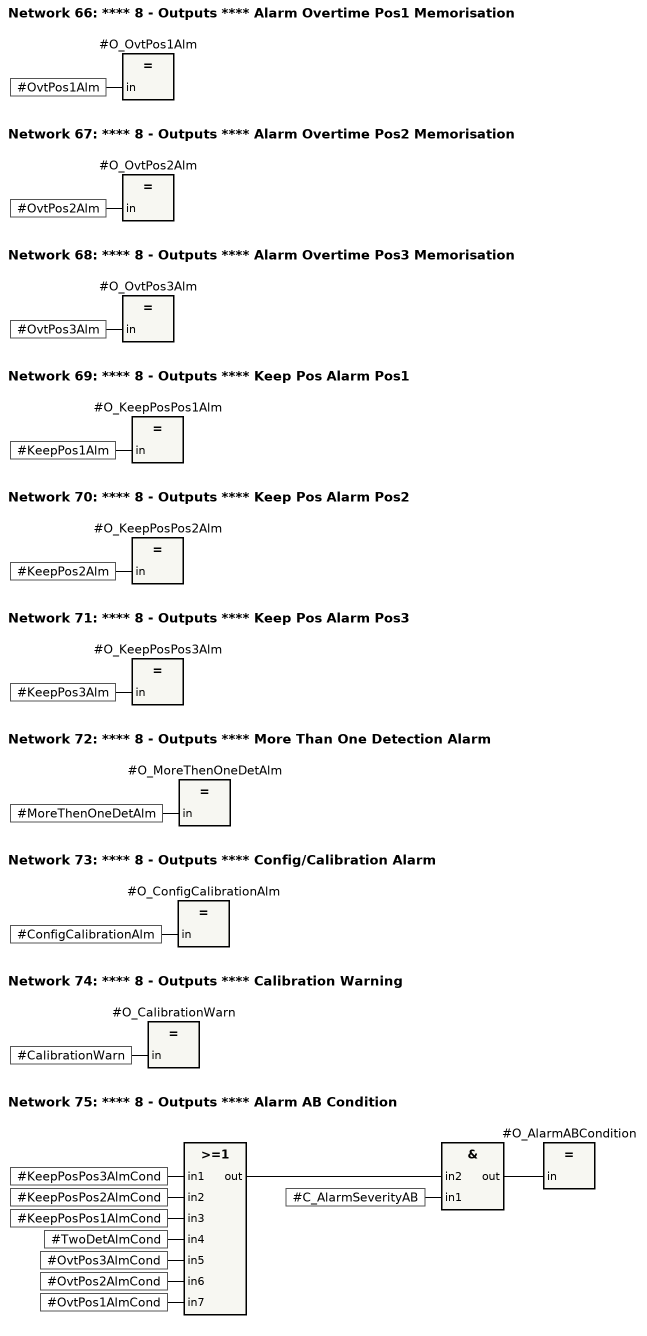
   #O_OvtPos1Alm := #OvtPos1Alm;
END_REGION

REGION Network 67: **** 8 - Outputs **** Alarm Overtime Pos2 Memorisation
   // Alarm Overtime Pos2 Memorisation
   #O_OvtPos2Alm := #OvtPos2Alm;
END_REGION

REGION Network 68: **** 8 - Outputs **** Alarm Overtime Pos3 Memorisation
   // Alarm Overtime Pos3  Memorisation
   #O_OvtPos3Alm := #OvtPos3Alm;
END_REGION

REGION Network 69: **** 8 - Outputs **** Keep Pos Alarm Pos1
   // Keep Pos Alarm Pos1
   #O_KeepPosPos1Alm := #KeepPos1Alm;
END_REGION

REGION Network 70: **** 8 - Outputs **** Keep Pos Alarm Pos2
   // Keep Pos Alarm Pos2
   #O_KeepPosPos2Alm := #KeepPos2Alm;
END_REGION

REGION Network 71: **** 8 - Outputs **** Keep Pos Alarm Pos3
   // Keep Pos Alarm Pos3
   #O_KeepPosPos3Alm := #KeepPos3Alm;
END_REGION

REGION Network 72: **** 8 - Outputs **** More Than One Detection Alarm
   // More Than One Detection Alarm
   #O_MoreThenOneDetAlm := #MoreThenOneDetAlm;
END_REGION

REGION Network 73: **** 8 - Outputs **** Config/Calibration Alarm
   #O_ConfigCalibrationAlm := #ConfigCalibrationAlm;
END_REGION

REGION Network 74: **** 8 - Outputs **** Calibration Warning
   #O_CalibrationWarn := #CalibrationWarn;
END_REGION

REGION Network 75: **** 8 - Outputs **** Alarm AB Condition
   // Alarm AB Condition
   #O_AlarmABCondition := (#KeepPosPos3AlmCond OR #KeepPosPos2AlmCond OR #KeepPosPos1AlmCond OR #TwoDetAlmCond OR #OvtPos3AlmCond OR #OvtPos2AlmCond OR #OvtPos1AlmCond) AND #C_AlarmSeverityAB;
END_REGION
END_FUNCTION_BLOCK

FUNCTION_BLOCK "LMovFnc3Pos2S"   // FB2192, FBD
TITLE = LMovFnc3Pos2S
{ S7_Optimized_Access := 'TRUE' }
VERSION : 0.1
// =============================================================================
// This module will be used for the steering of a three Position movement wit 2 speed
// It will get the commands from different Modes, evaluate the status of the 
// Interlock and give the command to the Actuator or direct to simple outputs.
// =============================================================================
// stored: AutoNumber false, IsIECCheckEnabled false, IsRetainMemResEnabled false, MemoryReserve 100, SetENOAutomatically False, UDAEnableTagReadback false
   VAR_INPUT
      I_Pos1 { ExternalAccessible := 'False'; ExternalVisible := 'False'; ExternalWritable := 'False'} : Bool;   // Position 1 Detection or Summary
      I_Pos2 { ExternalAccessible := 'False'; ExternalVisible := 'False'; ExternalWritable := 'False'} : Bool;   // Position 2 Detection or Summary
      I_Pos3 { ExternalAccessible := 'False'; ExternalVisible := 'False'; ExternalWritable := 'False'} : Bool;   // Position 3 Detection or Summary
      I_SlowPos1 { ExternalAccessible := 'False'; ExternalVisible := 'False'; ExternalWritable := 'False'} : Bool;   // Slow Position 1 Detection
      I_SlowPos2 { ExternalAccessible := 'False'; ExternalVisible := 'False'; ExternalWritable := 'False'} : Bool;   // Slow Position 2 Detection
      I_SlowPos3 { ExternalAccessible := 'False'; ExternalVisible := 'False'; ExternalWritable := 'False'} : Bool;   // Slow Position 3 Detection
      I_PBSet { ExternalAccessible := 'False'; ExternalVisible := 'False'; ExternalWritable := 'False'} : Bool;   // Push button for Set direction (used in manual with button OP panels )
      I_PBReset { ExternalAccessible := 'False'; ExternalVisible := 'False'; ExternalWritable := 'False'} : Bool;   // Push button for Reset direction (used in manual with Pushbutton OP panels)
      I_Pos1Begin { ExternalAccessible := 'False'; ExternalVisible := 'False'; ExternalWritable := 'False'} : Bool;   // Request Pos 1 Function Begin
      I_Pos2Begin { ExternalAccessible := 'False'; ExternalVisible := 'False'; ExternalWritable := 'False'} : Bool;   // Request Pos 2 Function Begin
      I_Pos3Begin { ExternalAccessible := 'False'; ExternalVisible := 'False'; ExternalWritable := 'False'} : Bool;   // Request Pos 3 Function Begin
      I_SetIntlkOK { ExternalAccessible := 'False'; ExternalVisible := 'False'; ExternalWritable := 'False'} : Bool;   // Interlock Set Ok
      I_ResIntlkOK { ExternalAccessible := 'False'; ExternalVisible := 'False'; ExternalWritable := 'False'} : Bool;   // Interlock Reset Ok
      I_SafetyOk { ExternalAccessible := 'False'; ExternalVisible := 'False'; ExternalWritable := 'False'} : Bool;   // Safety ok
      I_HardwareOk { ExternalAccessible := 'False'; ExternalVisible := 'False'; ExternalWritable := 'False'} : Bool;   // Safety Ok / Hardware Ok
   END_VAR
   VAR_OUTPUT
      O_CmdSetHighSpeed { ExternalAccessible := 'False'; ExternalVisible := 'False'; ExternalWritable := 'False'} : Bool;   // Command to Activate Set movement
      O_CmdResHighSpeed { ExternalAccessible := 'False'; ExternalVisible := 'False'; ExternalWritable := 'False'} : Bool;   // Command to Activate Reset movement
      O_CmdSetLowSpeed { ExternalAccessible := 'False'; ExternalVisible := 'False'; ExternalWritable := 'False'} : Bool;   // Command to Activate Slow Set movement
      O_CmdResLowSpeed { ExternalAccessible := 'False'; ExternalVisible := 'False'; ExternalWritable := 'False'} : Bool;   // Command to Activate Slow Reset movement
      O_CmdPos1 { ExternalAccessible := 'False'; ExternalVisible := 'False'; ExternalWritable := 'False'} : Bool;   // Command to activate Set movement / Command to Activate Pos1 movement
      O_CmdPos2 { ExternalAccessible := 'False'; ExternalVisible := 'False'; ExternalWritable := 'False'} : Bool;   // Command to activate Set movement / Command to Activate Pos2 movement
      O_CmdPos3 { ExternalAccessible := 'False'; ExternalVisible := 'False'; ExternalWritable := 'False'} : Bool;   // Command to activate Reset movement / Command to Activate Pos3 movement
      O_FuncRunning { ExternalAccessible := 'False'; ExternalVisible := 'False'; ExternalWritable := 'False'} : Bool;   // Signal that the function is running
      O_FuncBusyTM { ExternalAccessible := 'False'; ExternalVisible := 'False'; ExternalWritable := 'False'} : Bool;   // Memory Signal that the function is busy
      O_Pos1Finished { ExternalAccessible := 'False'; ExternalVisible := 'False'; ExternalWritable := 'False'} : Bool;   // Position1 Finished
      O_Pos2Finished { ExternalAccessible := 'False'; ExternalVisible := 'False'; ExternalWritable := 'False'} : Bool;   // Position2 Finished
      O_Pos3Finished { ExternalAccessible := 'False'; ExternalVisible := 'False'; ExternalWritable := 'False'} : Bool;   // Position3 Finished
      O_IntlkSetAlm { ExternalAccessible := 'False'; ExternalVisible := 'False'; ExternalWritable := 'False'} : Bool;   // Alarm Interlock Set
      O_IntlkResAlm { ExternalAccessible := 'False'; ExternalVisible := 'False'; ExternalWritable := 'False'} : Bool;   // Alarm Interlock Reset
      O_FuncIsSelInMan { ExternalAccessible := 'False'; ExternalVisible := 'False'; ExternalWritable := 'False'} : Bool;   // The function is Selected in manual Mode
      O_LED { ExternalAccessible := 'False'; ExternalVisible := 'False'; ExternalWritable := 'False'} : Bool;   // LED - Indication
      O_AlarmABCondition { ExternalAccessible := 'False'; ExternalVisible := 'False'; ExternalWritable := 'False'} : Bool;   // Alarms AB condition
   END_VAR
   VAR_IN_OUT
      IO_Modes : "Modes";   // Modes
      H_HMI : "H_HMI";   // Animation
      H_MovFnc3Pos2S : "H_MovFnc3Pos";   // Animation
      H_FncSelInHMI { ExternalAccessible := 'False'; ExternalVisible := 'False'; ExternalWritable := 'False'} : Bool;   // This function is Selected to run from HMI
      C_AlarmResetUsed { ExternalAccessible := 'False'; ExternalVisible := 'False'; ExternalWritable := 'False'} : Bool;   // If true, the alrms will be stored untill Reseted
      C_EnableMemBegin { ExternalAccessible := 'False'; ExternalVisible := 'False'; ExternalWritable := 'False'} : Bool;   // Enable memory Begin (Command request is memorised until pos reached)
      C_EnIntlkAlm { ExternalAccessible := 'False'; ExternalVisible := 'False'; ExternalWritable := 'False'} : Bool := TRUE;   // Enable Interlock Alarm
      C_ForceManual { ExternalAccessible := 'False'; ExternalVisible := 'False'; ExternalWritable := 'False'} : Bool := FALSE;   // Force Manual
   END_VAR
   VAR
      ResetAlarm { ExternalAccessible := 'False'; ExternalVisible := 'False'; ExternalWritable := 'False'} : Bool;   // Reset Alarm Memory
      BeginPos1Req { ExternalAccessible := 'False'; ExternalVisible := 'False'; ExternalWritable := 'False'} : Bool;   // Request Pos 1 Function Begin
      BeginPos2Req { ExternalAccessible := 'False'; ExternalVisible := 'False'; ExternalWritable := 'False'} : Bool;   // Request Pos 2 Function Begin
      BeginPos3Req { ExternalAccessible := 'False'; ExternalVisible := 'False'; ExternalWritable := 'False'} : Bool;   // Request Pos 3 Function Begin
      CmdSet { ExternalAccessible := 'False'; ExternalVisible := 'False'; ExternalWritable := 'False'} : Bool;   // Command set
      CmdSetSl { ExternalAccessible := 'False'; ExternalVisible := 'False'; ExternalWritable := 'False'} : Bool;   // Command to Activate Slow Set movement
      CmdSetRequest { ExternalAccessible := 'False'; ExternalVisible := 'False'; ExternalWritable := 'False'} : Bool;   // Set Command request to Activate the Interlock
      CmdRes { ExternalAccessible := 'False'; ExternalVisible := 'False'; ExternalWritable := 'False'} : Bool;   // Command Reset
      CmdResSl { ExternalAccessible := 'False'; ExternalVisible := 'False'; ExternalWritable := 'False'} : Bool;   // Command to Activate Slow Reset movement
      CmdResRequest { ExternalAccessible := 'False'; ExternalVisible := 'False'; ExternalWritable := 'False'} : Bool;   // Reset Command request to Activate the Interlock
   END_VAR
   VAR RETAIN
      BetweenPos1Pos2 { ExternalAccessible := 'False'; ExternalVisible := 'False'; ExternalWritable := 'False'} : Bool;   // Table Between Pos 1 And 2
      BetweenPos1Pos2Set { ExternalAccessible := 'False'; ExternalVisible := 'False'; ExternalWritable := 'False'} : Bool;   // Table Between Pos 1 And 2 Set
      BetweenPos1Pos2Res { ExternalAccessible := 'False'; ExternalVisible := 'False'; ExternalWritable := 'False'} : Bool;   // Table Between Pos 1 And 2 Reset
      BetweenPos2Pos3 { ExternalAccessible := 'False'; ExternalVisible := 'False'; ExternalWritable := 'False'} : Bool;   // Table Between Pos 2 And 3
      BetweenPos2Pos3Set { ExternalAccessible := 'False'; ExternalVisible := 'False'; ExternalWritable := 'False'} : Bool;   // Table Between Pos 2 And 3 Set
      BetweenPos2Pos3Res { ExternalAccessible := 'False'; ExternalVisible := 'False'; ExternalWritable := 'False'} : Bool;   // Table Between Pos 2 And 3 Reset
   END_VAR
   VAR
      Pos2SetReached { ExternalAccessible := 'False'; ExternalVisible := 'False'; ExternalWritable := 'False'} : Bool;   // Position 2 Set Reached
      P_CmdSetRequest { ExternalAccessible := 'False'; ExternalVisible := 'False'; ExternalWritable := 'False'} : Bool;   // Cmd Request Set Pos Trig
      Pos2ResReached { ExternalAccessible := 'False'; ExternalVisible := 'False'; ExternalWritable := 'False'} : Bool;   // Position 2 Reset Reached
      P_CmdResRequest { ExternalAccessible := 'False'; ExternalVisible := 'False'; ExternalWritable := 'False'} : Bool;   // Cmd Request Res Pos Trig
      CmdPos1 { ExternalAccessible := 'False'; ExternalVisible := 'False'; ExternalWritable := 'False'} : Bool;   // Command to activate Set movement / Command to Activate Pos1 movement
      CmdPos2 { ExternalAccessible := 'False'; ExternalVisible := 'False'; ExternalWritable := 'False'} : Bool;   // Command to activate Set movement / Command to Activate Pos2 movement
      CmdPos3 { ExternalAccessible := 'False'; ExternalVisible := 'False'; ExternalWritable := 'False'} : Bool;   // Command to activate Reset movement / Command to Activate Pos3 movement
      IntlkSetAlm { ExternalAccessible := 'False'; ExternalVisible := 'False'; ExternalWritable := 'False'} : Bool;   // Alarm Interlock Set
      IntlkResAlm { ExternalAccessible := 'False'; ExternalVisible := 'False'; ExternalWritable := 'False'} : Bool;   // Alarm Interlock Reset
      IntlkSetAlmCond { ExternalAccessible := 'False'; ExternalVisible := 'False'; ExternalWritable := 'False'} : Bool;   // Alarm Interlock Set condition
      IntlkResAlmCond { ExternalAccessible := 'False'; ExternalVisible := 'False'; ExternalWritable := 'False'} : Bool;   // Alarm Interlock Reset condition
      FuncRunning { ExternalAccessible := 'False'; ExternalVisible := 'False'; ExternalWritable := 'False'} : Bool;   // Function is running
      FuncBusyTM { ExternalAccessible := 'False'; ExternalVisible := 'False'; ExternalWritable := 'False'} : Bool;   // Memory Signal that the function is busy
      Edge { ExternalAccessible := 'False'; ExternalVisible := 'False'; ExternalWritable := 'False'} : Array[1..5] of Bool;   // Edge
      AlarmTimer { ExternalAccessible := 'False'; ExternalVisible := 'False'; ExternalWritable := 'False'} : "LTimer";
      AlmFilterResult { ExternalAccessible := 'False'; ExternalVisible := 'False'; ExternalWritable := 'False'} : Bool;
   END_VAR
   VAR_TEMP   // added for the SCL form of the ladder/FBD networks
      _w1 : Bool;
      _w2 : Bool;
      _w3 : Bool;
      _w4 : Bool;
   END_VAR
BEGIN

REGION Network 1: **** 2.2 - Alarms - Alarm Generation **** Alarm Filter
   // Alarm Filter
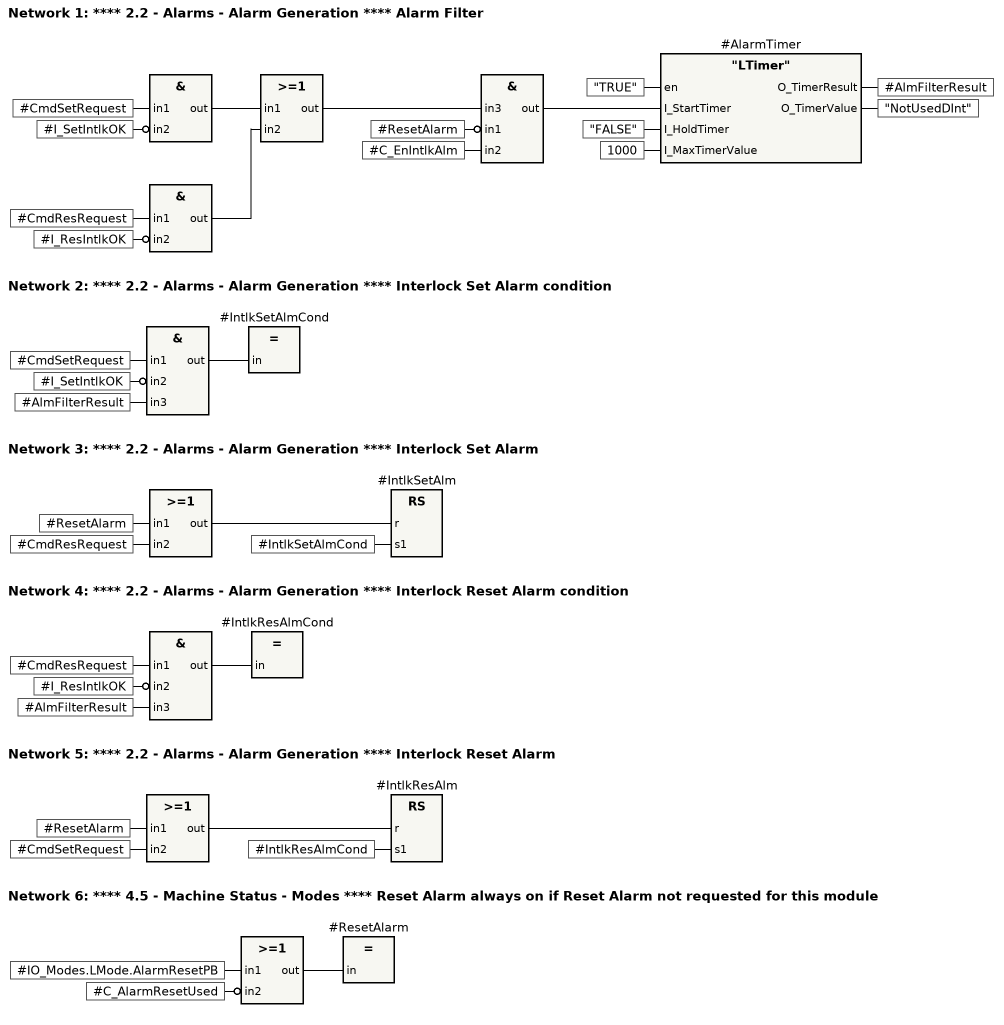
   IF "TRUE" THEN
       #AlarmTimer(I_StartTimer := ((#CmdSetRequest AND NOT #I_SetIntlkOK) OR (#CmdResRequest AND NOT #I_ResIntlkOK)) AND NOT #ResetAlarm AND #C_EnIntlkAlm,   // "LTimer"
                   I_HoldTimer := "FALSE",
                   I_MaxTimerValue := 1000,
                   O_TimerResult => #AlmFilterResult,
                   O_TimerValue => "NotUsedDInt");
   END_IF;
END_REGION

REGION Network 2: **** 2.2 - Alarms - Alarm Generation **** Interlock Set Alarm condition
   // Interlock Set Alarm condition
   #IntlkSetAlmCond := #CmdSetRequest AND NOT #I_SetIntlkOK AND #AlmFilterResult;
END_REGION

REGION Network 3: **** 2.2 - Alarms - Alarm Generation **** Interlock Set Alarm
   // Interlock Set Alarm
   IF #ResetAlarm OR #CmdResRequest THEN
       #IntlkSetAlm := FALSE;   // RS flip-flop
   END_IF;
   IF #IntlkSetAlmCond THEN #IntlkSetAlm := TRUE; END_IF;
END_REGION

REGION Network 4: **** 2.2 - Alarms - Alarm Generation **** Interlock Reset Alarm condition
   // Interlock Reset Alarm condition
   #IntlkResAlmCond := #CmdResRequest AND NOT #I_ResIntlkOK AND #AlmFilterResult;
END_REGION

REGION Network 5: **** 2.2 - Alarms - Alarm Generation **** Interlock Reset Alarm
   // Interlock Reset Alarm
   IF #ResetAlarm OR #CmdSetRequest THEN
       #IntlkResAlm := FALSE;   // RS flip-flop
   END_IF;
   IF #IntlkResAlmCond THEN #IntlkResAlm := TRUE; END_IF;
END_REGION

REGION Network 6: **** 4.5 - Machine Status - Modes **** Reset Alarm always on if Reset Alarm not requested for this module
   // Reset Alarm always on if Reset Alarm not requested for this module
   #ResetAlarm := #IO_Modes.LMode.AlarmResetPB OR NOT #C_AlarmResetUsed;
END_REGION

REGION Network 7: **** 4.6 - Machine Status - Indication **** Icon Animation
   // Icon Animation
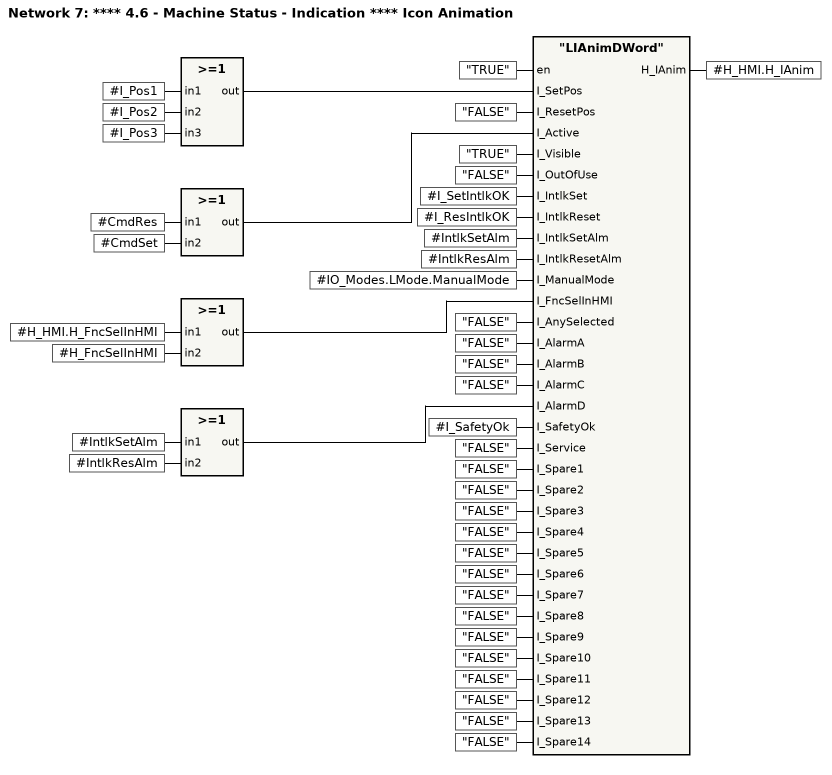
   IF "TRUE" THEN
       "LIAnimDWord"(I_SetPos := #I_Pos1 OR #I_Pos2 OR #I_Pos3,
                     I_ResetPos := "FALSE",
                     I_Active := #CmdRes OR #CmdSet,
                     I_Visible := "TRUE",
                     I_OutOfUse := "FALSE",
                     I_IntlkSet := #I_SetIntlkOK,
                     I_IntlkReset := #I_ResIntlkOK,
                     I_IntlkSetAlm := #IntlkSetAlm,
                     I_IntlkResetAlm := #IntlkResAlm,
                     I_ManualMode := #IO_Modes.LMode.ManualMode,
                     I_FncSelInHMI := #H_HMI.H_FncSelInHMI OR #H_FncSelInHMI,
                     I_AnySelected := "FALSE",
                     I_AlarmA := "FALSE",
                     I_AlarmB := "FALSE",
                     I_AlarmC := "FALSE",
                     I_AlarmD := #IntlkSetAlm OR #IntlkResAlm,
                     I_SafetyOk := #I_SafetyOk,
                     I_Service := "FALSE",
                     I_Spare1 := "FALSE",
                     I_Spare2 := "FALSE",
                     I_Spare3 := "FALSE",
                     I_Spare4 := "FALSE",
                     I_Spare5 := "FALSE",
                     I_Spare6 := "FALSE",
                     I_Spare7 := "FALSE",
                     I_Spare8 := "FALSE",
                     I_Spare9 := "FALSE",
                     I_Spare10 := "FALSE",
                     I_Spare11 := "FALSE",
                     I_Spare12 := "FALSE",
                     I_Spare13 := "FALSE",
                     I_Spare14 := "FALSE",
                     H_IAnim => #H_HMI.H_IAnim);
   END_IF;
END_REGION

REGION Network 8: **** 4.6 - Machine Status - Indication **** Animation
   // Animation
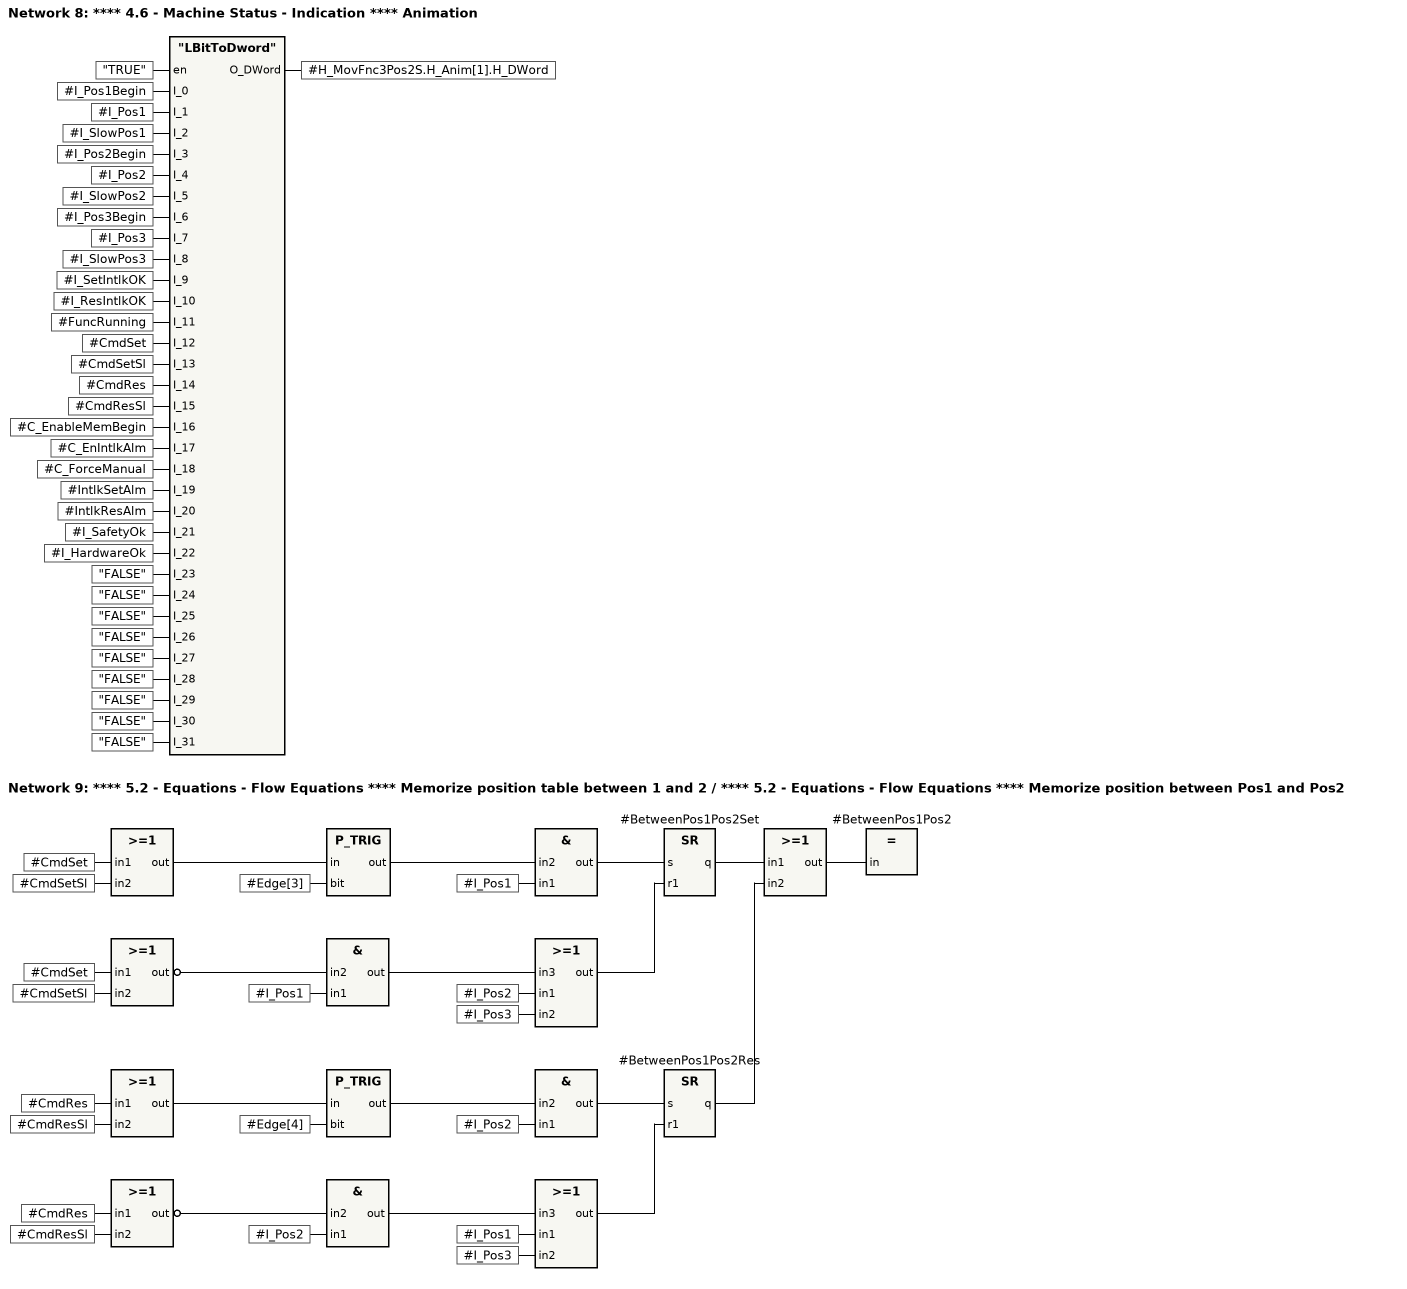
   IF "TRUE" THEN
       "LBitToDword"(I_0 := #I_Pos1Begin,
                     I_1 := #I_Pos1,
                     I_2 := #I_SlowPos1,
                     I_3 := #I_Pos2Begin,
                     I_4 := #I_Pos2,
                     I_5 := #I_SlowPos2,
                     I_6 := #I_Pos3Begin,
                     I_7 := #I_Pos3,
                     I_8 := #I_SlowPos3,
                     I_9 := #I_SetIntlkOK,
                     I_10 := #I_ResIntlkOK,
                     I_11 := #FuncRunning,
                     I_12 := #CmdSet,
                     I_13 := #CmdSetSl,
                     I_14 := #CmdRes,
                     I_15 := #CmdResSl,
                     I_16 := #C_EnableMemBegin,
                     I_17 := #C_EnIntlkAlm,
                     I_18 := #C_ForceManual,
                     I_19 := #IntlkSetAlm,
                     I_20 := #IntlkResAlm,
                     I_21 := #I_SafetyOk,
                     I_22 := #I_HardwareOk,
                     I_23 := "FALSE",
                     I_24 := "FALSE",
                     I_25 := "FALSE",
                     I_26 := "FALSE",
                     I_27 := "FALSE",
                     I_28 := "FALSE",
                     I_29 := "FALSE",
                     I_30 := "FALSE",
                     I_31 := "FALSE",
                     O_DWord => #H_MovFnc3Pos2S.H_Anim[1].H_DWord);
   END_IF;
END_REGION

REGION Network 9: **** 5.2 - Equations - Flow Equations **** Memorize position table between 1 and 2 / **** 5.2 - Equations - Flow Equations **** Memorize position between Pos1 and Pos2
   // Memorize Position table between 1 and 2
   #_w1 := #CmdSet OR #CmdSetSl;
   #_w2 := #_w1 AND NOT #Edge[3];   // rising edge
   #Edge[3] := #_w1;
   IF #_w2 AND #I_Pos1 THEN
       #BetweenPos1Pos2Set := TRUE;   // SR flip-flop
   END_IF;
   IF (NOT (#CmdSet OR #CmdSetSl) AND #I_Pos1) OR #I_Pos2 OR #I_Pos3 THEN
       #BetweenPos1Pos2Set := FALSE;
   END_IF;
   #_w3 := #CmdRes OR #CmdResSl;
   #_w4 := #_w3 AND NOT #Edge[4];   // rising edge
   #Edge[4] := #_w3;
   IF #_w4 AND #I_Pos2 THEN
       #BetweenPos1Pos2Res := TRUE;   // SR flip-flop
   END_IF;
   IF (NOT (#CmdRes OR #CmdResSl) AND #I_Pos2) OR #I_Pos1 OR #I_Pos3 THEN
       #BetweenPos1Pos2Res := FALSE;
   END_IF;
   #BetweenPos1Pos2 := #BetweenPos1Pos2Set OR #BetweenPos1Pos2Res;
END_REGION

REGION Network 10: **** 5.2 - Equations - Flow Equations **** Memorize position between 2 and 3 / **** 5.2 - Equations - Flow Equations **** Memorize position between Pos2 and Pos3
   // Memorize Position table  2 and 3
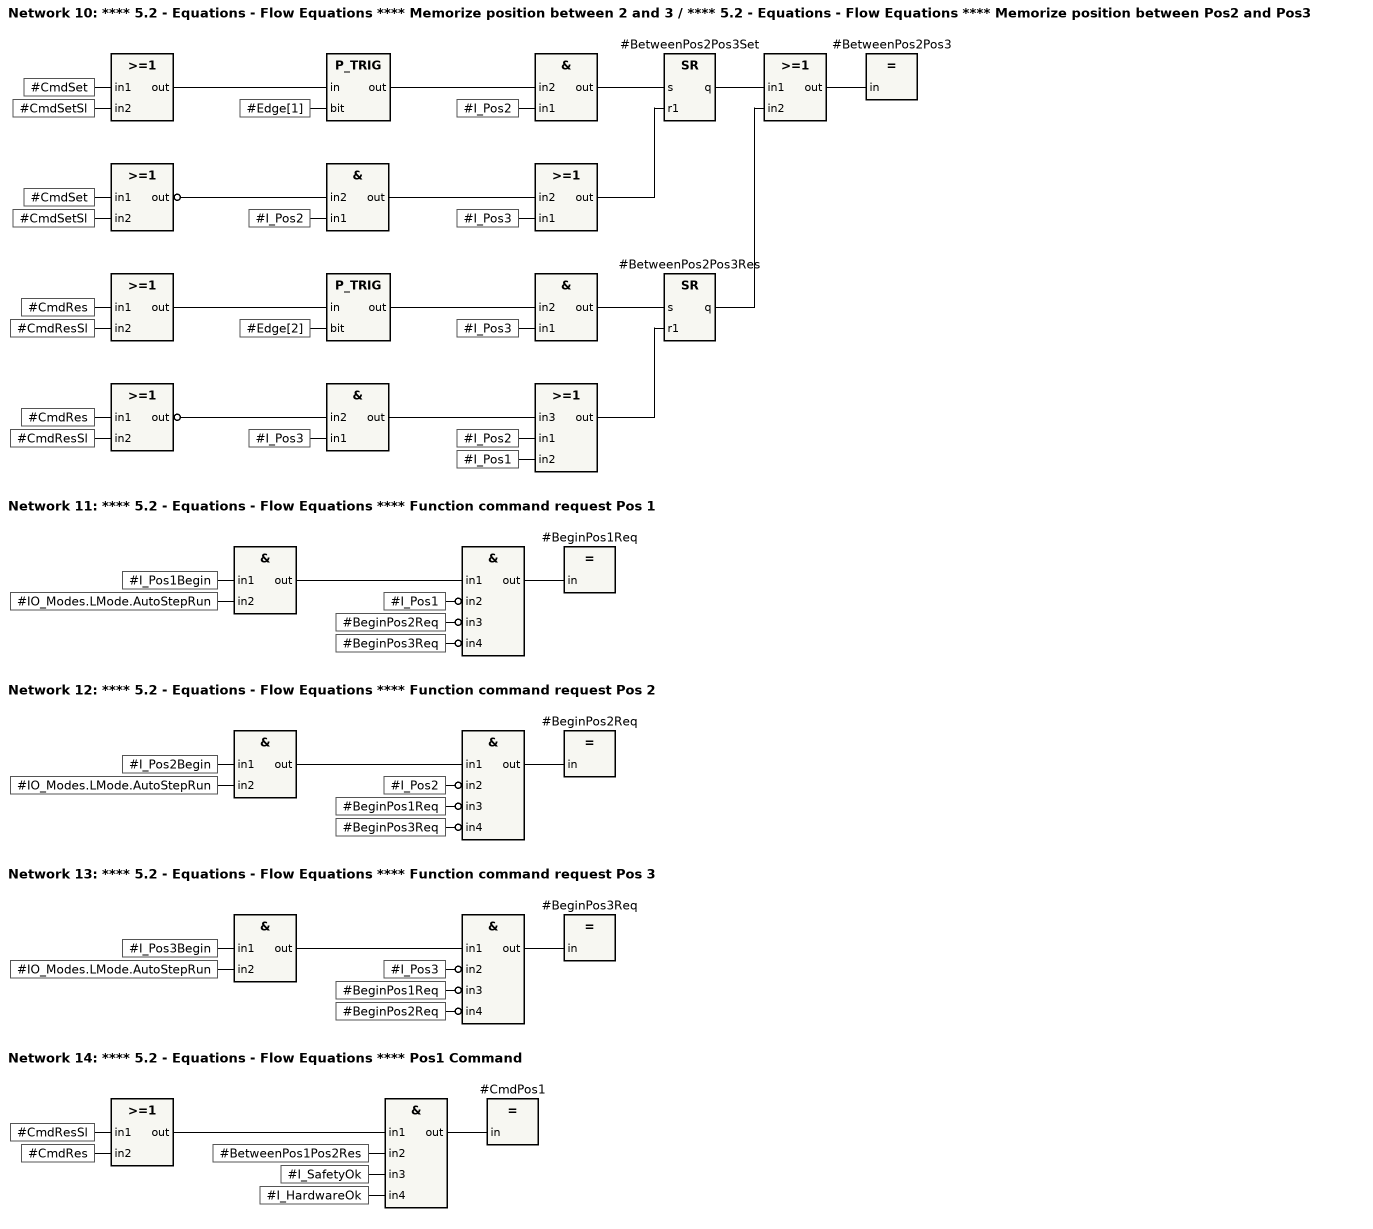
   #_w1 := #CmdSet OR #CmdSetSl;
   #_w2 := #_w1 AND NOT #Edge[1];   // rising edge
   #Edge[1] := #_w1;
   IF #_w2 AND #I_Pos2 THEN
       #BetweenPos2Pos3Set := TRUE;   // SR flip-flop
   END_IF;
   IF (NOT (#CmdSet OR #CmdSetSl) AND #I_Pos2) OR #I_Pos3 THEN #BetweenPos2Pos3Set := FALSE; END_IF;
   #_w3 := #CmdRes OR #CmdResSl;
   #_w4 := #_w3 AND NOT #Edge[2];   // rising edge
   #Edge[2] := #_w3;
   IF #_w4 AND #I_Pos3 THEN
       #BetweenPos2Pos3Res := TRUE;   // SR flip-flop
   END_IF;
   IF (NOT (#CmdRes OR #CmdResSl) AND #I_Pos3) OR #I_Pos2 OR #I_Pos1 THEN
       #BetweenPos2Pos3Res := FALSE;
   END_IF;
   #BetweenPos2Pos3 := #BetweenPos2Pos3Set OR #BetweenPos2Pos3Res;
END_REGION

REGION Network 11: **** 5.2 - Equations - Flow Equations **** Function command request Pos 1
   // Function command request Pos 1
   #BeginPos1Req := #I_Pos1Begin AND #IO_Modes.LMode.AutoStepRun AND NOT #I_Pos1 AND NOT #BeginPos2Req AND NOT #BeginPos3Req;
END_REGION

REGION Network 12: **** 5.2 - Equations - Flow Equations **** Function command request Pos 2
   // Function command request Pos 2
   #BeginPos2Req := #I_Pos2Begin AND #IO_Modes.LMode.AutoStepRun AND NOT #I_Pos2 AND NOT #BeginPos1Req AND NOT #BeginPos3Req;
END_REGION

REGION Network 13: **** 5.2 - Equations - Flow Equations **** Function command request Pos 3
   // Function command request Pos 3
   #BeginPos3Req := #I_Pos3Begin AND #IO_Modes.LMode.AutoStepRun AND NOT #I_Pos3 AND NOT #BeginPos1Req AND NOT #BeginPos2Req;
END_REGION

REGION Network 14: **** 5.2 - Equations - Flow Equations **** Pos1 Command
   // Pos1 Command
   #CmdPos1 := (#CmdResSl OR #CmdRes) AND #BetweenPos1Pos2Res AND #I_SafetyOk AND #I_HardwareOk;
END_REGION

REGION Network 15: **** 5.2 - Equations - Flow Equations **** Pos2 Command
   // Pos2 Command
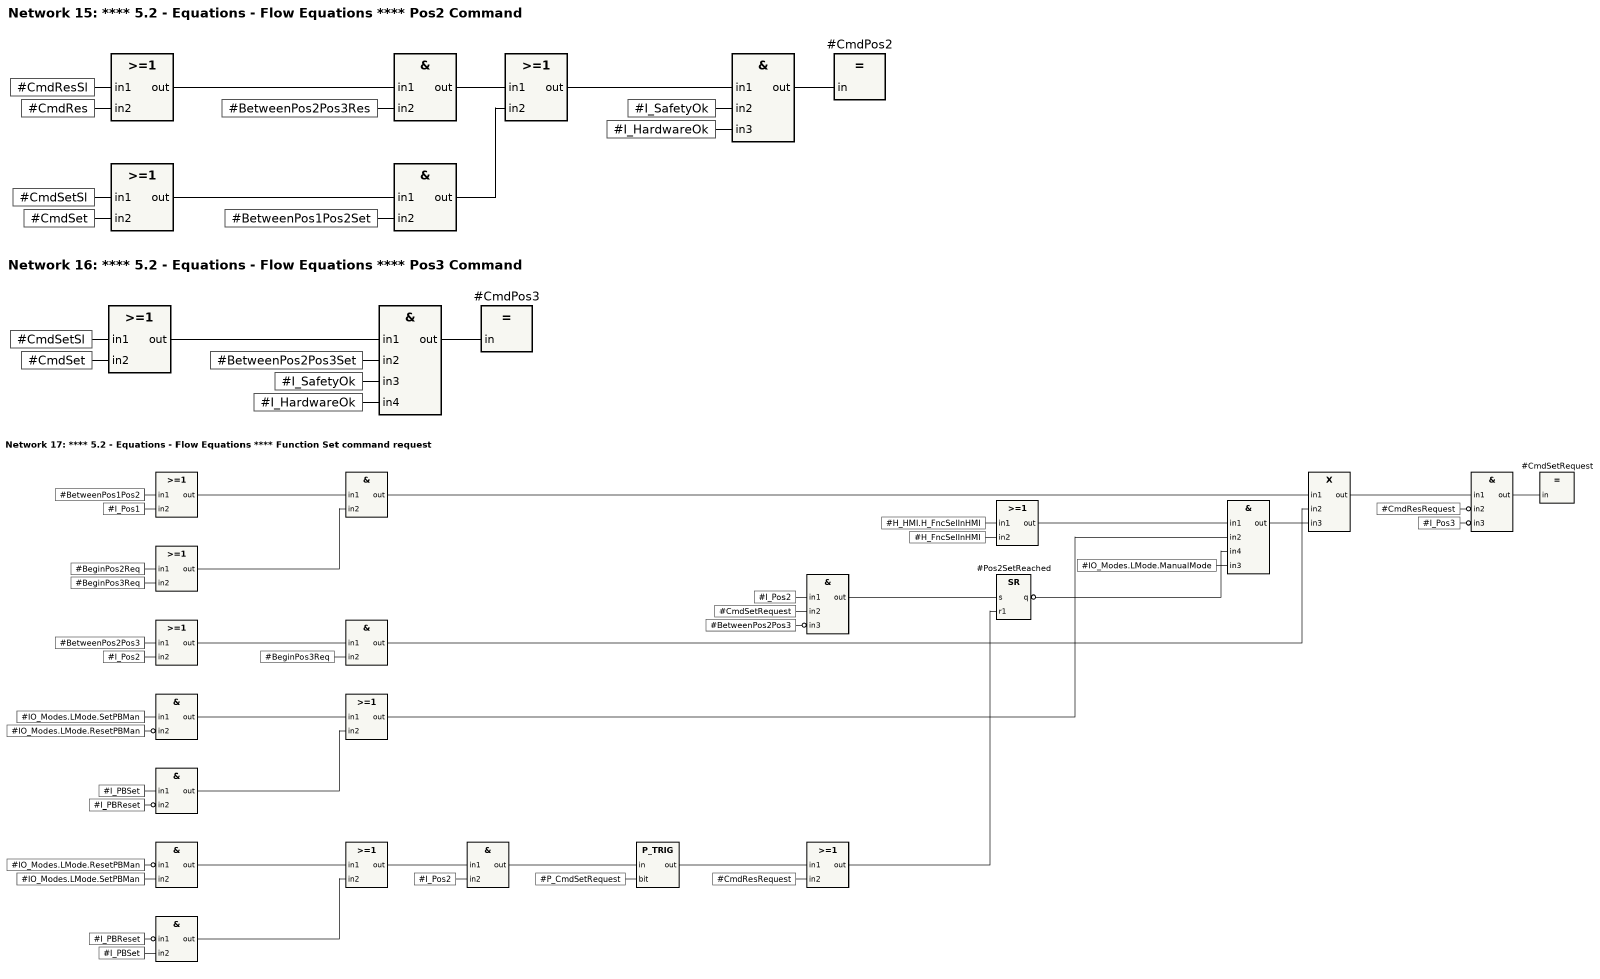
   #CmdPos2 := (((#CmdResSl OR #CmdRes) AND #BetweenPos2Pos3Res) OR ((#CmdSetSl OR #CmdSet) AND #BetweenPos1Pos2Set)) AND #I_SafetyOk AND #I_HardwareOk;
END_REGION

REGION Network 16: **** 5.2 - Equations - Flow Equations **** Pos3 Command
   // Pos3 Command
   #CmdPos3 := (#CmdSetSl OR #CmdSet) AND #BetweenPos2Pos3Set AND #I_SafetyOk AND #I_HardwareOk;
END_REGION

REGION Network 17: **** 5.2 - Equations - Flow Equations **** Function Set command request
   // Function Set command request
   #_w1 := ((NOT #IO_Modes.LMode.ResetPBMan AND #IO_Modes.LMode.SetPBMan) OR (NOT #I_PBReset AND #I_PBSet)) AND #I_Pos2;
   #_w2 := #_w1 AND NOT #P_CmdSetRequest;   // rising edge
   #P_CmdSetRequest := #_w1;
   IF #I_Pos2 AND #CmdSetRequest AND NOT #BetweenPos2Pos3 THEN
       #Pos2SetReached := TRUE;   // SR flip-flop
   END_IF;
   IF #_w2 OR #CmdResRequest THEN #Pos2SetReached := FALSE; END_IF;
   #CmdSetRequest := (((#BetweenPos1Pos2 OR #I_Pos1) AND (#BeginPos2Req OR #BeginPos3Req)) XOR ((#BetweenPos2Pos3 OR #I_Pos2) AND #BeginPos3Req) XOR ((#H_HMI.H_FncSelInHMI OR #H_FncSelInHMI) AND ((#IO_Modes.LMode.SetPBMan AND NOT #IO_Modes.LMode.ResetPBMan) OR (#I_PBSet AND NOT #I_PBReset)) AND NOT #Pos2SetReached AND #IO_Modes.LMode.ManualMode)) AND NOT #CmdResRequest AND NOT #I_Pos3;
END_REGION

REGION Network 18: **** 5.2 - Equations - Flow Equations **** Function Reset command request
   // Function Reset command request
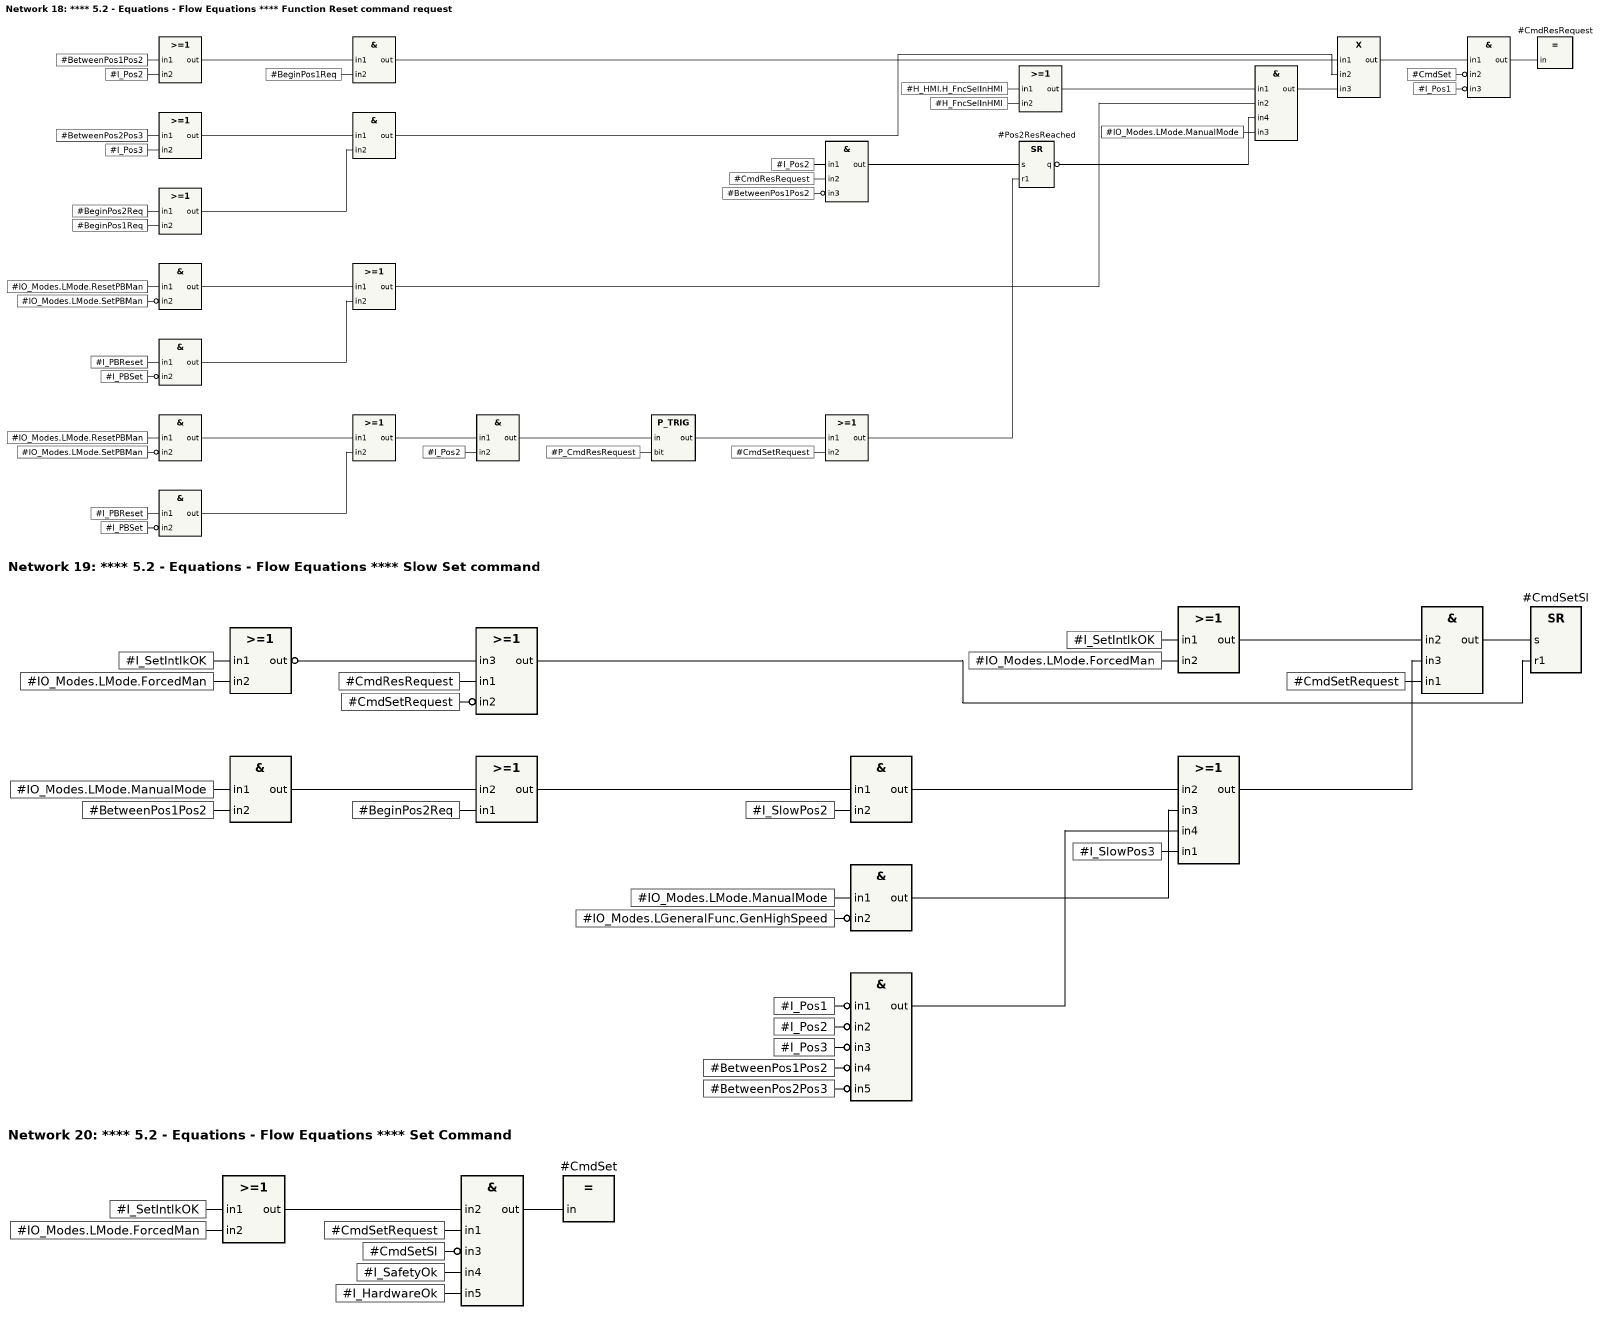
   #_w1 := ((#IO_Modes.LMode.ResetPBMan AND NOT #IO_Modes.LMode.SetPBMan) OR (#I_PBReset AND NOT #I_PBSet)) AND #I_Pos2;
   #_w2 := #_w1 AND NOT #P_CmdResRequest;   // rising edge
   #P_CmdResRequest := #_w1;
   IF #I_Pos2 AND #CmdResRequest AND NOT #BetweenPos1Pos2 THEN
       #Pos2ResReached := TRUE;   // SR flip-flop
   END_IF;
   IF #_w2 OR #CmdSetRequest THEN #Pos2ResReached := FALSE; END_IF;
   #CmdResRequest := (((#BetweenPos1Pos2 OR #I_Pos2) AND #BeginPos1Req) XOR ((#BetweenPos2Pos3 OR #I_Pos3) AND (#BeginPos2Req OR #BeginPos1Req)) XOR ((#H_HMI.H_FncSelInHMI OR #H_FncSelInHMI) AND ((#IO_Modes.LMode.ResetPBMan AND NOT #IO_Modes.LMode.SetPBMan) OR (#I_PBReset AND NOT #I_PBSet)) AND NOT #Pos2ResReached AND #IO_Modes.LMode.ManualMode)) AND NOT #CmdSet AND NOT #I_Pos1;
END_REGION

REGION Network 19: **** 5.2 - Equations - Flow Equations **** Slow Set command
   // Slow Set command
   IF (#I_SetIntlkOK OR #IO_Modes.LMode.ForcedMan) AND ((((#IO_Modes.LMode.ManualMode AND #BetweenPos1Pos2) OR #BeginPos2Req) AND #I_SlowPos2) OR (#IO_Modes.LMode.ManualMode AND NOT #IO_Modes.LGeneralFunc.GenHighSpeed) OR (NOT #I_Pos1 AND NOT #I_Pos2 AND NOT #I_Pos3 AND NOT #BetweenPos1Pos2 AND NOT #BetweenPos2Pos3) OR #I_SlowPos3) AND #CmdSetRequest THEN
       #CmdSetSl := TRUE;   // SR flip-flop
   END_IF;
   IF NOT (#I_SetIntlkOK OR #IO_Modes.LMode.ForcedMan) OR #CmdResRequest OR NOT #CmdSetRequest THEN
       #CmdSetSl := FALSE;
   END_IF;
END_REGION

REGION Network 20: **** 5.2 - Equations - Flow Equations **** Set Command
   // Set Command
   #CmdSet := (#I_SetIntlkOK OR #IO_Modes.LMode.ForcedMan) AND #CmdSetRequest AND NOT #CmdSetSl AND #I_SafetyOk AND #I_HardwareOk;
END_REGION

REGION Network 21: **** 5.2 - Equations - Flow Equations **** Slow Reset command
   // Slow Reset command
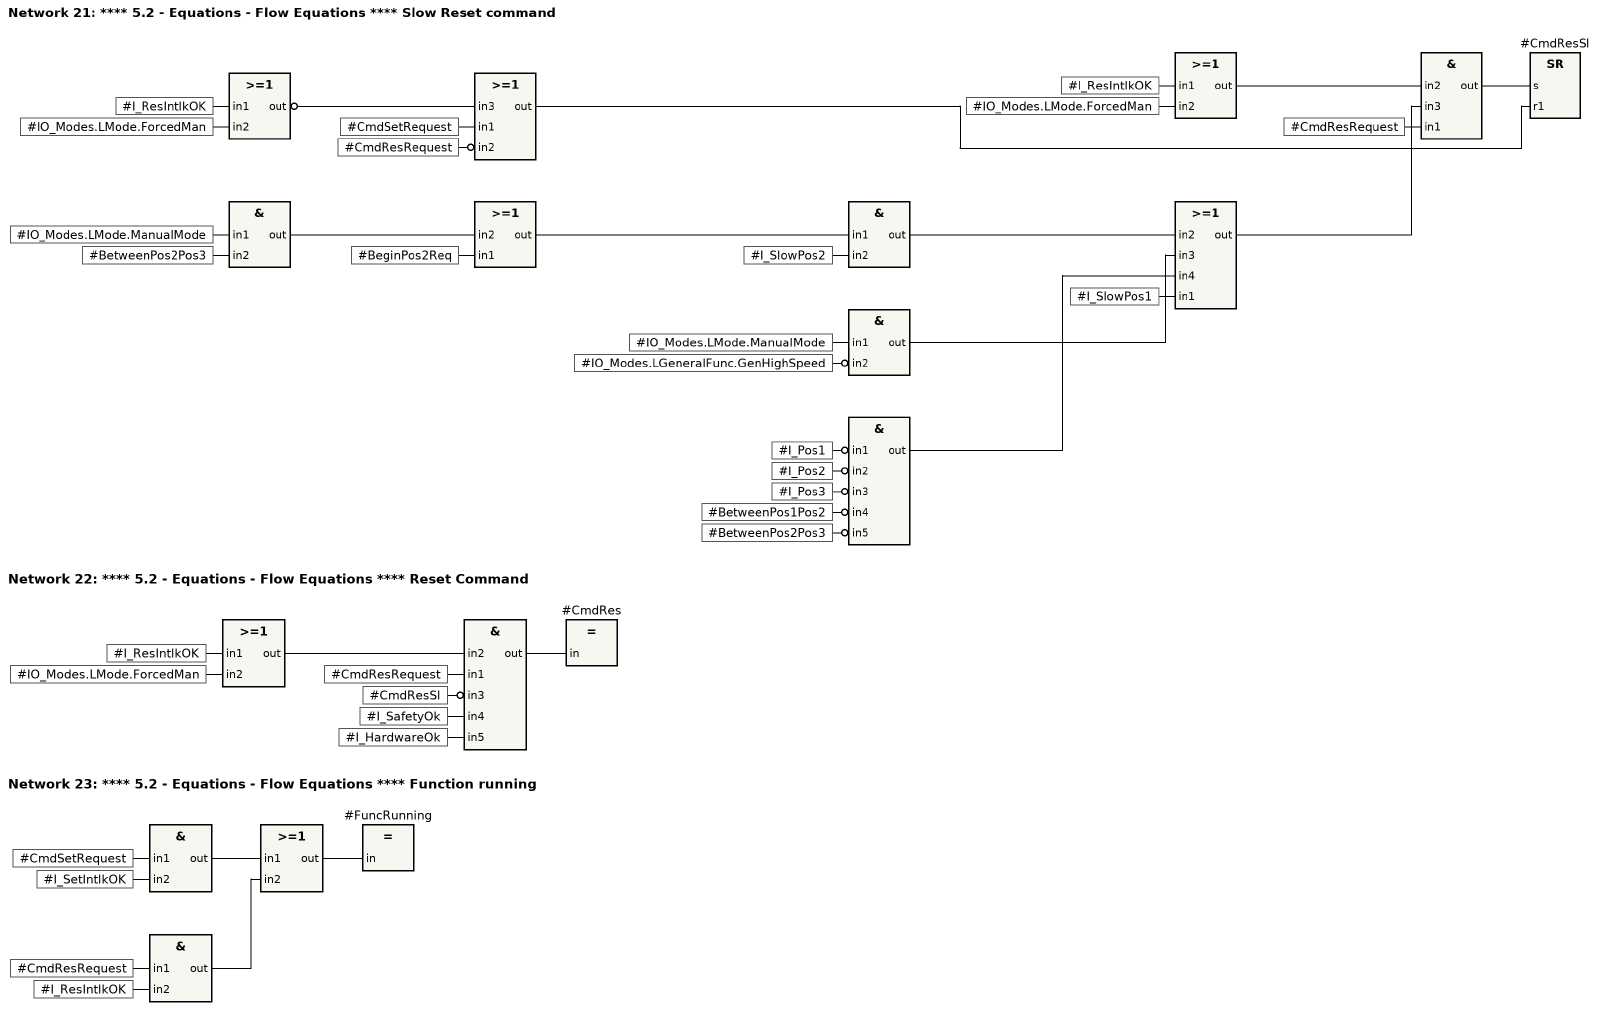
   IF (#I_ResIntlkOK OR #IO_Modes.LMode.ForcedMan) AND ((((#IO_Modes.LMode.ManualMode AND #BetweenPos2Pos3) OR #BeginPos2Req) AND #I_SlowPos2) OR (#IO_Modes.LMode.ManualMode AND NOT #IO_Modes.LGeneralFunc.GenHighSpeed) OR (NOT #I_Pos1 AND NOT #I_Pos2 AND NOT #I_Pos3 AND NOT #BetweenPos1Pos2 AND NOT #BetweenPos2Pos3) OR #I_SlowPos1) AND #CmdResRequest THEN
       #CmdResSl := TRUE;   // SR flip-flop
   END_IF;
   IF NOT (#I_ResIntlkOK OR #IO_Modes.LMode.ForcedMan) OR #CmdSetRequest OR NOT #CmdResRequest THEN
       #CmdResSl := FALSE;
   END_IF;
END_REGION

REGION Network 22: **** 5.2 - Equations - Flow Equations **** Reset Command
   // Reset Command
   #CmdRes := (#I_ResIntlkOK OR #IO_Modes.LMode.ForcedMan) AND #CmdResRequest AND NOT #CmdResSl AND #I_SafetyOk AND #I_HardwareOk;
END_REGION

REGION Network 23: **** 5.2 - Equations - Flow Equations **** Function running
   // Function running
   #FuncRunning := (#CmdSetRequest AND #I_SetIntlkOK) OR (#CmdResRequest AND #I_ResIntlkOK);
END_REGION

REGION Network 24: **** 5.2 - Equations - Flow Equations **** Set Function Running
   // Set Function Running
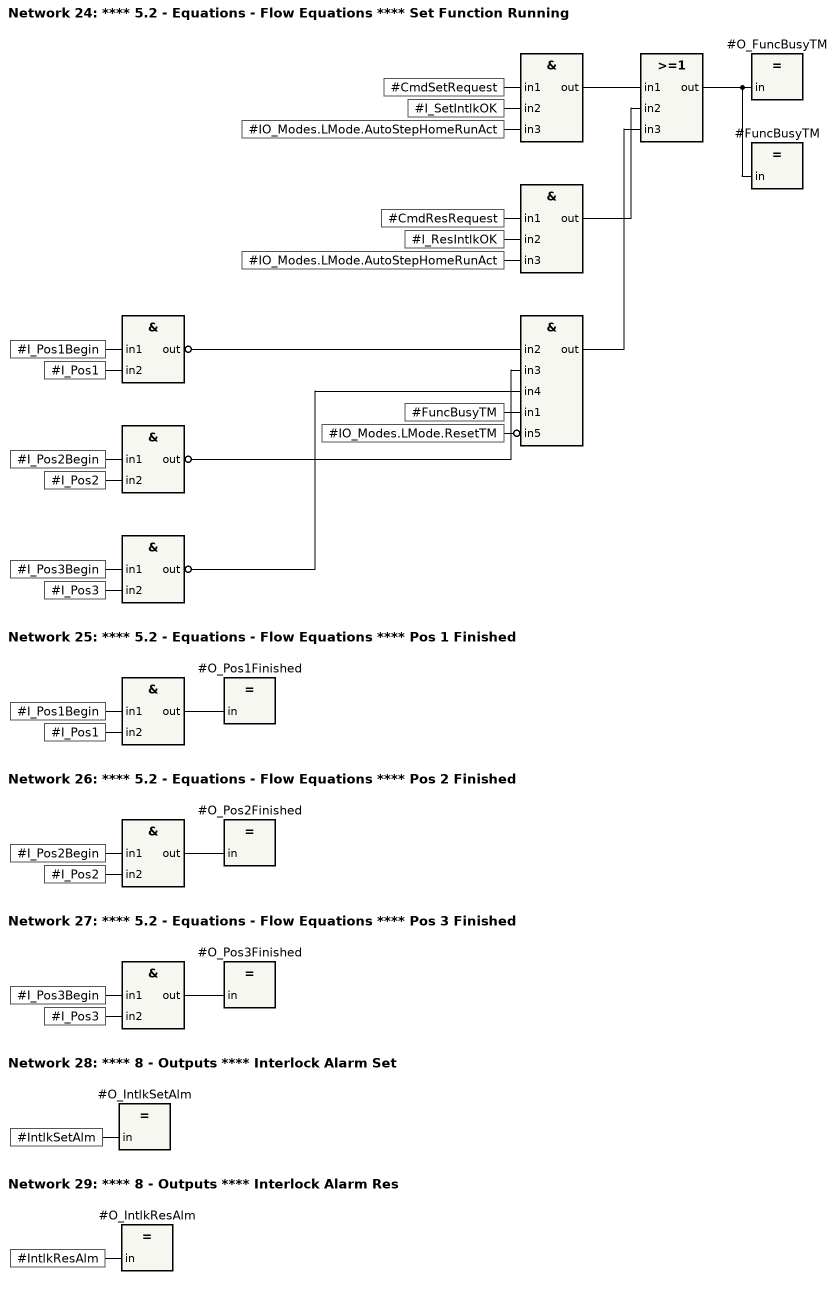
   #O_FuncBusyTM := (#CmdSetRequest AND #I_SetIntlkOK AND #IO_Modes.LMode.AutoStepHomeRunAct) OR (#CmdResRequest AND #I_ResIntlkOK AND #IO_Modes.LMode.AutoStepHomeRunAct) OR (NOT (#I_Pos1Begin AND #I_Pos1) AND NOT (#I_Pos2Begin AND #I_Pos2) AND NOT (#I_Pos3Begin AND #I_Pos3) AND #FuncBusyTM AND NOT #IO_Modes.LMode.ResetTM);
   #FuncBusyTM := #O_FuncBusyTM;
END_REGION

REGION Network 25: **** 5.2 - Equations - Flow Equations **** Pos 1 Finished
   // Pos 1 Finished
   #O_Pos1Finished := #I_Pos1Begin AND #I_Pos1;
END_REGION

REGION Network 26: **** 5.2 - Equations - Flow Equations **** Pos 2 Finished
   // Pos 2 Finished
   #O_Pos2Finished := #I_Pos2Begin AND #I_Pos2;
END_REGION

REGION Network 27: **** 5.2 - Equations - Flow Equations **** Pos 3 Finished
   // Pos 3 Finished
   #O_Pos3Finished := #I_Pos3Begin AND #I_Pos3;
END_REGION

REGION Network 28: **** 8 - Outputs **** Interlock Alarm Set
   // Interlock Alarm Set
   #O_IntlkSetAlm := #IntlkSetAlm;
END_REGION

REGION Network 29: **** 8 - Outputs **** Interlock Alarm Res
   // Interlock Alarm Res
   #O_IntlkResAlm := #IntlkResAlm;
END_REGION

REGION Network 30: **** 8 - Outputs **** Command High set
   // Command set
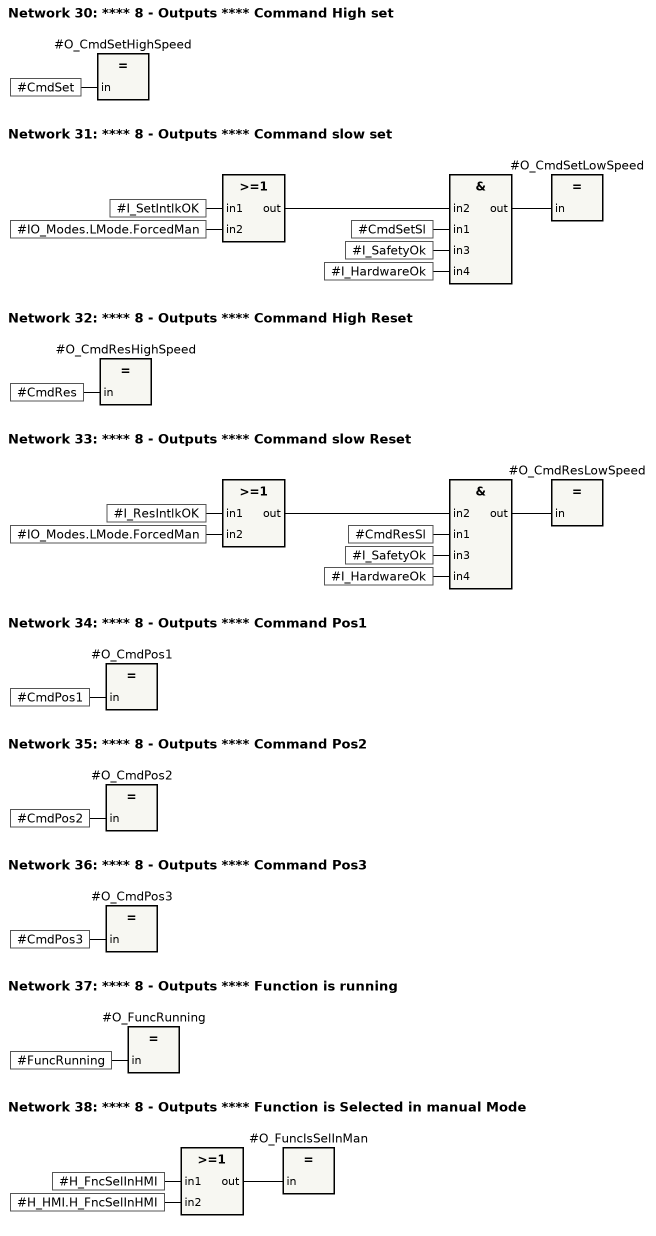
   #O_CmdSetHighSpeed := #CmdSet;
END_REGION

REGION Network 31: **** 8 - Outputs **** Command slow set
   // Command slow set
   #O_CmdSetLowSpeed := (#I_SetIntlkOK OR #IO_Modes.LMode.ForcedMan) AND #CmdSetSl AND #I_SafetyOk AND #I_HardwareOk;
END_REGION

REGION Network 32: **** 8 - Outputs **** Command High Reset
   // Command Reset
   #O_CmdResHighSpeed := #CmdRes;
END_REGION

REGION Network 33: **** 8 - Outputs **** Command slow Reset
   // Command slow Reset
   #O_CmdResLowSpeed := (#I_ResIntlkOK OR #IO_Modes.LMode.ForcedMan) AND #CmdResSl AND #I_SafetyOk AND #I_HardwareOk;
END_REGION

REGION Network 34: **** 8 - Outputs **** Command Pos1
   // Command Pos1
   #O_CmdPos1 := #CmdPos1;
END_REGION

REGION Network 35: **** 8 - Outputs **** Command Pos2
   // Command Pos2
   #O_CmdPos2 := #CmdPos2;
END_REGION

REGION Network 36: **** 8 - Outputs **** Command Pos3
   // Command Pos3
   #O_CmdPos3 := #CmdPos3;
END_REGION

REGION Network 37: **** 8 - Outputs **** Function is running
   // Function is running
   #O_FuncRunning := #FuncRunning;
END_REGION

REGION Network 38: **** 8 - Outputs **** Function is Selected in manual Mode
   // Function is Selected in manual Mode
   #O_FuncIsSelInMan := #H_FncSelInHMI OR #H_HMI.H_FncSelInHMI;
END_REGION

REGION Network 39: **** 8 - Outputs **** LED - Indication
   // LED - Indication
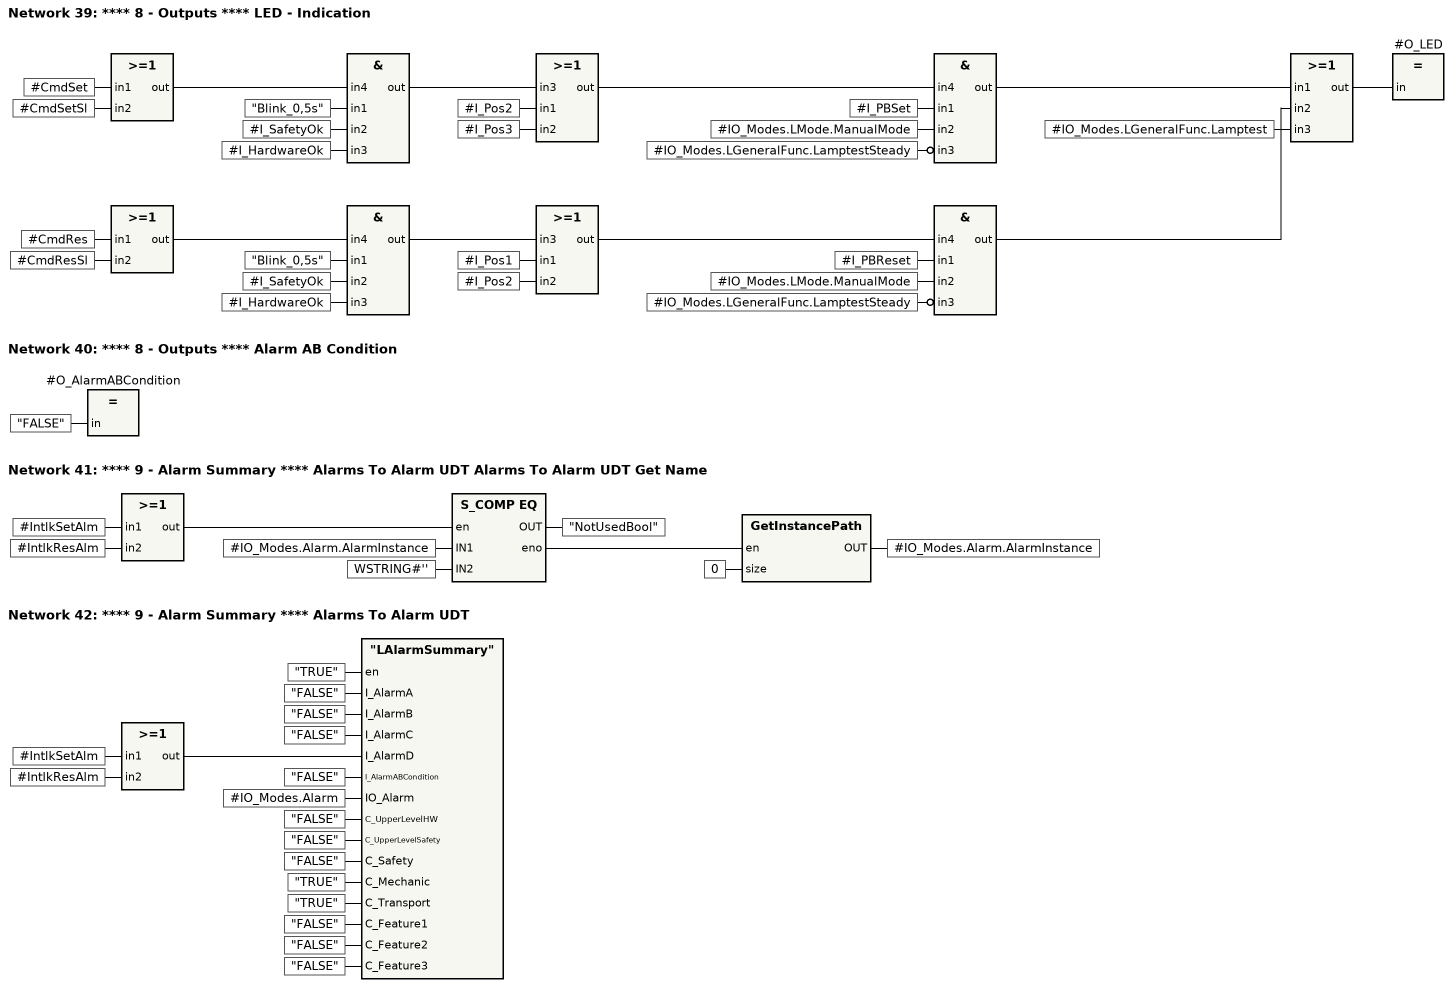
   #O_LED := ((((#CmdSet OR #CmdSetSl) AND "Blink_0,5s" AND #I_SafetyOk AND #I_HardwareOk) OR #I_Pos2 OR #I_Pos3) AND #I_PBSet AND #IO_Modes.LMode.ManualMode AND NOT #IO_Modes.LGeneralFunc.LamptestSteady) OR ((((#CmdRes OR #CmdResSl) AND "Blink_0,5s" AND #I_SafetyOk AND #I_HardwareOk) OR #I_Pos1 OR #I_Pos2) AND #I_PBReset AND #IO_Modes.LMode.ManualMode AND NOT #IO_Modes.LGeneralFunc.LamptestSteady) OR #IO_Modes.LGeneralFunc.Lamptest;
END_REGION

REGION Network 40: **** 8 - Outputs **** Alarm AB Condition
   // Alarm AB Condition
   #O_AlarmABCondition := "FALSE";
END_REGION

REGION Network 41: **** 9 - Alarm Summary **** Alarms To Alarm UDT Alarms To Alarm UDT Get Name
   // Alarms To Alarm UDT Alarms To Alarm UDT Get Name
   S_COMP(EN := #IntlkSetAlm OR #IntlkResAlm,
          IN1 := #IO_Modes.Alarm.AlarmInstance,
          IN2 := WSTRING#'',
          OUT => "NotUsedBool",
          ENO => #_w1);
   IF #_w1 THEN GetInstancePath(size := 0, OUT => #IO_Modes.Alarm.AlarmInstance); END_IF;
END_REGION

REGION Network 42: **** 9 - Alarm Summary **** Alarms To Alarm UDT
   // Alarms To Alarm UDT
   IF "TRUE" THEN
       "LAlarmSummary"(I_AlarmA := "FALSE",
                       I_AlarmB := "FALSE",
                       I_AlarmC := "FALSE",
                       I_AlarmD := #IntlkSetAlm OR #IntlkResAlm,
                       I_AlarmABCondition := "FALSE",
                       IO_Alarm := #IO_Modes.Alarm,
                       C_UpperLevelHW := "FALSE",
                       C_UpperLevelSafety := "FALSE",
                       C_Safety := "FALSE",
                       C_Mechanic := "TRUE",
                       C_Transport := "TRUE",
                       C_Feature1 := "FALSE",
                       C_Feature2 := "FALSE",
                       C_Feature3 := "FALSE");
   END_IF;
END_REGION
END_FUNCTION_BLOCK

FUNCTION_BLOCK "LPNIODiagS7-1500"   // FB2205, SCL
TITLE = PN_IO for HMI
{ S7_Optimized_Access := 'TRUE' }
AUTHOR : VCC
FAMILY : PNIODiag
VERSION : 0.0.0.0
// apette18,PADA
// stored: AutoNumber false, IsIECCheckEnabled true, IsRetainMemResEnabled true, MemoryReserve 200, RetainMemoryReserve 0, SetENOAutomatically True, UDAEnableTagReadback false
   VAR_INPUT
      I_HWIOSYSTEM { ExternalAccessible := 'False'; ExternalVisible := 'False'; ExternalWritable := 'False'} : HW_IOSYSTEM;   // HW ID ProfiNet System
      I_PLCIOSYSTEM { ExternalAccessible := 'False'; ExternalVisible := 'False'; ExternalWritable := 'False'} : HW_INTERFACE;   // HW ID ProfiNet System PLC Port 1
      I_LastDeviceNumber { ExternalAccessible := 'False'; ExternalVisible := 'False'; ExternalWritable := 'False'} : Int;   // Last Device of ProfiNet System
   END_VAR
   VAR_OUTPUT
      O_LastDeviceNumber { ExternalAccessible := 'False'; ExternalVisible := 'False'; ExternalWritable := 'False'} : Int;   // Last Device of ProfiNet System
   END_VAR
   VAR_IN_OUT
      IO_DeviceExist : Array[0..255] of Bool;   // IO devices exist
      IO_HWIdentifier : Array[0..255] of UInt;   // HW Device
      IO_PNIODIAG_Global : "H_PNIODiagS7-1500";
   END_VAR
   VAR
      PNDeviceConfigured { ExternalAccessible := 'False'; ExternalVisible := 'False'; ExternalWritable := 'False'} : Array[0..255] of Bool;   // IO devices are configured
      PNDeviceExist { ExternalAccessible := 'False'; ExternalVisible := 'False'; ExternalWritable := 'False'} : Array[0..255] of Bool;   // IO devices are faulty
      PNDeviceFaulty { ExternalAccessible := 'False'; ExternalVisible := 'False'; ExternalWritable := 'False'} : Array[0..255] of Bool;   // IO devices are faulty
      PNDeviceDisabled { ExternalAccessible := 'False'; ExternalVisible := 'False'; ExternalWritable := 'False'} : Array[0..255] of Bool;   // IO devices are disabled
      PNDeviceServiceReq { ExternalAccessible := 'False'; ExternalVisible := 'False'; ExternalWritable := 'False'} : Array[0..255] of Bool;   // IO devices for which a problem has occurred
      Edge { ExternalAccessible := 'False'; ExternalVisible := 'False'; ExternalWritable := 'False'} : Bool;   // Temp
      GeoAdress { ExternalAccessible := 'False'; ExternalVisible := 'False'; ExternalWritable := 'False'; S7_SetPoint := 'True'} : GEOADDR;   // Int Function
      _ReadIP { ExternalAccessible := 'False'; ExternalVisible := 'False'; ExternalWritable := 'False'; S7_SetPoint := 'True'} : "LPNIODiagReadIPS7-1500";   // FB
      TimerResetPNStatus { ExternalAccessible := 'False'; ExternalVisible := 'False'; ExternalWritable := 'False'; S7_SetPoint := 'True'} : TP_TIME;   // Timer
   END_VAR
   VAR_TEMP
      No1 : Int;   // Temp
      ReturnMode1 : Int;   // Temp
      ReturnMode2 : Int;   // Temp
      ReturnMode3 : Int;   // Temp
      ReturnMode4 : Int;   // Temp
      ReturnMode5 : Int;   // Temp
      ReturnGeo : Int;   // Temp
      ReturnActPNIO : Int;   // Temp
   END_VAR
   // GeoAdress.HWTYPE := 2;
   // GeoAdress.AREA := 1;
   // GeoAdress.IOSYSTEM := 100;
BEGIN

   //**** 1 - Inputs **** Activate Scan
   IF "TRUE" THEN
       #ReturnMode1 := DeviceStates(LADDR := #I_HWIOSYSTEM, MODE := 1, STATE := #PNDeviceConfigured); //1:IO devices are configured
       #ReturnMode2 := DeviceStates(LADDR := #I_HWIOSYSTEM, MODE := 2, STATE := #PNDeviceFaulty); //2: IO devices are faulty   
       #ReturnMode3 := DeviceStates(LADDR := #I_HWIOSYSTEM, MODE := 3, STATE := #PNDeviceDisabled); //3: IO devices are disabled
       #ReturnMode4 := DeviceStates(LADDR := #I_HWIOSYSTEM, MODE := 4, STATE := #PNDeviceExist); //4: IO devices exist
       #ReturnMode5 := DeviceStates(LADDR := #I_HWIOSYSTEM, MODE := 5, STATE := #PNDeviceServiceReq); //5: IO devices for which a problem has occurred    
   END_IF;

   //**** 2.2 - Alarms - Alarm Generation **** Reset Alarm and Warning
   #IO_PNIODIAG_Global.GlobStat_DeviceFaulty := FALSE;
   #IO_PNIODIAG_Global.GlobStat_DeviceDisabled := FALSE;
   #IO_PNIODIAG_Global.GlobStat_DeviceServiceReq := FALSE;

   //**** 4.4 - Machine status - Calculated  **** Set Status color on the HMI
   FOR #No1 := 1 TO #I_LastDeviceNumber DO
       IF #PNDeviceConfigured[#No1] THEN

           //Get HW_DEVICE number from all PN devices that are aviable on the PROFINET
           #GeoAdress.AREA := 1;
           #GeoAdress.HWTYPE := 2;
           #GeoAdress.STATION := INT_TO_UINT(#No1);
           #ReturnGeo := GEO2LOG(GEOADDR := #GeoAdress, LADDR => #IO_HWIdentifier[#No1]);

           //Check If IO Devices Are Faulty
           IF #PNDeviceFaulty[#No1] THEN
               #IO_PNIODIAG_Global.DeviceColor[#No1]:= 1; //red
               #IO_PNIODIAG_Global.DeviceFaulty[#No1] := True;
               #IO_PNIODIAG_Global.DeviceDisabled[#No1] := False;
               #IO_PNIODIAG_Global.DeviceServiceReq[#No1] := False;
               #IO_PNIODIAG_Global.GlobStat_DeviceFaulty := True;
               #IO_PNIODIAG_Global.GlobStat_DeviceDisabled := False;
               #IO_PNIODIAG_Global.GlobStat_DeviceServiceReq := False;

               //Check If  Maintenance Demand Or Service Request Is Active   
           ELSIF #PNDeviceServiceReq[#No1] = TRUE THEN
               #IO_PNIODIAG_Global.DeviceColor[#No1] := 4; //yellow
               #IO_PNIODIAG_Global.DeviceServiceReq[#No1] := True;
               #IO_PNIODIAG_Global.GlobStat_DeviceServiceReq := True;

               //Check if IO Devices Are disabled
           ELSIF #PNDeviceDisabled[#No1] = TRUE THEN
               #IO_PNIODIAG_Global.DeviceColor[#No1] := 2; //blue
               #IO_PNIODIAG_Global.DeviceDisabled[#No1] := True;
               #IO_PNIODIAG_Global.DeviceFaulty[#No1] := False;
               #IO_PNIODIAG_Global.GlobStat_DeviceFaulty := False;
               #IO_PNIODIAG_Global.GlobStat_DeviceDisabled := True;

               //Check If IO Devices Are Existing Without Error/Fault
           ELSIF #PNDeviceExist[#No1] = TRUE THEN
               #IO_PNIODIAG_Global.DeviceColor[#No1] := 3; //green
           END_IF;
       END_IF;
   END_FOR;


   //**** 4.4 - Machine status - Calculated  **** Get IP Address of PLC
   #_ReadIP(I_ReqIN := "TRUE",
            I_HWID := #I_PLCIOSYSTEM);


   //**** 4.4 - Machine status - Calculated  **** Reset the status from the HMI
   IF #IO_PNIODIAG_Global.HMICmd_ResetPNStatus AND NOT #Edge THEN
       #Edge := TRUE;
       FOR #No1 := 1 TO #I_LastDeviceNumber DO
           #IO_PNIODIAG_Global.DeviceFaulty[#No1] := FALSE;
           #IO_PNIODIAG_Global.DeviceDisabled[#No1] := FALSE;
           #IO_PNIODIAG_Global.DeviceServiceReq[#No1] := FALSE;
           #IO_PNIODIAG_Global.GlobStat_DeviceFaulty := FALSE;
           #IO_PNIODIAG_Global.GlobStat_DeviceDisabled := FALSE;
           #IO_PNIODIAG_Global.GlobStat_DeviceServiceReq := FALSE;
       END_FOR;
       #Edge := FALSE;
   END_IF;
   #TimerResetPNStatus(IN:=#IO_PNIODIAG_Global.HMICmd_ResetPNStatus,
                       PT:=T#500ms);
   //IF #TimerResetPNStatus.Q THEN
   //    #IO_PNIODIAG_Global.HMICmd_ResetPNStatus := False;
   //END_IF;


   //**** 4.4 - Machine status - Calculated  **** Activate or Deactivate PN Devices
   #ReturnActPNIO := D_ACT_DP(REQ := #IO_PNIODIAG_Global.HMICmd_ActivateDeactivate, MODE :=#IO_PNIODIAG_Global.PNMode, LADDR := #IO_HWIdentifier[ #IO_PNIODIAG_Global.DeviceNumber], BUSY => #IO_PNIODIAG_Global.ActivateDeactivateBusy);
   #IO_PNIODIAG_Global.HMICmd_ActivateDeactivate := FALSE;


   // **** 4.6 - Machine status - Indication ****  Animation
   #IO_PNIODIAG_Global.IPAddressPLC[0]:= #_ReadIP.O_IPParam.IPAddress[0];
   #IO_PNIODIAG_Global.IPAddressPLC[1] := #_ReadIP.O_IPParam.IPAddress[1];
   #IO_PNIODIAG_Global.IPAddressPLC[2] := #_ReadIP.O_IPParam.IPAddress[2];
   #IO_PNIODIAG_Global.IPAddressPLC[3] := #_ReadIP.O_IPParam.IPAddress[3];

   #IO_PNIODIAG_Global.DeviceExist := #PNDeviceExist;
   #IO_DeviceExist := #PNDeviceExist;

   #O_LastDeviceNumber := #I_LastDeviceNumber;
END_FUNCTION_BLOCK

FUNCTION_BLOCK "LPNIODiagReadIPS7-1500"   // FB2209, SCL
TITLE = LPNIODiagReadIPS7-1500
{ S7_Optimized_Access := 'TRUE' }
AUTHOR : VCC
FAMILY : PNIODiag
VERSION : 0.0.0.0
// apette18,PADA
// stored: AutoNumber false, IsIECCheckEnabled false, IsRetainMemResEnabled false, MemoryReserve 100, SetENOAutomatically False, UDAEnableTagReadback false
   VAR_INPUT
      I_ReqIN { ExternalAccessible := 'False'; ExternalVisible := 'False'; ExternalWritable := 'False'} : Bool;
      I_HWID { ExternalAccessible := 'False'; ExternalVisible := 'False'; ExternalWritable := 'False'} : UInt := 16#64;
   END_VAR
   VAR_OUTPUT
      O_IPParam { ExternalAccessible := 'False'; ExternalVisible := 'False'; ExternalWritable := 'False'} : Struct
         IPAddress { ExternalAccessible := 'False'; ExternalVisible := 'False'; ExternalWritable := 'False'} : Array[0..3] of USInt;
         SubnetMask { ExternalAccessible := 'False'; ExternalVisible := 'False'; ExternalWritable := 'False'} : Array[0..3] of USInt;
         StandardGateway { ExternalAccessible := 'False'; ExternalVisible := 'False'; ExternalWritable := 'False'} : Array[0..3] of USInt;
         MACAddress { ExternalAccessible := 'False'; ExternalVisible := 'False'; ExternalWritable := 'False'} : Array[0..5] of USInt;
         PNName { ExternalAccessible := 'False'; ExternalVisible := 'False'; ExternalWritable := 'False'} : String;
      END_STRUCT;
      O_Busy { ExternalAccessible := 'False'; ExternalVisible := 'False'; ExternalWritable := 'False'} : Bool;
      O_Valid { ExternalAccessible := 'False'; ExternalVisible := 'False'; ExternalWritable := 'False'} : Bool;
      O_Error { ExternalAccessible := 'False'; ExternalVisible := 'False'; ExternalWritable := 'False'} : Bool;
      O_Status { ExternalAccessible := 'False'; ExternalVisible := 'False'; ExternalWritable := 'False'} : DWord;
      O_LEN { ExternalAccessible := 'False'; ExternalVisible := 'False'; ExternalWritable := 'False'} : UInt;
   END_VAR
   VAR
      ReqFlag { ExternalAccessible := 'False'; ExternalVisible := 'False'; ExternalWritable := 'False'} : Bool;
      RDREC_Status { ExternalAccessible := 'False'; ExternalVisible := 'False'; ExternalWritable := 'False'} : DWord;
      RDREC_LEN { ExternalAccessible := 'False'; ExternalVisible := 'False'; ExternalWritable := 'False'} : UInt;
      RDREC_Valid { ExternalAccessible := 'False'; ExternalVisible := 'False'; ExternalWritable := 'False'} : Bool;
      RDREC_Busy { ExternalAccessible := 'False'; ExternalVisible := 'False'; ExternalWritable := 'False'} : Bool;
      RDREC_Error { ExternalAccessible := 'False'; ExternalVisible := 'False'; ExternalWritable := 'False'} : Bool;
      StatusSave { ExternalAccessible := 'False'; ExternalVisible := 'False'; ExternalWritable := 'False'} : DWord;
      PDInterfaceDataReal { ExternalAccessible := 'False'; ExternalVisible := 'False'; ExternalWritable := 'False'} : Struct
         BlockType { ExternalAccessible := 'False'; ExternalVisible := 'False'; ExternalWritable := 'False'} : UInt;
         BlockLength { ExternalAccessible := 'False'; ExternalVisible := 'False'; ExternalWritable := 'False'} : UInt;
         BlockVersionHigh { ExternalAccessible := 'False'; ExternalVisible := 'False'; ExternalWritable := 'False'} : USInt;
         BlockVersionLow { ExternalAccessible := 'False'; ExternalVisible := 'False'; ExternalWritable := 'False'} : USInt;
         Data { ExternalAccessible := 'False'; ExternalVisible := 'False'; ExternalWritable := 'False'} : Array[0..301] of Byte;
         OwnChassisID { ExternalAccessible := 'False'; ExternalVisible := 'False'; ExternalWritable := 'False'} : String;
      END_STRUCT;
      R_TRIG { ExternalAccessible := 'False'; ExternalVisible := 'False'; ExternalWritable := 'False'; S7_SetPoint := 'True'} : R_TRIG;
      RDREC { ExternalAccessible := 'False'; ExternalVisible := 'False'; ExternalWritable := 'False'; S7_SetPoint := 'True'} : RDREC;
   END_VAR
   VAR_TEMP
      IPParValStartAddress : USInt;
      LengthOwnChassisID : USInt;
   END_VAR
BEGIN
   (*
   =================================================================================================================
   This Block is used for reading the IP Address, Subnet Mask etc. of the PLC.
   =================================================================================================================
   *)

   #R_TRIG(CLK:=#I_ReqIN,
           Q=>#ReqFlag);

   #RDREC(REQ:=#ReqFlag,
          ID:=#I_HWID,
          INDEX:=w#16#8080,
          MLEN:=300,
          VALID=>#RDREC_Valid,
          BUSY=>#RDREC_Busy,
          ERROR=>#RDREC_Error,
          STATUS=>#RDREC_Status,
          LEN=>#RDREC_LEN,
          RECORD:=#PDInterfaceDataReal);

   IF #RDREC_Valid THEN

       // Get PN-interface Name. String starts at an odd address within the array
       Chars_TO_Strg(Chars := #PDInterfaceDataReal.Data, pChars := 1, Cnt := #PDInterfaceDataReal.Data[0], Strg => #O_IPParam.PNName );

       // Calculate start address of IP-address data. Blockdata is padded to make it Unsigned32 aligned!      
       #IPParValStartAddress := #PDInterfaceDataReal.Data[0]  + (4 - ((#PDInterfaceDataReal.Data[0] + 2) MOD 4));

       // Copy MAC-Address data
       #O_IPParam.MACAddress[0] := #PDInterfaceDataReal.Data[#IPParValStartAddress + 0];
       #O_IPParam.MACAddress[1] := #PDInterfaceDataReal.Data[#IPParValStartAddress + 1];
       #O_IPParam.MACAddress[2] := #PDInterfaceDataReal.Data[#IPParValStartAddress + 2];
       #O_IPParam.MACAddress[3] := #PDInterfaceDataReal.Data[#IPParValStartAddress + 3];
       #O_IPParam.MACAddress[4] := #PDInterfaceDataReal.Data[#IPParValStartAddress + 4];
       #O_IPParam.MACAddress[5] := #PDInterfaceDataReal.Data[#IPParValStartAddress + 5];

        // Copy IP-Address data
       #O_IPParam.IPAddress[0] := #PDInterfaceDataReal.Data[#IPParValStartAddress + 8 + 0];
       #O_IPParam.IPAddress[1] := #PDInterfaceDataReal.Data[#IPParValStartAddress + 8 + 1];
       #O_IPParam.IPAddress[2] := #PDInterfaceDataReal.Data[#IPParValStartAddress + 8 + 2];
       #O_IPParam.IPAddress[3] := #PDInterfaceDataReal.Data[#IPParValStartAddress + 8 + 3];

       // Copy Subnetmask data
       #O_IPParam.SubnetMask[0] := #PDInterfaceDataReal.Data[#IPParValStartAddress + 12 + 0];
       #O_IPParam.SubnetMask[1] := #PDInterfaceDataReal.Data[#IPParValStartAddress + 12 + 1];
       #O_IPParam.SubnetMask[2] := #PDInterfaceDataReal.Data[#IPParValStartAddress + 12 + 2];
       #O_IPParam.SubnetMask[3] := #PDInterfaceDataReal.Data[#IPParValStartAddress + 12 + 3];

     // Copy Standard Gateway data
       #O_IPParam.StandardGateway[0] := #PDInterfaceDataReal.Data[#IPParValStartAddress + 16 + 0];
       #O_IPParam.StandardGateway[1] := #PDInterfaceDataReal.Data[#IPParValStartAddress + 16 + 1];
       #O_IPParam.StandardGateway[2] := #PDInterfaceDataReal.Data[#IPParValStartAddress + 16 + 2];
       #O_IPParam.StandardGateway[3] := #PDInterfaceDataReal.Data[#IPParValStartAddress + 16 + 3];

   END_IF;

   IF #RDREC_Error THEN
     // Statement section IF
     #StatusSave:=#RDREC_Status;
     #O_LEN:=0;
   ELSE
     #StatusSave:=0;
     #O_LEN:=#RDREC_LEN;
   END_IF;


   IF  #RDREC_Error OR #RDREC_Valid THEN
     // Statement section IF
     #ReqFlag:=FALSE;
   END_IF;

   #O_Status:=#StatusSave;
   #O_Valid:=#RDREC_Valid;
   #O_Busy:=#RDREC_Busy;
   #O_Error:=#RDREC_Error;
END_FUNCTION_BLOCK

FUNCTION_BLOCK "LVDComMasterS7-1500"   // FB2210, FBD
TITLE = LVDComMasterPNS7-1500
{ S7_Optimized_Access := 'FALSE' }
AUTHOR : VCC
FAMILY : Communic
VERSION : 0.1
// =============================================================================
// This module Is Used To Read & Send Data With VDCom Protocol
// =============================================================================
// stored: AutoNumber false, IsIECCheckEnabled false, SetENOAutomatically False, UDAEnableTagReadback false
   VAR_INPUT
      I_VDCommRecvDB { ExternalAccessible := 'False'; ExternalVisible := 'False'; ExternalWritable := 'False'} : DB_ANY;   // VD Communication Master DB
      I_VDCommSendDB { ExternalAccessible := 'False'; ExternalVisible := 'False'; ExternalWritable := 'False'} : DB_ANY;   // VD Communication Master DB
   END_VAR
   VAR_OUTPUT
      O_AlarmA { ExternalAccessible := 'False'; ExternalVisible := 'False'; ExternalWritable := 'False'} : Bool;   // Alarm A
      O_AlarmB { ExternalAccessible := 'False'; ExternalVisible := 'False'; ExternalWritable := 'False'} : Bool;   // Alarm B
      O_AlarmC { ExternalAccessible := 'False'; ExternalVisible := 'False'; ExternalWritable := 'False'} : Bool;   // Alarm C
      O_AlarmD { ExternalAccessible := 'False'; ExternalVisible := 'False'; ExternalWritable := 'False'} : Bool;   // Alarm D
      H_AlarmWord { ExternalAccessible := 'False'; ExternalVisible := 'False'; ExternalWritable := 'False'} : DWord;   // HMI Animation
   END_VAR
   VAR_IN_OUT
      IO_Alarm : "Alarm";   // Alarm
      IO_VD : "VDComm";
      IO_ConnectionSetting : Variant;   // Software Connection Settings
      "H_VDComMasterPNS7-1500" : "H_VDComMasterPNS7-1500";   // Animation
   END_VAR
   VAR DB_SPECIFIC
      AD_SendTimeOut { ExternalAccessible := 'False'; ExternalVisible := 'False'; ExternalWritable := 'False'} : Bool;   // Communication Error Send Condition Active Too Long / Kommunikationsfel Sändvillkor Aktivt För Länge
      AD_VersionError { ExternalAccessible := 'False'; ExternalVisible := 'False'; ExternalWritable := 'False'} : Bool;   // Wrong Version Number / Fel Versionsnummer
      AD_ConnError { ExternalAccessible := 'False'; ExternalVisible := 'False'; ExternalWritable := 'False'} : Bool;   // Communication Error Connecting Or Disconnecting / Kommunikationsfel Uppkoppling Eller Nerkoppling
      AD_TCONConnected { ExternalAccessible := 'False'; ExternalVisible := 'False'; ExternalWritable := 'False'} : Bool;   // Not Connected / Ej Uppkopplad
      AD_TSENDError { ExternalAccessible := 'False'; ExternalVisible := 'False'; ExternalWritable := 'False'} : Bool;   // Error Transmission / Fel Sändning
      AD_TRECVError { ExternalAccessible := 'False'; ExternalVisible := 'False'; ExternalWritable := 'False'} : Bool;   // Error Receiving / Fel Mottagning
      AD_NoAckReceived { ExternalAccessible := 'False'; ExternalVisible := 'False'; ExternalWritable := 'False'} : Bool;   // Error On Ack Message / Fel Vid Ack Meddelande
      AD_SequenceNumberNok { ExternalAccessible := 'False'; ExternalVisible := 'False'; ExternalWritable := 'False'} : Bool;   // Incorrect Sequence Number / Felaktigt Sekvensnummer
      AD_TimeoutApplMsgMem { ExternalAccessible := 'False'; ExternalVisible := 'False'; ExternalWritable := 'False'} : Bool;   // Timeout Message To Subsystem / Timeout Meddelande Till Subsystem
      HMIManual { ExternalAccessible := 'False'; ExternalVisible := 'False'; ExternalWritable := 'False'} : Bool;   // Connect or disconnect manual via HMI
      HMIResetAndInit { ExternalAccessible := 'False'; ExternalVisible := 'False'; ExternalWritable := 'False'} : Bool;   // Reset Alarms from HMI
      HMIConnect { ExternalAccessible := 'False'; ExternalVisible := 'False'; ExternalWritable := 'False'} : Bool;   // Connect from HMI
      HMIDisConnect { ExternalAccessible := 'False'; ExternalVisible := 'False'; ExternalWritable := 'False'} : Bool;   // DisConnect from HMI
      Manual { ExternalAccessible := 'False'; ExternalVisible := 'False'; ExternalWritable := 'False'} : Bool;   // Connect or disconnect manual via HMI
      SendActive { ExternalAccessible := 'False'; ExternalVisible := 'False'; ExternalWritable := 'False'} : Bool;   // Sending is Active
      NdrDelayed { ExternalAccessible := 'False'; ExternalVisible := 'False'; ExternalWritable := 'False'} : Bool;   // Time required to elapse before to send acknowledge
      KeepAliveReq { ExternalAccessible := 'False'; ExternalVisible := 'False'; ExternalWritable := 'False'} : Bool;   // Request to send keep alive message
      AckRcvd { ExternalAccessible := 'False'; ExternalVisible := 'False'; ExternalWritable := 'False'} : Bool;   // Acknowledge Received
      SeqNbrOk { ExternalAccessible := 'False'; ExternalVisible := 'False'; ExternalWritable := 'False'} : Bool;   // Sequence number in received message is the same as sended
      AckOk { ExternalAccessible := 'False'; ExternalVisible := 'False'; ExternalWritable := 'False'} : Bool;   // Received acknowledge message ok
      AckNok { ExternalAccessible := 'False'; ExternalVisible := 'False'; ExternalWritable := 'False'} : Bool;   // Received acknowledge message not ok
      NewMessage { ExternalAccessible := 'False'; ExternalVisible := 'False'; ExternalWritable := 'False'} : Bool;   // New Data Message has been received
      SendInactive { ExternalAccessible := 'False'; ExternalVisible := 'False'; ExternalWritable := 'False'} : Bool;   // Sending inActive
      SendJobCompleted { ExternalAccessible := 'False'; ExternalVisible := 'False'; ExternalWritable := 'False'} : Bool;   // Status of the TSEND module: Job Completed no job active
      SendStartOfProc { ExternalAccessible := 'False'; ExternalVisible := 'False'; ExternalWritable := 'False'} : Bool;   // Status of TSEND: Start of Processing
      SendFollowOnCall { ExternalAccessible := 'False'; ExternalVisible := 'False'; ExternalWritable := 'False'} : Bool;   // Status of TSEND: Followon calls being processed
      SendNackMem { ExternalAccessible := 'False'; ExternalVisible := 'False'; ExternalWritable := 'False'} : Bool;   // Command to send Not acknowledge message
      SendNackPulse { ExternalAccessible := 'False'; ExternalVisible := 'False'; ExternalWritable := 'False'} : Bool;   // Pulse to send the Not Acknowledge message
      SendNackCmd { ExternalAccessible := 'False'; ExternalVisible := 'False'; ExternalWritable := 'False'} : Bool;   // Command to send a NOT Acknowledge message
      SendAckMem { ExternalAccessible := 'False'; ExternalVisible := 'False'; ExternalWritable := 'False'} : Bool;   // Command to send Acknowledge message
      SendAckPulse { ExternalAccessible := 'False'; ExternalVisible := 'False'; ExternalWritable := 'False'} : Bool;   // Pulse to send Acknowledge message
      SendAckCmd { ExternalAccessible := 'False'; ExternalVisible := 'False'; ExternalWritable := 'False'} : Bool;   // Command to send an Acknowledge message
      SendKeepAliveMem { ExternalAccessible := 'False'; ExternalVisible := 'False'; ExternalWritable := 'False'} : Bool;   // Command to send the keep alive signal
      SendKeepAlivePulse { ExternalAccessible := 'False'; ExternalVisible := 'False'; ExternalWritable := 'False'} : Bool;   // Pulse to send keep alive message
      SendKeepAliveCmd { ExternalAccessible := 'False'; ExternalVisible := 'False'; ExternalWritable := 'False'} : Bool;   // Command to Send Keep Alive message
      SendApplMsgMem { ExternalAccessible := 'False'; ExternalVisible := 'False'; ExternalWritable := 'False'} : Bool;   // Command to send apllication data
      SendApplMsgPulse { ExternalAccessible := 'False'; ExternalVisible := 'False'; ExternalWritable := 'False'} : Bool;   // Pulse created upon SendApplMsgCmd
      SendApplMsgCmd { ExternalAccessible := 'False'; ExternalVisible := 'False'; ExternalWritable := 'False'} : Bool;   // Command to send an Application message
      NewMsgNbr { ExternalAccessible := 'False'; ExternalVisible := 'False'; ExternalWritable := 'False'} : Bool;   // Message number of last received message
      NackIsLastSent { ExternalAccessible := 'False'; ExternalVisible := 'False'; ExternalWritable := 'False'} : Bool;   // Memorise that Nack was send
      DupplMsg { ExternalAccessible := 'False'; ExternalVisible := 'False'; ExternalWritable := 'False'} : Bool;   // When received msg number is the same as previous
      RecvLenOK { ExternalAccessible := 'False'; ExternalVisible := 'False'; ExternalWritable := 'False'} : Bool;   // If protocol Len and actual received msg are the same
      WaitForAck { ExternalAccessible := 'False'; ExternalVisible := 'False'; ExternalWritable := 'False'} : Bool;   // State waiting for acknowledge
      TimeOutTConn { ExternalAccessible := 'False'; ExternalVisible := 'False'; ExternalWritable := 'False'} : Bool;   // Time out on connecting or disconnecting
      TimeoutTCON { ExternalAccessible := 'False'; ExternalVisible := 'False'; ExternalWritable := 'False'} : Bool;   // Memory of connection time out
      TimeoutTDISCON { ExternalAccessible := 'False'; ExternalVisible := 'False'; ExternalWritable := 'False'} : Bool;   // Time out on disconnecting
      TimeoutApplMsg { ExternalAccessible := 'False'; ExternalVisible := 'False'; ExternalWritable := 'False'} : Bool;   // Time Out on apllication message, no ack received
      DisconnConn { ExternalAccessible := 'False'; ExternalVisible := 'False'; ExternalWritable := 'False'} : Bool;   // Time before connecting after disconnecting
      Edge { ExternalAccessible := 'False'; ExternalVisible := 'False'; ExternalWritable := 'False'} : Bool;   // Positive edge Detection for connected
      ResetAppliMsgCnt { ExternalAccessible := 'False'; ExternalVisible := 'False'; ExternalWritable := 'False'} : Bool;   // Reset the Application message counter
      ResetKeepAliveCnt { ExternalAccessible := 'False'; ExternalVisible := 'False'; ExternalWritable := 'False'} : Bool;   // Reset the keep alive counter
      ResetAckCmdCnt { ExternalAccessible := 'False'; ExternalVisible := 'False'; ExternalWritable := 'False'} : Bool;   // Reset the acknowledge counter
      ResetNackCmdCnt { ExternalAccessible := 'False'; ExternalVisible := 'False'; ExternalWritable := 'False'} : Bool;   // Reset the Nacknowledge counter
      ResetAckRcvCnt { ExternalAccessible := 'False'; ExternalVisible := 'False'; ExternalWritable := 'False'} : Bool;   // Reset the received Ack counter
      ResetDataMsgCnt { ExternalAccessible := 'False'; ExternalVisible := 'False'; ExternalWritable := 'False'} : Bool;   // Reset the received Data message counter
      ResetSeqNokCnt { ExternalAccessible := 'False'; ExternalVisible := 'False'; ExternalWritable := 'False'} : Bool;   // Reset the sequence nok counter
      ResetSendActive { ExternalAccessible := 'False'; ExternalVisible := 'False'; ExternalWritable := 'False'} : Bool;   // Reset Send Active due to time out
      SendDone { ExternalAccessible := 'False'; ExternalVisible := 'False'; ExternalWritable := 'False'} : Bool;   // Reset the Ndr counter on overrun
      DelayOpen { ExternalAccessible := 'False'; ExternalVisible := 'False'; ExternalWritable := 'False'} : Bool;   // Delay Start Connect
      DelayConn { ExternalAccessible := 'False'; ExternalVisible := 'False'; ExternalWritable := 'False'} : Bool;   // Delay Connected
      AlarmA { ExternalAccessible := 'False'; ExternalVisible := 'False'; ExternalWritable := 'False'} : Bool;   // Alarm A
      AlarmB { ExternalAccessible := 'False'; ExternalVisible := 'False'; ExternalWritable := 'False'} : Bool;   // Alarm B
      AlarmC { ExternalAccessible := 'False'; ExternalVisible := 'False'; ExternalWritable := 'False'} : Bool;   // Alarm C
      AlarmD { ExternalAccessible := 'False'; ExternalVisible := 'False'; ExternalWritable := 'False'} : Bool;   // Alarm D
      OldSubSystem { ExternalAccessible := 'False'; ExternalVisible := 'False'; ExternalWritable := 'False'} : Word;   // Memorise last received subsystem address
      OldRecMsgNbr { ExternalAccessible := 'False'; ExternalVisible := 'False'; ExternalWritable := 'False'} : Word := W#16#999;   // Memorise the last message number
      SendMsgNbr { ExternalAccessible := 'False'; ExternalVisible := 'False'; ExternalWritable := 'False'} : Word;   // Number is incremented for each msg and Reset to 1 when > 1000
      RecvLen { ExternalAccessible := 'False'; ExternalVisible := 'False'; ExternalWritable := 'False'} : Int;   // Memory of the received data length
      RecvDBNbr { ExternalAccessible := 'False'; ExternalVisible := 'False'; ExternalWritable := 'False'} : Int;   // Receive DB Number
      SendDBNbr { ExternalAccessible := 'False'; ExternalVisible := 'False'; ExternalWritable := 'False'} : Int;   // Send DB Number
      SendApplMsgCnt { ExternalAccessible := 'False'; ExternalVisible := 'False'; ExternalWritable := 'False'} : Int;   // Counting number of Application messages
      SendKeepAliveCnt { ExternalAccessible := 'False'; ExternalVisible := 'False'; ExternalWritable := 'False'} : Int;   // Counting number of keep alive messages
      SendAckCmdCnt { ExternalAccessible := 'False'; ExternalVisible := 'False'; ExternalWritable := 'False'} : Int;   // Counting the number of Ack messages
      SendNackCmdCnt { ExternalAccessible := 'False'; ExternalVisible := 'False'; ExternalWritable := 'False'} : Int;   // Counting the number of Nack messages
      RcvAckCnt { ExternalAccessible := 'False'; ExternalVisible := 'False'; ExternalWritable := 'False'} : Int;   // Counting the number of received Ack messages
      RcvDataMsgCnt { ExternalAccessible := 'False'; ExternalVisible := 'False'; ExternalWritable := 'False'} : Int;   // Counting the number of Data messages
      SeqNokCnt { ExternalAccessible := 'False'; ExternalVisible := 'False'; ExternalWritable := 'False'} : Int;   // Counter indicating the number of received sequence errors
      NdrCnt { ExternalAccessible := 'False'; ExternalVisible := 'False'; ExternalWritable := 'False'} : Int;   // Counter indicating the all received events
   END_VAR
   VAR
      TConVD { ExternalAccessible := 'False'; ExternalVisible := 'False'; ExternalWritable := 'False'; S7_SetPoint := 'True'} : TCON;   // Connect
      TDisConVD { ExternalAccessible := 'False'; ExternalVisible := 'False'; ExternalWritable := 'False'; S7_SetPoint := 'True'} : TDISCON;   // Disconnect
      TRcvVDData { ExternalAccessible := 'False'; ExternalVisible := 'False'; ExternalWritable := 'False'; S7_SetPoint := 'True'} : TRCV;   // Receive
      TSendVD { ExternalAccessible := 'False'; ExternalVisible := 'False'; ExternalWritable := 'False'; S7_SetPoint := 'True'} : TSEND;   // Send
   END_VAR
   VAR DB_SPECIFIC
      TCON { ExternalAccessible := 'False'; ExternalVisible := 'False'; ExternalWritable := 'False'} : Struct   // Structure
         Connecting { ExternalAccessible := 'False'; ExternalVisible := 'False'; ExternalWritable := 'False'} : Bool;
         Connected { ExternalAccessible := 'False'; ExternalVisible := 'False'; ExternalWritable := 'False'} : Bool;
         Done { ExternalAccessible := 'False'; ExternalVisible := 'False'; ExternalWritable := 'False'} : Bool;
         Busy { ExternalAccessible := 'False'; ExternalVisible := 'False'; ExternalWritable := 'False'} : Bool;
         Error { ExternalAccessible := 'False'; ExternalVisible := 'False'; ExternalWritable := 'False'} : Bool;
         Req { ExternalAccessible := 'False'; ExternalVisible := 'False'; ExternalWritable := 'False'} : Bool;
         Status { ExternalAccessible := 'False'; ExternalVisible := 'False'; ExternalWritable := 'False'} : Word;
         Status_Mem { ExternalAccessible := 'False'; ExternalVisible := 'False'; ExternalWritable := 'False'} : Word;
         Status_Int { ExternalAccessible := 'False'; ExternalVisible := 'False'; ExternalWritable := 'False'} : Int;
      END_STRUCT;
      TDISCON { ExternalAccessible := 'False'; ExternalVisible := 'False'; ExternalWritable := 'False'} : Struct   // Structure
         Disconnecting { ExternalAccessible := 'False'; ExternalVisible := 'False'; ExternalWritable := 'False'} : Bool;
         Done { ExternalAccessible := 'False'; ExternalVisible := 'False'; ExternalWritable := 'False'} : Bool;
         Busy { ExternalAccessible := 'False'; ExternalVisible := 'False'; ExternalWritable := 'False'} : Bool;
         Error { ExternalAccessible := 'False'; ExternalVisible := 'False'; ExternalWritable := 'False'} : Bool;
         Req { ExternalAccessible := 'False'; ExternalVisible := 'False'; ExternalWritable := 'False'} : Bool;
         Status { ExternalAccessible := 'False'; ExternalVisible := 'False'; ExternalWritable := 'False'} : Word;
         Status_Mem { ExternalAccessible := 'False'; ExternalVisible := 'False'; ExternalWritable := 'False'} : Word;
      END_STRUCT;
      TRECV { ExternalAccessible := 'False'; ExternalVisible := 'False'; ExternalWritable := 'False'} : Struct   // Structure
         Receiving { ExternalAccessible := 'False'; ExternalVisible := 'False'; ExternalWritable := 'False'} : Bool;
         Ndr { ExternalAccessible := 'False'; ExternalVisible := 'False'; ExternalWritable := 'False'} : Bool;
         Busy { ExternalAccessible := 'False'; ExternalVisible := 'False'; ExternalWritable := 'False'} : Bool;
         Error { ExternalAccessible := 'False'; ExternalVisible := 'False'; ExternalWritable := 'False'} : Bool;
         RcvConError { ExternalAccessible := 'False'; ExternalVisible := 'False'; ExternalWritable := 'False'} : Bool;
         Status { ExternalAccessible := 'False'; ExternalVisible := 'False'; ExternalWritable := 'False'} : Word;
         Status_Mem { ExternalAccessible := 'False'; ExternalVisible := 'False'; ExternalWritable := 'False'} : Word;
         Length { ExternalAccessible := 'False'; ExternalVisible := 'False'; ExternalWritable := 'False'} : UDInt;
      END_STRUCT;
      TSEND { ExternalAccessible := 'False'; ExternalVisible := 'False'; ExternalWritable := 'False'} : Struct   // Structure
         Sending { ExternalAccessible := 'False'; ExternalVisible := 'False'; ExternalWritable := 'False'} : Bool;
         Done { ExternalAccessible := 'False'; ExternalVisible := 'False'; ExternalWritable := 'False'} : Bool;
         Busy { ExternalAccessible := 'False'; ExternalVisible := 'False'; ExternalWritable := 'False'} : Bool;
         Error { ExternalAccessible := 'False'; ExternalVisible := 'False'; ExternalWritable := 'False'} : Bool;
         Status { ExternalAccessible := 'False'; ExternalVisible := 'False'; ExternalWritable := 'False'} : Word;
         Status_Mem { ExternalAccessible := 'False'; ExternalVisible := 'False'; ExternalWritable := 'False'} : Word;
      END_STRUCT;
      NackCmdCntr { ExternalAccessible := 'False'; ExternalVisible := 'False'; ExternalWritable := 'False'; S7_SetPoint := 'True'} : CTU_INT;   // Count number of NotAck messages send by PLC
      AckCmdCnt { ExternalAccessible := 'False'; ExternalVisible := 'False'; ExternalWritable := 'False'; S7_SetPoint := 'True'} : CTU_INT;   // Count number of Ack messages send by PLC
      KeepAliveCnt { ExternalAccessible := 'False'; ExternalVisible := 'False'; ExternalWritable := 'False'; S7_SetPoint := 'True'} : CTU_INT;   // Count number of Keep Alived Messages send by PLC
      AppliMsgCnt { ExternalAccessible := 'False'; ExternalVisible := 'False'; ExternalWritable := 'False'; S7_SetPoint := 'True'} : CTU_INT;   // Count number of Application messages send by PLC
      AckRvcCntr { ExternalAccessible := 'False'; ExternalVisible := 'False'; ExternalWritable := 'False'; S7_SetPoint := 'True'} : CTU_INT;   // Count number of Ack messages received
      DataMsgRcvCntr { ExternalAccessible := 'False'; ExternalVisible := 'False'; ExternalWritable := 'False'; S7_SetPoint := 'True'} : CTU_INT;   // Count number of data messages received
      SeqNumNok { ExternalAccessible := 'False'; ExternalVisible := 'False'; ExternalWritable := 'False'; S7_SetPoint := 'True'} : CTU_INT;   // counter to know the sequence number errors
      NdrPace { ExternalAccessible := 'False'; ExternalVisible := 'False'; ExternalWritable := 'False'; S7_SetPoint := 'True'} : TOF_TIME;   // Make sure that not too many messages are received at once
      TimeOutSending { ExternalAccessible := 'False'; ExternalVisible := 'False'; ExternalWritable := 'False'; S7_SetPoint := 'True'} : TON_TIME;   // TimeOut on Send operation
      TimeOutAckApplMsg { ExternalAccessible := 'False'; ExternalVisible := 'False'; ExternalWritable := 'False'; S7_SetPoint := 'True'} : TON_TIME;   // Timeout on reception of Ack on Application message
      TimeOutOnConnection { ExternalAccessible := 'False'; ExternalVisible := 'False'; ExternalWritable := 'False'; S7_SetPoint := 'True'} : TON_TIME;   // TimeOut on connecting
      KeepAliveFreq { ExternalAccessible := 'False'; ExternalVisible := 'False'; ExternalWritable := 'False'; S7_SetPoint := 'True'} : TON_TIME;   // Timer to timeout the keep alive messages
      DisconnectRequest { ExternalAccessible := 'False'; ExternalVisible := 'False'; ExternalWritable := 'False'; S7_SetPoint := 'True'} : TON_TIME;   // Request to disconnect after timeout
      WaitingForAck { ExternalAccessible := 'False'; ExternalVisible := 'False'; ExternalWritable := 'False'; S7_SetPoint := 'True'} : TON_TIME;   // Waiting for Ack to receive
      SubSystResponseTimeOut { ExternalAccessible := 'False'; ExternalVisible := 'False'; ExternalWritable := 'False'; S7_SetPoint := 'True'} : TON_TIME;   // TimeOut subsystem reply
      TimeOutSendActive { ExternalAccessible := 'False'; ExternalVisible := 'False'; ExternalWritable := 'False'; S7_SetPoint := 'True'} : TON_TIME;   // When SendActive is ON for too long
      DelayStartConnect { ExternalAccessible := 'False'; ExternalVisible := 'False'; ExternalWritable := 'False'; S7_SetPoint := 'True'} : TON_TIME;   // FB
      DelayConnected { ExternalAccessible := 'False'; ExternalVisible := 'False'; ExternalWritable := 'False'; S7_SetPoint := 'True'} : TON_TIME;   // FB
   END_VAR
   VAR
      _VDConManual { ExternalAccessible := 'False'; ExternalVisible := 'False'; ExternalWritable := 'False'; S7_SetPoint := 'True'} : "LToggle";   // FB
   END_VAR
   VAR DB_SPECIFIC
      ConnectionSettings { ExternalAccessible := 'False'; ExternalVisible := 'False'; ExternalWritable := 'False'; S7_SetPoint := 'True'} : TCON_Param;   // Structrure
   END_VAR
   VAR_TEMP
      PointerRecv : Any;   // Pointer to receive buffer
      PointerSend : Any;   // Pointer to Send Buffer
      PointerSendBuf : Any;   // Pointer to Send buffer
      OutBuf : Int;   // Integer to select the Send buffer
      UserMsgType : Bool;   // Message Type
      RecvTimeOut : Bool;   // Receive Time Out
      MsgLen : UDInt;   // Message length
      MessageLengthRecv : Int;   // Message Length receive
      TempIntStatus : Int;   // for type casting to integer
      TempInt : Int;   // for type casting to integer
      RecvDBNO : UInt;
      LengthDB : UDInt;
      TempBool : Array[1..16] of Bool;
      ConnectionSetting : Variant;
   END_VAR
   VAR_TEMP   // added for the SCL form of the ladder/FBD networks
      _w1 : Bool;
      _w2 : Bool;
   END_VAR
BEGIN

REGION Network 1: **** 1 - Inputs **** Extract the selection from HMI
   // Extract the selection from HMI
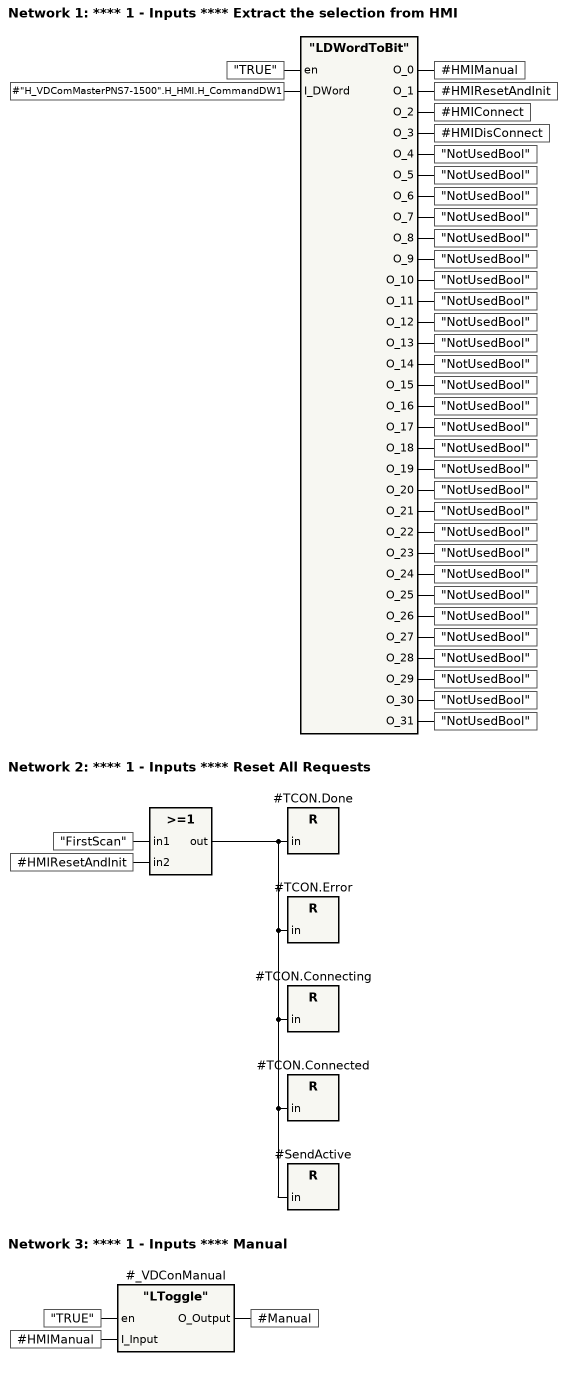
   IF "TRUE" THEN
       "LDWordToBit"(I_DWord := #"H_VDComMasterPNS7-1500".H_HMI.H_CommandDW1,
                     O_0 => #HMIManual,
                     O_1 => #HMIResetAndInit,
                     O_2 => #HMIConnect,
                     O_3 => #HMIDisConnect,
                     O_4 => "NotUsedBool",
                     O_5 => "NotUsedBool",
                     O_6 => "NotUsedBool",
                     O_7 => "NotUsedBool",
                     O_8 => "NotUsedBool",
                     O_9 => "NotUsedBool",
                     O_10 => "NotUsedBool",
                     O_11 => "NotUsedBool",
                     O_12 => "NotUsedBool",
                     O_13 => "NotUsedBool",
                     O_14 => "NotUsedBool",
                     O_15 => "NotUsedBool",
                     O_16 => "NotUsedBool",
                     O_17 => "NotUsedBool",
                     O_18 => "NotUsedBool",
                     O_19 => "NotUsedBool",
                     O_20 => "NotUsedBool",
                     O_21 => "NotUsedBool",
                     O_22 => "NotUsedBool",
                     O_23 => "NotUsedBool",
                     O_24 => "NotUsedBool",
                     O_25 => "NotUsedBool",
                     O_26 => "NotUsedBool",
                     O_27 => "NotUsedBool",
                     O_28 => "NotUsedBool",
                     O_29 => "NotUsedBool",
                     O_30 => "NotUsedBool",
                     O_31 => "NotUsedBool");
   END_IF;
END_REGION

REGION Network 2: **** 1 - Inputs **** Reset All Requests
   // Reset All Requests
   IF "FirstScan" OR #HMIResetAndInit THEN
       #TCON.Done := FALSE;
       #TCON.Error := FALSE;
       #TCON.Connecting := FALSE;
       #TCON.Connected := FALSE;
       #SendActive := FALSE;
   END_IF;
END_REGION

REGION Network 3: **** 1 - Inputs **** Manual
   // Manual
   IF "TRUE" THEN
       #_VDConManual(I_Input := #HMIManual, O_Output => #Manual);   // "LToggle"
   END_IF;
END_REGION

REGION Network 4: **** 1 - Inputs **** Reset Com Disconnect
   // Reset Com Disconnect
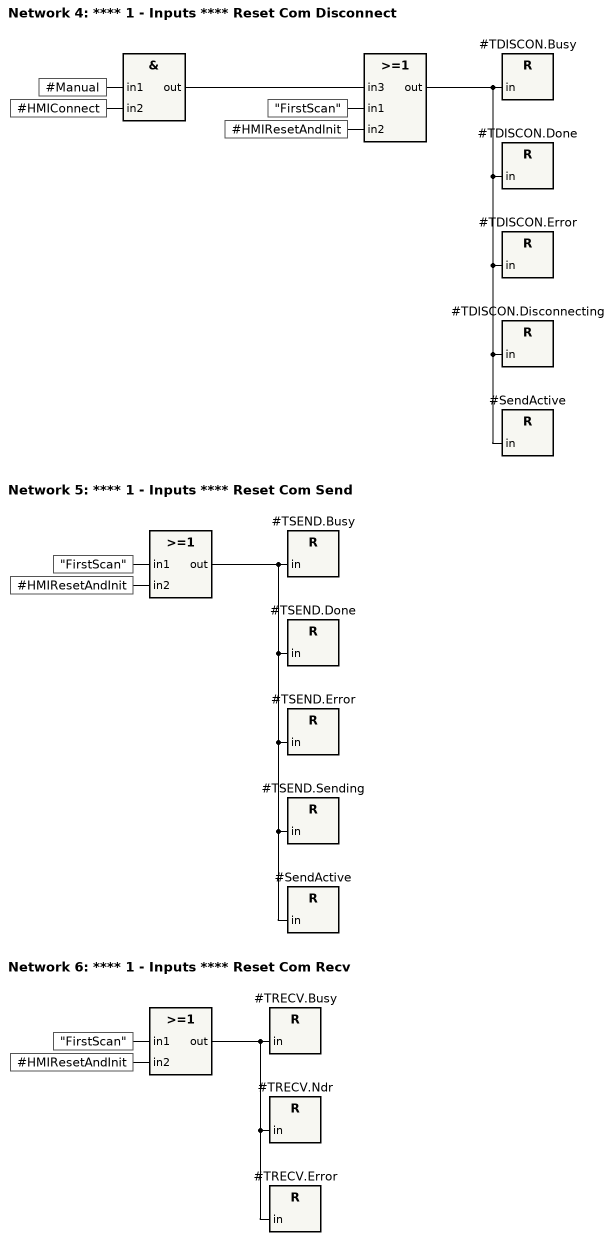
   IF (#Manual AND #HMIConnect) OR "FirstScan" OR #HMIResetAndInit THEN
       #TDISCON.Busy := FALSE;
       #TDISCON.Done := FALSE;
       #TDISCON.Error := FALSE;
       #TDISCON.Disconnecting := FALSE;
       #SendActive := FALSE;
   END_IF;
END_REGION

REGION Network 5: **** 1 - Inputs **** Reset Com Send
   // Reset com Send
   IF "FirstScan" OR #HMIResetAndInit THEN
       #TSEND.Busy := FALSE;
       #TSEND.Done := FALSE;
       #TSEND.Error := FALSE;
       #TSEND.Sending := FALSE;
       #SendActive := FALSE;
   END_IF;
END_REGION

REGION Network 6: **** 1 - Inputs **** Reset Com Recv
   // Reset Com Recv
   IF "FirstScan" OR #HMIResetAndInit THEN
       #TRECV.Busy := FALSE;
       #TRECV.Ndr := FALSE;
       #TRECV.Error := FALSE;
   END_IF;
END_REGION

REGION Network 7: **** 3.1 - Communication - Other Systems **** Reset Communications / **** 1 - Inputs **** Reset Communication
   // Reset Communications / Reset communication status words
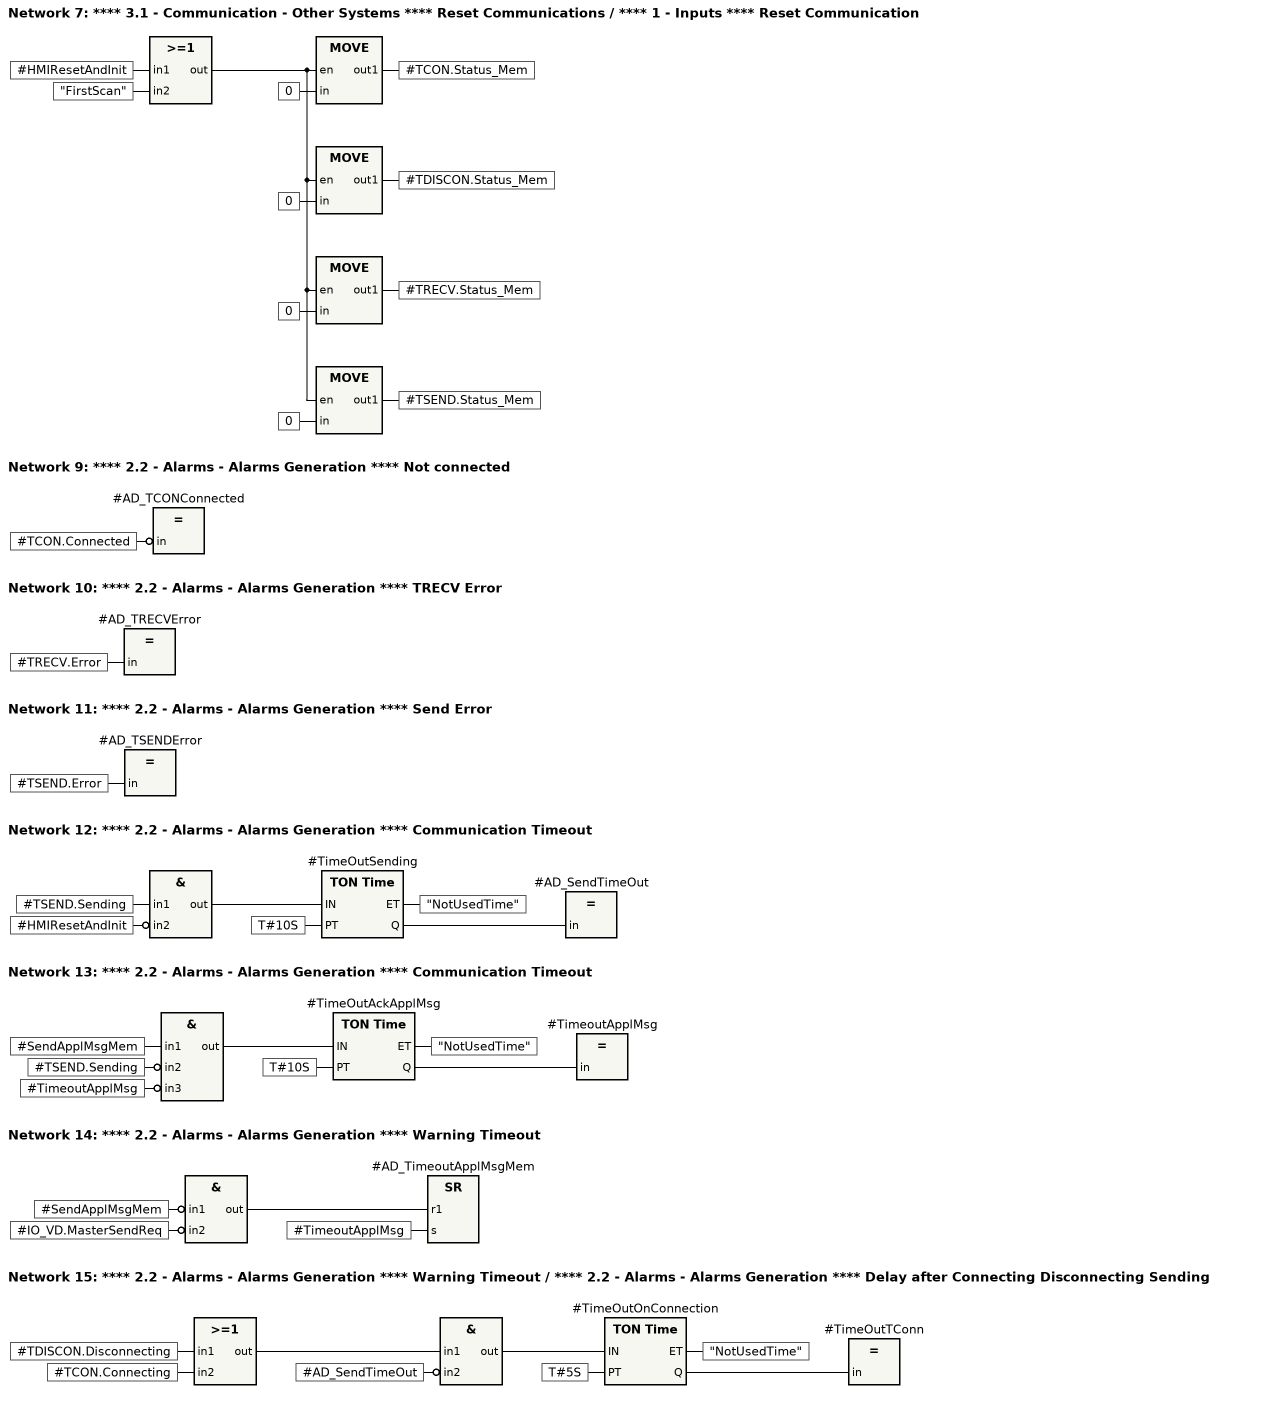
   IF #HMIResetAndInit OR "FirstScan" THEN
       #TCON.Status_Mem := 0;
       #TDISCON.Status_Mem := 0;
       #TRECV.Status_Mem := 0;
       #TSEND.Status_Mem := 0;
   END_IF;
END_REGION

NETWORK
TITLE = **** 1 - Inputs **** Load DB
// Load DB numbers to local variables from the Receive and Send DB
// Read DB Number Receive (VD Master System Receive DB)
      OPN   #I_VDCommRecvDB;
      L     DBNO;
      T     #RecvDBNbr;

// Read DB Number Send (VD Master System Send DB)
      OPN   #I_VDCommSendDB;
      L     DBNO;
      T     #SendDBNbr;



REGION Network 9: **** 2.2 - Alarms - Alarms Generation **** Not connected
   // Not connected
   #AD_TCONConnected := NOT #TCON.Connected;
END_REGION

REGION Network 10: **** 2.2 - Alarms - Alarms Generation **** TRECV Error
   // TRECV Error
   #AD_TRECVError := #TRECV.Error;
END_REGION

REGION Network 11: **** 2.2 - Alarms - Alarms Generation **** Send Error
   // Send Error
   #AD_TSENDError := #TSEND.Error;
END_REGION

REGION Network 12: **** 2.2 - Alarms - Alarms Generation **** Communication Timeout
   // Communication timeout while sending
   #TimeOutSending(IN := #TSEND.Sending AND NOT #HMIResetAndInit, PT := T#10S, ET => "NotUsedTime");   // TON
   #AD_SendTimeOut := #TimeOutSending.Q;
END_REGION

REGION Network 13: **** 2.2 - Alarms - Alarms Generation **** Communication Timeout
   // Communication timeout while Application message
   #TimeOutAckApplMsg(IN := #SendApplMsgMem AND NOT #TSEND.Sending AND NOT #TimeoutApplMsg,   // TON
                      PT := T#10S,
                      ET => "NotUsedTime");
   #TimeoutApplMsg := #TimeOutAckApplMsg.Q;
END_REGION

REGION Network 14: **** 2.2 - Alarms - Alarms Generation **** Warning Timeout
   // Warning Timeout Application message
   IF #TimeoutApplMsg THEN
       #AD_TimeoutApplMsgMem := TRUE;   // SR flip-flop
   END_IF;
   IF NOT #SendApplMsgMem AND NOT #IO_VD.MasterSendReq THEN #AD_TimeoutApplMsgMem := FALSE; END_IF;
END_REGION

REGION Network 15: **** 2.2 - Alarms - Alarms Generation **** Warning Timeout / **** 2.2 - Alarms - Alarms Generation **** Delay after Connecting Disconnecting Sending
   // Warning Timeout Application message / Delay after Connecting Disconnecting Sending
   #TimeOutOnConnection(IN := (#TDISCON.Disconnecting OR #TCON.Connecting) AND NOT #AD_SendTimeOut,   // TON
                        PT := T#5S,
                        ET => "NotUsedTime");
   #TimeOutTConn := #TimeOutOnConnection.Q;
END_REGION

REGION Network 16: **** 2.2 - Alarms - Alarms Generation **** Timeout Keep Alive
   // Timeout Keep Alive
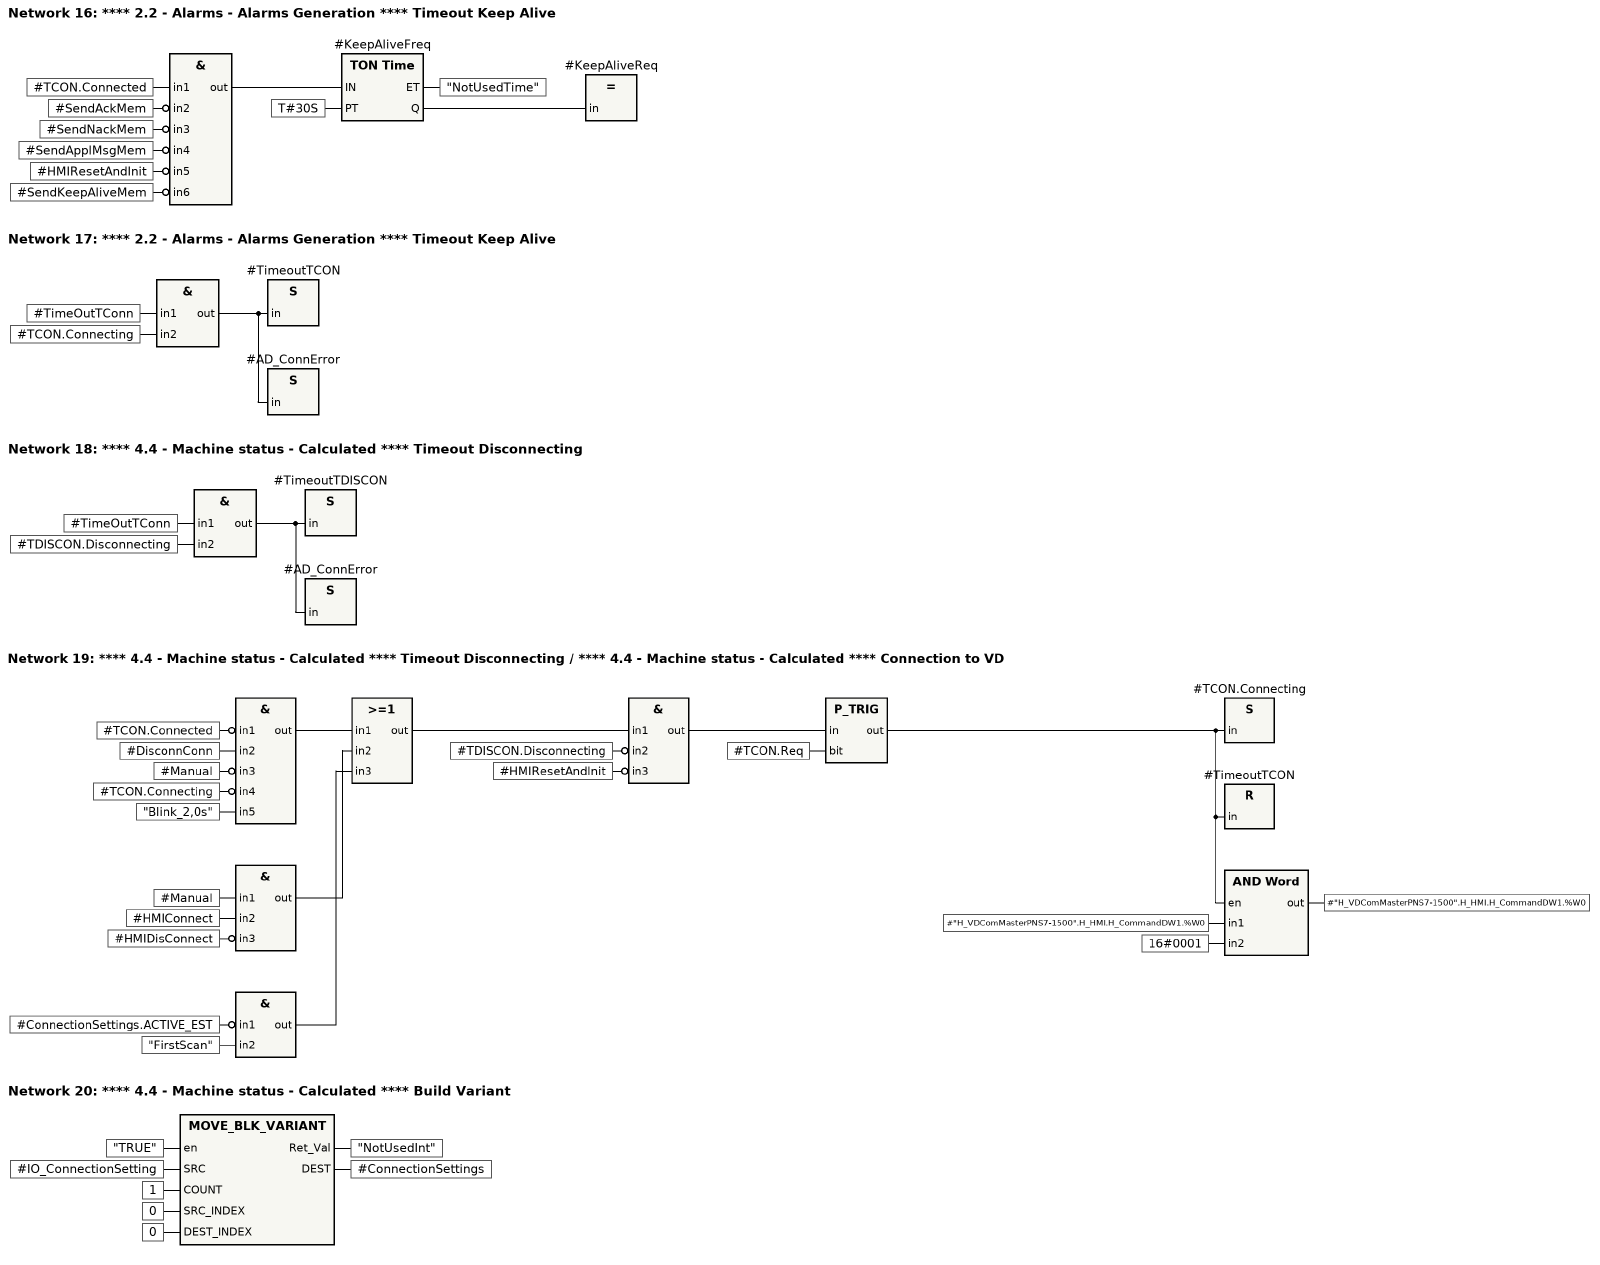
   #KeepAliveFreq(IN := #TCON.Connected AND NOT #SendAckMem AND NOT #SendNackMem AND NOT #SendApplMsgMem AND NOT #HMIResetAndInit AND NOT #SendKeepAliveMem,   // TON
                  PT := T#30S,
                  ET => "NotUsedTime");
   #KeepAliveReq := #KeepAliveFreq.Q;
END_REGION

REGION Network 17: **** 2.2 - Alarms - Alarms Generation **** Timeout Keep Alive
   // Timeout Keep Alive
   IF #TimeOutTConn AND #TCON.Connecting THEN
       #TimeoutTCON := TRUE;
       #AD_ConnError := TRUE;
   END_IF;
END_REGION

REGION Network 18: **** 4.4 - Machine status - Calculated **** Timeout Disconnecting
   // Timeout Disconnecting
   IF #TimeOutTConn AND #TDISCON.Disconnecting THEN
       #TimeoutTDISCON := TRUE;
       #AD_ConnError := TRUE;
   END_IF;
END_REGION

REGION Network 19: **** 4.4 - Machine status - Calculated **** Timeout Disconnecting / **** 4.4 - Machine status - Calculated **** Connection to VD
   // Timeout Disconnecting / Connection to the VD if NOT connecting AND NOT connecte PLC restart and passive connection establishment (to be ready to listen)
   #_w1 := ((NOT #TCON.Connected AND #DisconnConn AND NOT #Manual AND NOT #TCON.Connecting AND "Blink_2,0s") OR (#Manual AND #HMIConnect AND NOT #HMIDisConnect) OR (NOT #ConnectionSettings.ACTIVE_EST AND "FirstScan")) AND NOT #TDISCON.Disconnecting AND NOT #HMIResetAndInit;
   #_w2 := #_w1 AND NOT #TCON.Req;   // rising edge
   #TCON.Req := #_w1;
   IF #_w2 THEN
       #TCON.Connecting := TRUE;
       #TimeoutTCON := FALSE;
       #"H_VDComMasterPNS7-1500".H_HMI.H_CommandDW1.%W0 := #"H_VDComMasterPNS7-1500".H_HMI.H_CommandDW1.%W0 AND 16#0001;
   END_IF;
END_REGION

REGION Network 20: **** 4.4 - Machine status - Calculated **** Build Variant
   // Build Variant
   IF "TRUE" THEN
       "NotUsedInt" := MOVE_BLK_VARIANT(SRC := #IO_ConnectionSetting,
                               COUNT := 1,
                               SRC_INDEX := 0,
                               DEST_INDEX := 0,
                               DEST => #ConnectionSettings);
   END_IF;
END_REGION

REGION Network 21: **** 4.4 - Machine status - Calculated **** Build Variant / **** 4.4 - Machine status - Calculated **** Connection
   // Build Variant / Connection
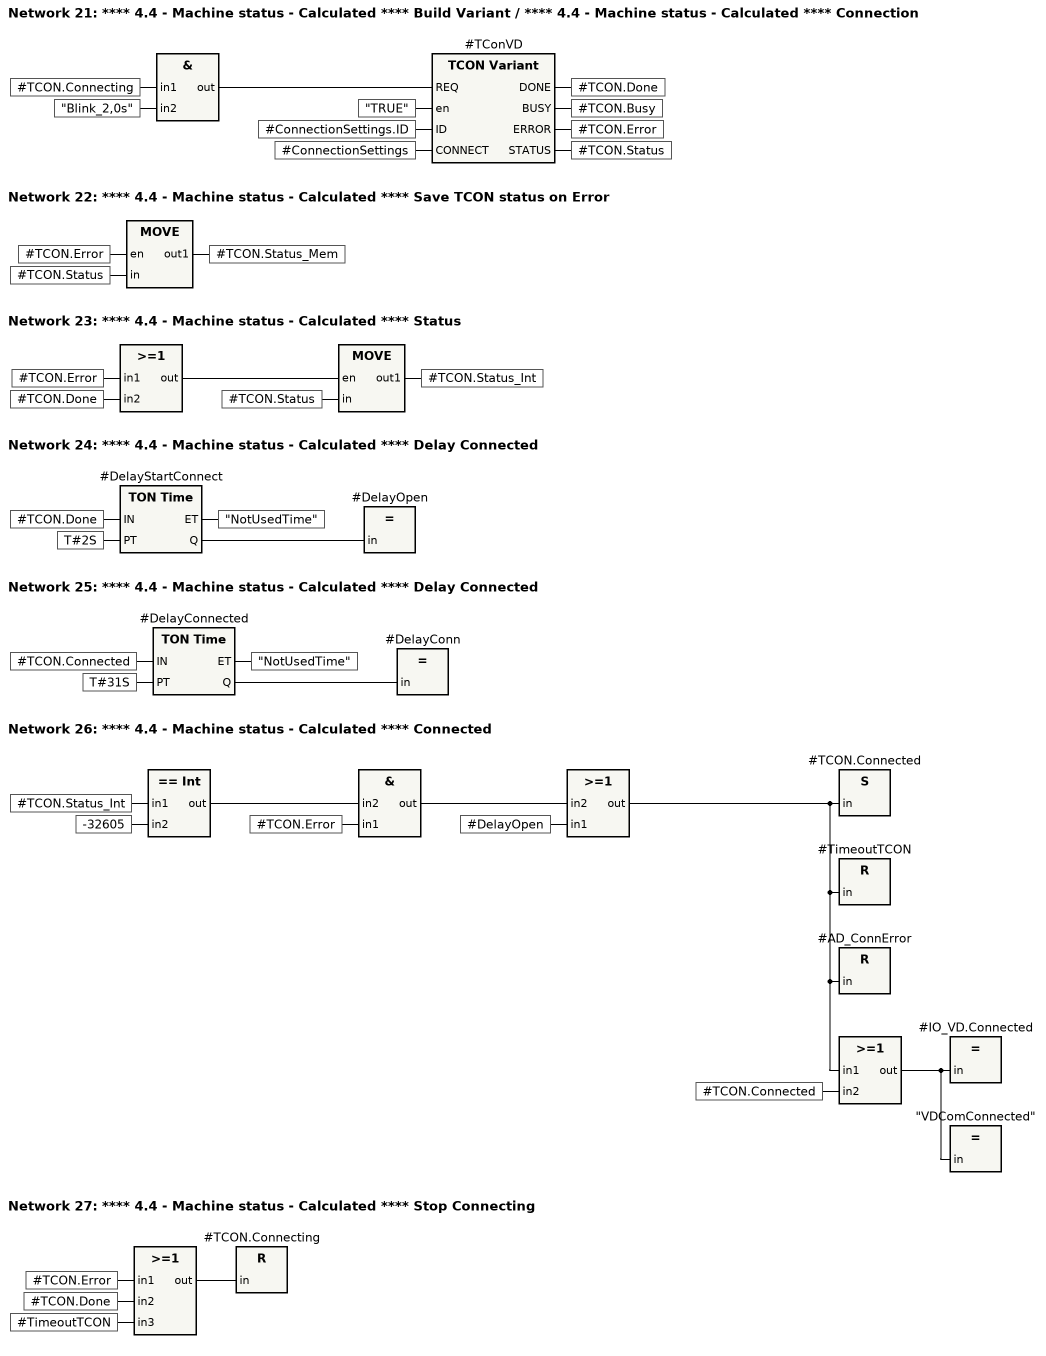
   IF "TRUE" THEN
       #TConVD(REQ := #TCON.Connecting AND "Blink_2,0s",   // TCON
               ID := #ConnectionSettings.ID,
               CONNECT := #ConnectionSettings,
               DONE => #TCON.Done,
               BUSY => #TCON.Busy,
               ERROR => #TCON.Error,
               STATUS => #TCON.Status);
   END_IF;
END_REGION

REGION Network 22: **** 4.4 - Machine status - Calculated **** Save TCON status on Error
   // Save TCON status on Error
   IF #TCON.Error THEN #TCON.Status_Mem := #TCON.Status; END_IF;
END_REGION

REGION Network 23: **** 4.4 - Machine status - Calculated **** Status
   // Status
   IF #TCON.Error OR #TCON.Done THEN #TCON.Status_Int := #TCON.Status; END_IF;
END_REGION

REGION Network 24: **** 4.4 - Machine status - Calculated **** Delay Connected
   // Delay Conected
   #DelayStartConnect(IN := #TCON.Done, PT := T#2S, ET => "NotUsedTime");   // TON
   #DelayOpen := #DelayStartConnect.Q;
END_REGION

REGION Network 25: **** 4.4 - Machine status - Calculated **** Delay Connected
   // Delay Conected
   #DelayConnected(IN := #TCON.Connected, PT := T#31S, ET => "NotUsedTime");   // TON
   #DelayConn := #DelayConnected.Q;
END_REGION

REGION Network 26: **** 4.4 - Machine status - Calculated **** Connected
   // Connected if ,Done bit or if connected already (80A3 = -32605)
   #_w1 := ((#TCON.Status_Int = (-32605)) AND #TCON.Error) OR #DelayOpen;
   IF #_w1 THEN
       #TCON.Connected := TRUE;
       #TimeoutTCON := FALSE;
       #AD_ConnError := FALSE;
   END_IF;
   #IO_VD.Connected := #_w1 OR #TCON.Connected;
   "VDComConnected" := #IO_VD.Connected;
END_REGION

REGION Network 27: **** 4.4 - Machine status - Calculated **** Stop Connecting
   // Stop connecting attempt if Error,Done,Connecting AND NOT Busy
   IF #TCON.Error OR #TCON.Done OR #TimeoutTCON THEN #TCON.Connecting := FALSE; END_IF;
END_REGION

REGION Network 28: **** 4.4 - Machine status - Calculated **** Timeout Disconnecting / **** 4.4 - Machine status - Calculated **** Disconnect on Receive
   // Timeout Disconnecting / Disconnect on Receive error or on HMI Request
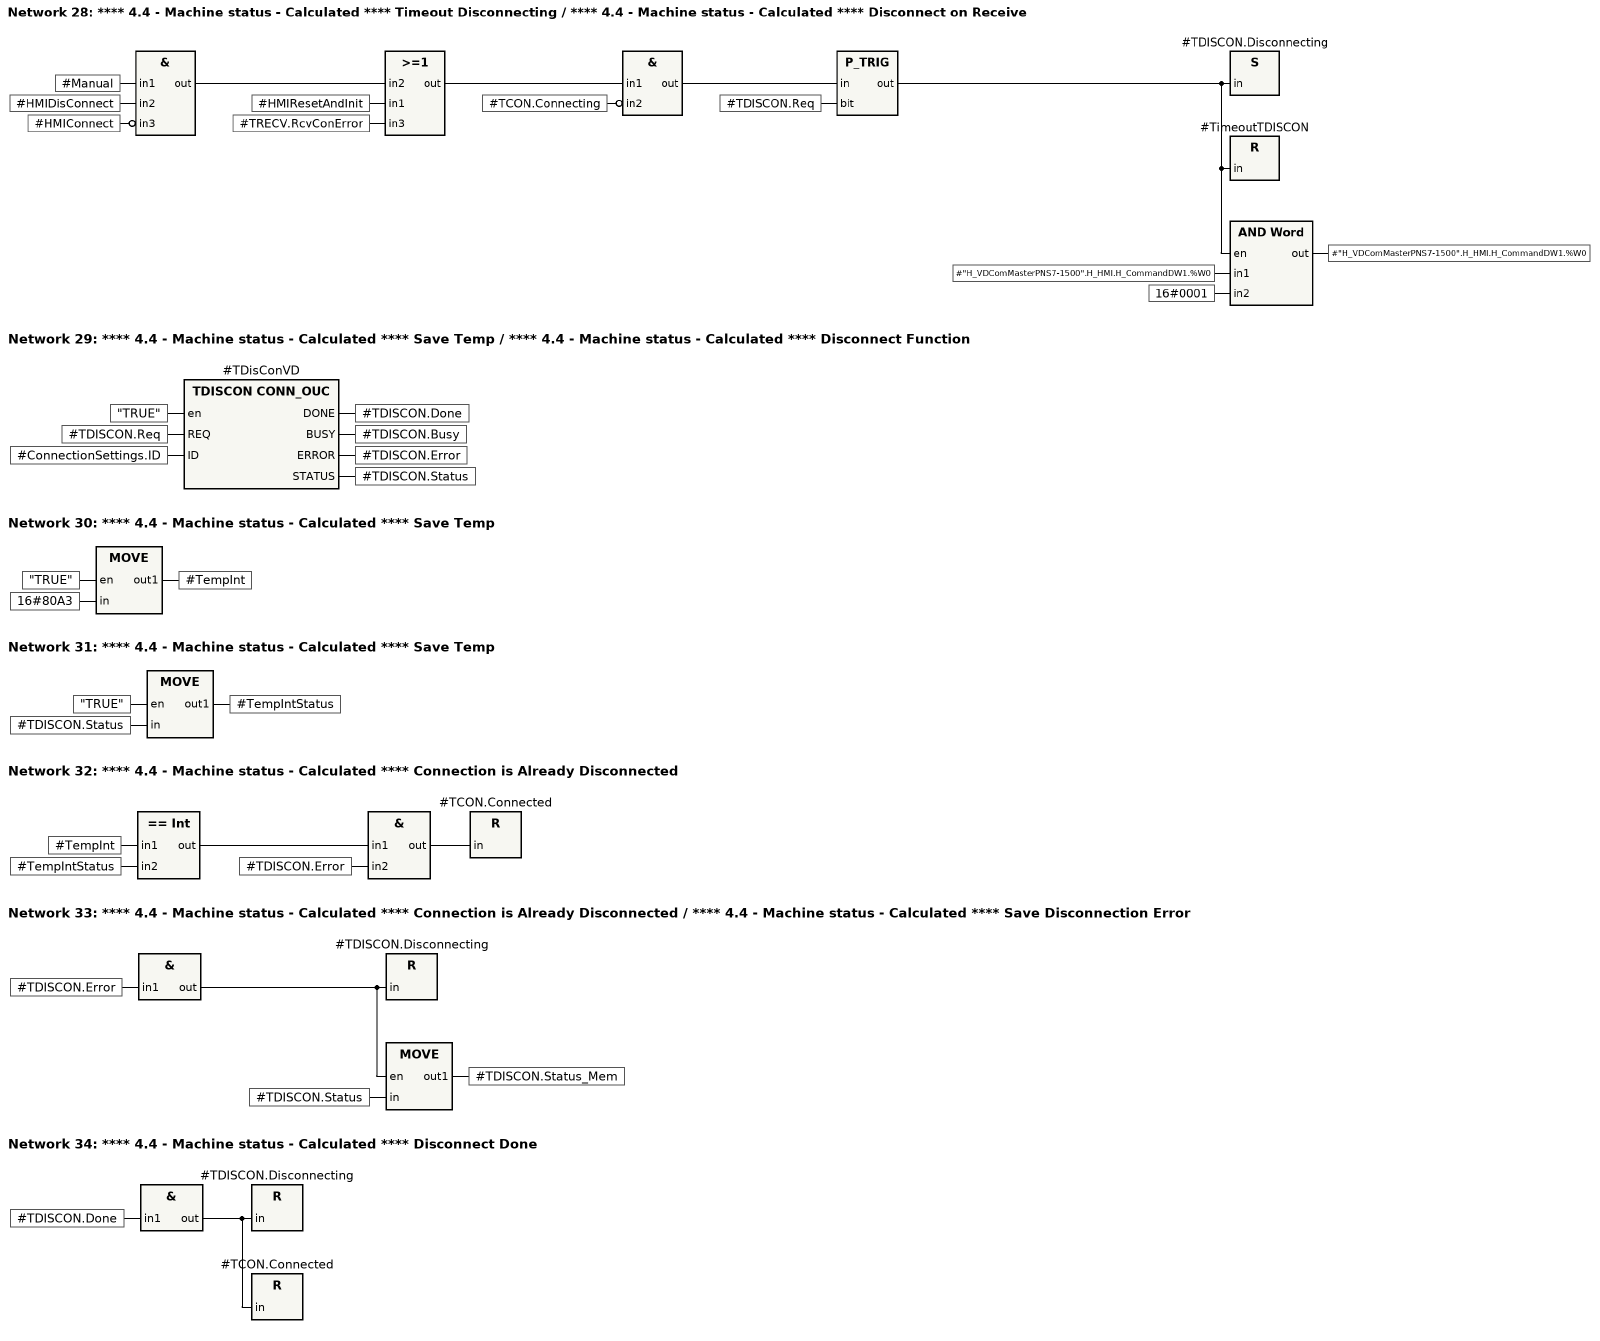
   #_w1 := ((#Manual AND #HMIDisConnect AND NOT #HMIConnect) OR #HMIResetAndInit OR #TRECV.RcvConError) AND NOT #TCON.Connecting;
   #_w2 := #_w1 AND NOT #TDISCON.Req;   // rising edge
   #TDISCON.Req := #_w1;
   IF #_w2 THEN
       #TDISCON.Disconnecting := TRUE;
       #TimeoutTDISCON := FALSE;
       #"H_VDComMasterPNS7-1500".H_HMI.H_CommandDW1.%W0 := #"H_VDComMasterPNS7-1500".H_HMI.H_CommandDW1.%W0 AND 16#0001;
   END_IF;
END_REGION

REGION Network 29: **** 4.4 - Machine status - Calculated **** Save Temp / **** 4.4 - Machine status - Calculated **** Disconnect Function
   // Temp / Disconnect function
   IF "TRUE" THEN
       #TDisConVD(REQ := #TDISCON.Req,   // TDISCON
                  ID := #ConnectionSettings.ID,
                  DONE => #TDISCON.Done,
                  BUSY => #TDISCON.Busy,
                  ERROR => #TDISCON.Error,
                  STATUS => #TDISCON.Status);
   END_IF;
END_REGION

REGION Network 30: **** 4.4 - Machine status - Calculated **** Save Temp
   // Temp
   IF "TRUE" THEN #TempInt := 16#80A3; END_IF;
END_REGION

REGION Network 31: **** 4.4 - Machine status - Calculated **** Save Temp
   // Temp
   IF "TRUE" THEN #TempIntStatus := #TDISCON.Status; END_IF;
END_REGION

REGION Network 32: **** 4.4 - Machine status - Calculated **** Connection is Already Disconnected
   // Connection is Already Disconnected
   IF (#TempInt = #TempIntStatus) AND #TDISCON.Error THEN #TCON.Connected := FALSE; END_IF;
END_REGION

REGION Network 33: **** 4.4 - Machine status - Calculated **** Connection is Already Disconnected / **** 4.4 - Machine status - Calculated **** Save Disconnection Error
   // Connection is Already Disconnected / Save Disconnection error
   IF #TDISCON.Error THEN
       #TDISCON.Disconnecting := FALSE;
       #TDISCON.Status_Mem := #TDISCON.Status;
   END_IF;
END_REGION

REGION Network 34: **** 4.4 - Machine status - Calculated **** Disconnect Done
   // Disconnect Done
   IF #TDISCON.Done THEN
       #TDISCON.Disconnecting := FALSE;
       #TCON.Connected := FALSE;
   END_IF;
END_REGION

REGION Network 35: **** 4.4 - Machine status - Calculated **** Diconnect / **** 4.4 - Machine status - Calculated **** Disconnect
   // Diconnect / Disconnect
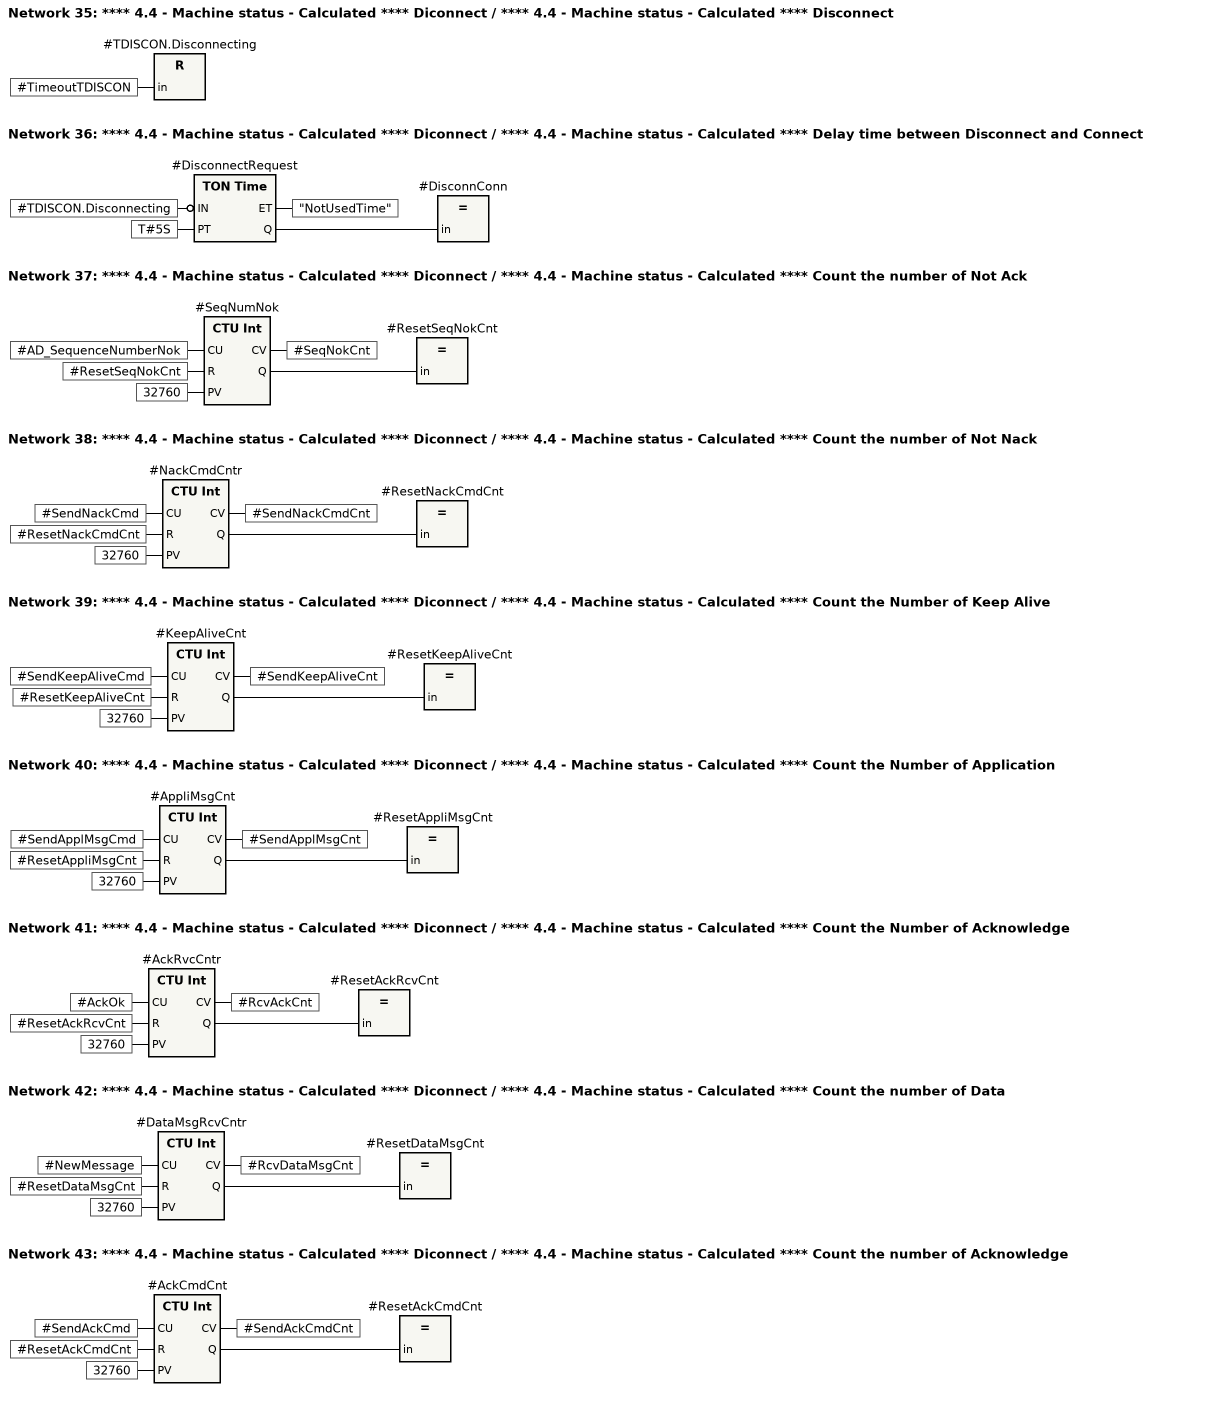
   IF #TimeoutTDISCON THEN #TDISCON.Disconnecting := FALSE; END_IF;
END_REGION

REGION Network 36: **** 4.4 - Machine status - Calculated **** Diconnect / **** 4.4 - Machine status - Calculated **** Delay time between Disconnect and Connect
   // Diconnect / Delay time between disconnect and connect
   #DisconnectRequest(IN := NOT #TDISCON.Disconnecting, PT := T#5S, ET => "NotUsedTime");   // TON
   #DisconnConn := #DisconnectRequest.Q;
END_REGION

REGION Network 37: **** 4.4 - Machine status - Calculated **** Diconnect / **** 4.4 - Machine status - Calculated **** Count the number of Not Ack
   // Diconnect / Count the number of Not acknowledge messages; for diagnostics only
   #SeqNumNok(CU := #AD_SequenceNumberNok, R := #ResetSeqNokCnt, PV := 32760, CV => #SeqNokCnt);   // CTU
   #ResetSeqNokCnt := #SeqNumNok.Q;
END_REGION

REGION Network 38: **** 4.4 - Machine status - Calculated **** Diconnect / **** 4.4 - Machine status - Calculated **** Count the number of Not Nack
   // Diconnect / Count the number of Not acknowledge messages; for diagnostics only
   #NackCmdCntr(CU := #SendNackCmd, R := #ResetNackCmdCnt, PV := 32760, CV => #SendNackCmdCnt);   // CTU
   #ResetNackCmdCnt := #NackCmdCntr.Q;
END_REGION

REGION Network 39: **** 4.4 - Machine status - Calculated **** Diconnect / **** 4.4 - Machine status - Calculated **** Count the Number of Keep Alive
   // Diconnect / Count the number of keep alive messages; for diagnostics only
   #KeepAliveCnt(CU := #SendKeepAliveCmd, R := #ResetKeepAliveCnt, PV := 32760, CV => #SendKeepAliveCnt);   // CTU
   #ResetKeepAliveCnt := #KeepAliveCnt.Q;
END_REGION

REGION Network 40: **** 4.4 - Machine status - Calculated **** Diconnect / **** 4.4 - Machine status - Calculated **** Count the Number of Application
   // Diconnect / Count the number of Application messages; for diagnostics only
   #AppliMsgCnt(CU := #SendApplMsgCmd, R := #ResetAppliMsgCnt, PV := 32760, CV => #SendApplMsgCnt);   // CTU
   #ResetAppliMsgCnt := #AppliMsgCnt.Q;
END_REGION

REGION Network 41: **** 4.4 - Machine status - Calculated **** Diconnect / **** 4.4 - Machine status - Calculated **** Count the Number of Acknowledge
   // Diconnect / Count the number of Acknowledge messages received; for diagnostics only
   #AckRvcCntr(CU := #AckOk, R := #ResetAckRcvCnt, PV := 32760, CV => #RcvAckCnt);   // CTU
   #ResetAckRcvCnt := #AckRvcCntr.Q;
END_REGION

REGION Network 42: **** 4.4 - Machine status - Calculated **** Diconnect / **** 4.4 - Machine status - Calculated **** Count the number of Data
   // Diconnect / Count the number of Data messages received; for diagnostics only
   #DataMsgRcvCntr(CU := #NewMessage, R := #ResetDataMsgCnt, PV := 32760, CV => #RcvDataMsgCnt);   // CTU
   #ResetDataMsgCnt := #DataMsgRcvCntr.Q;
END_REGION

REGION Network 43: **** 4.4 - Machine status - Calculated **** Diconnect / **** 4.4 - Machine status - Calculated **** Count the number of Acknowledge
   // Diconnect / Count the number of Acknowledge messages; for diagnostics only
   #AckCmdCnt(CU := #SendAckCmd, R := #ResetAckCmdCnt, PV := 32760, CV => #SendAckCmdCnt);   // CTU
   #ResetAckCmdCnt := #AckCmdCnt.Q;
END_REGION

NETWORK
TITLE = **** 4.4 - Machine status - Calculated **** Pointers
// Build the any pointers to the different DB's, needed for:
//  * BLKMOV (RecvPointer & BufferPointer)
//  * SEND (FB63 -> TSEND)
//  * RCV  (FB64 -> TRCV)
// Common Pointer parameters for
//  * RECV DB
//  * SEND DB
//  * SEND Buf DB
      LAR1  P##PointerRecv;
      L     16#1002;
      T     LW [AR1, P#0.0];
      LAR1  P##PointerSend;
      L     16#1002;
      T     LW [AR1, P#0.0];
      LAR1  P##PointerSendBuf;
      L     16#1002;
      T     LW [AR1, P#0.0];
// Cleaning Warnings APa
//      L     16#10                // S7  S7
//      T     %LB0                 // RECV
//      T     %LB10                // SEND
//      T     %LB20                // SEND BUF
//
//      L     16#02                //Data type (Bytes = 2)
//      T     %LB1                 // RECV
//      T     %LB11                // SEND
//      T     %LB21                // SEND BUF
      L     #RecvDBNbr;
      T     #RecvDBNO;

      CALL  ATTR_DB
      ( REQ       := "TRUE",
        DB_NUMBER := #RecvDBNO,
        RET_VAL   := "NotUsedInt",
        DB_LENGTH := #LengthDB,
        ATTRIB    := "NotUsedByte"
      );

//DB Header
      LAR1  P##PointerRecv;
      L     #LengthDB;
      T     LW [AR1, P#2.0];
      LAR1  P##PointerSend;
      L     16#000A;  //LengthLength
      T     LW [AR1, P#2.0];


//      L     #LengthDB
//      T     %LW2                 // RECV
//      L     16#000A              //LengthLength
//      T     %LW12                // SEND
      LAR1  P##PointerRecv;
      L     0;
      SLD   3;
      OD    16#8400_0000;
      T     LD [AR1, P#6.0];

      LAR1  P##PointerSend;
      L     0;
      SLD   3;
      OD    16#8400_0000;
      T     LD [AR1, P#6.0];


      LAR1  P##PointerSendBuf;
      L     0;
      SLD   3;
      OD    16#8400_0000;
      T     LD [AR1, P#6.0];

//      L     L#0                  //Offset in DB
//      SLD   3                    // Convert to pointer Convert to pointer
//      T     %LD6                 // RECV
//      T     %LD16                // SEND
//      T     %LD26                // SEND BUF

// Pointer to the Receive DB (Pointer_RECV) // DB no DB no
      LAR1  P##PointerRecv;
      L     #RecvDBNbr;
      T     LW [AR1, P#4.0];

//      L     #RecvDBNbr
//      T     %LW4                 // RECV

// Pointer to the Send DB (Pointer_SEND) Pointer to the Send DB (Pointer_SEND)
// DB no DB no
      LAR1  P##PointerSend;
      L     #SendDBNbr;
      T     LW [AR1, P#4.0];

//      L     #SendDBNbr
//      T     %LW14                // SEND

// Set memory area to DB Set memory area to DB
//      L     16#84                // Memory area DB Memory area DB
//      T     %LB6                 // RECV
//      T     %LB16                // SEND
//      T     %LB26                // SEND BUF




REGION Network 45: **** 4.4 - Machine status - Calculated **** Received Data
   // Received Data:
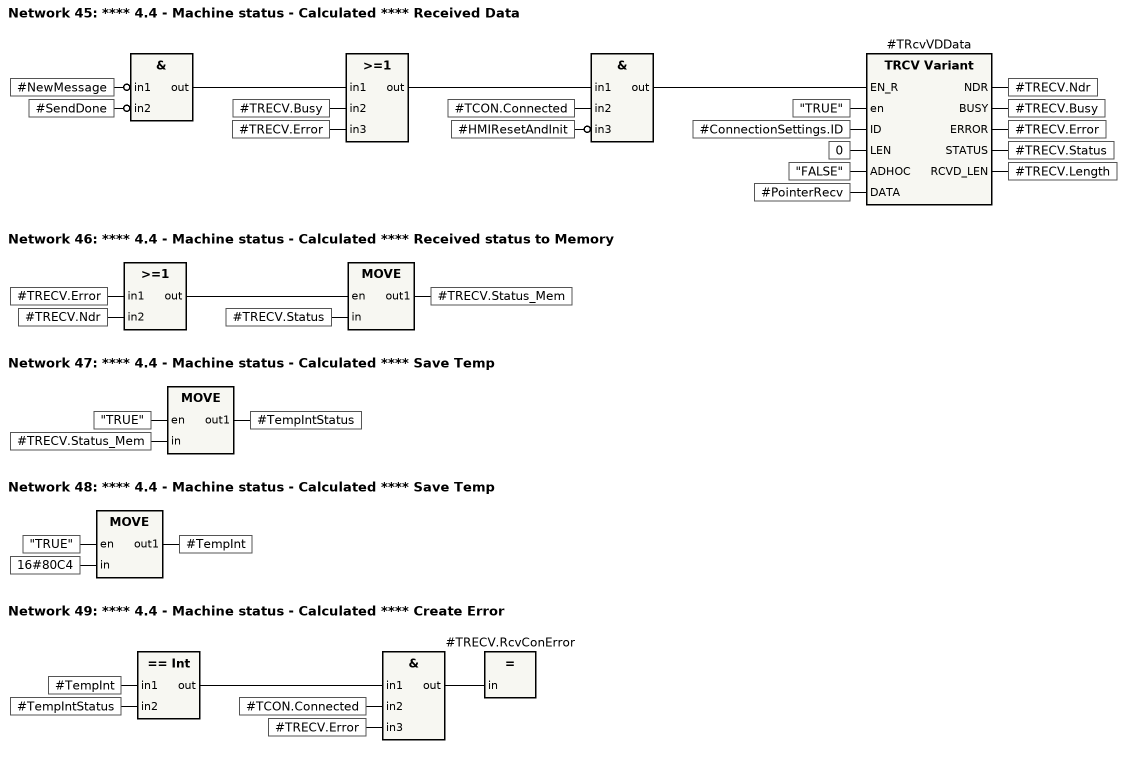
   IF "TRUE" THEN
       #TRcvVDData(EN_R := ((NOT #NewMessage AND NOT #SendDone) OR #TRECV.Busy OR #TRECV.Error) AND #TCON.Connected AND NOT #HMIResetAndInit,   // TRCV
                   ID := #ConnectionSettings.ID,
                   LEN := 0,
                   ADHOC := "FALSE",
                   DATA := #PointerRecv,
                   NDR => #TRECV.Ndr,
                   BUSY => #TRECV.Busy,
                   ERROR => #TRECV.Error,
                   STATUS => #TRECV.Status,
                   RCVD_LEN => #TRECV.Length);
   END_IF;
END_REGION

REGION Network 46: **** 4.4 - Machine status - Calculated **** Received status to Memory
   // Received status to memory
   IF #TRECV.Error OR #TRECV.Ndr THEN #TRECV.Status_Mem := #TRECV.Status; END_IF;
END_REGION

REGION Network 47: **** 4.4 - Machine status - Calculated **** Save Temp
   // Temp
   IF "TRUE" THEN #TempIntStatus := #TRECV.Status_Mem; END_IF;
END_REGION

REGION Network 48: **** 4.4 - Machine status - Calculated **** Save Temp
   // Temp
   IF "TRUE" THEN #TempInt := 16#80C4; END_IF;
END_REGION

REGION Network 49: **** 4.4 - Machine status - Calculated **** Create Error
   // Create error when status is equal to 0x80C4
   #TRECV.RcvConError := (#TempInt = #TempIntStatus) AND #TCON.Connected AND #TRECV.Error;
END_REGION

REGION Network 50: **** 4.6 - Machine Status - Indication **** Icon Animation
   // Icon Animation
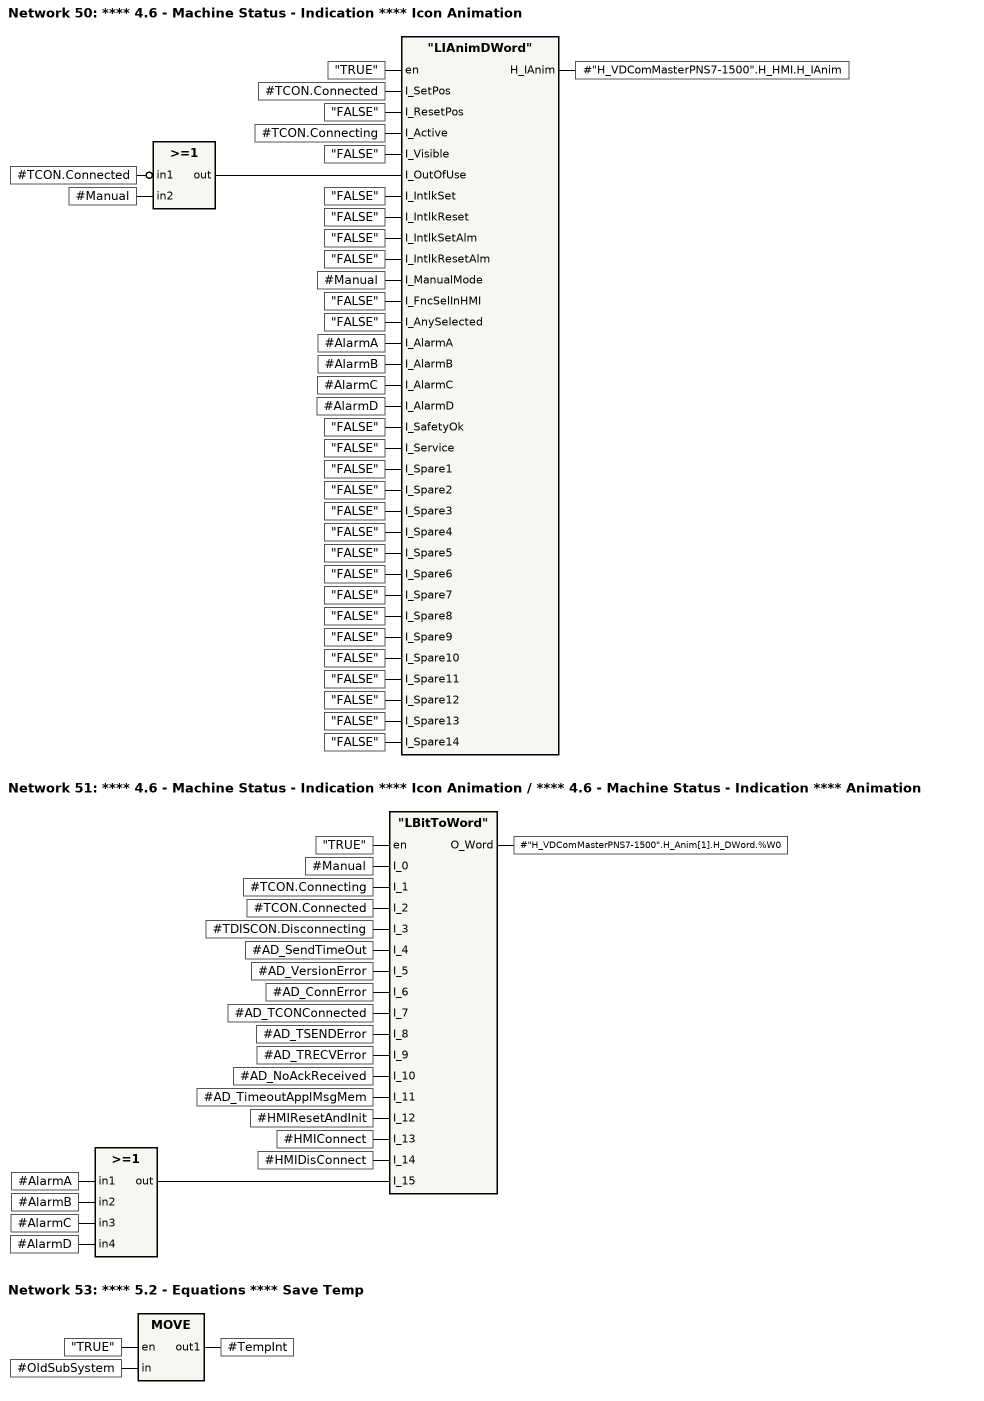
   IF "TRUE" THEN
       "LIAnimDWord"(I_SetPos := #TCON.Connected,
                     I_ResetPos := "FALSE",
                     I_Active := #TCON.Connecting,
                     I_Visible := "FALSE",
                     I_OutOfUse := NOT #TCON.Connected OR #Manual,
                     I_IntlkSet := "FALSE",
                     I_IntlkReset := "FALSE",
                     I_IntlkSetAlm := "FALSE",
                     I_IntlkResetAlm := "FALSE",
                     I_ManualMode := #Manual,
                     I_FncSelInHMI := "FALSE",
                     I_AnySelected := "FALSE",
                     I_AlarmA := #AlarmA,
                     I_AlarmB := #AlarmB,
                     I_AlarmC := #AlarmC,
                     I_AlarmD := #AlarmD,
                     I_SafetyOk := "FALSE",
                     I_Service := "FALSE",
                     I_Spare1 := "FALSE",
                     I_Spare2 := "FALSE",
                     I_Spare3 := "FALSE",
                     I_Spare4 := "FALSE",
                     I_Spare5 := "FALSE",
                     I_Spare6 := "FALSE",
                     I_Spare7 := "FALSE",
                     I_Spare8 := "FALSE",
                     I_Spare9 := "FALSE",
                     I_Spare10 := "FALSE",
                     I_Spare11 := "FALSE",
                     I_Spare12 := "FALSE",
                     I_Spare13 := "FALSE",
                     I_Spare14 := "FALSE",
                     H_IAnim => #"H_VDComMasterPNS7-1500".H_HMI.H_IAnim);
   END_IF;
END_REGION

REGION Network 51: **** 4.6 - Machine Status - Indication **** Icon Animation / **** 4.6 - Machine Status - Indication **** Animation
   // Icon Animation / Animation
   IF "TRUE" THEN
       "LBitToWord"(I_0 := #Manual,
                    I_1 := #TCON.Connecting,
                    I_2 := #TCON.Connected,
                    I_3 := #TDISCON.Disconnecting,
                    I_4 := #AD_SendTimeOut,
                    I_5 := #AD_VersionError,
                    I_6 := #AD_ConnError,
                    I_7 := #AD_TCONConnected,
                    I_8 := #AD_TSENDError,
                    I_9 := #AD_TRECVError,
                    I_10 := #AD_NoAckReceived,
                    I_11 := #AD_TimeoutApplMsgMem,
                    I_12 := #HMIResetAndInit,
                    I_13 := #HMIConnect,
                    I_14 := #HMIDisConnect,
                    I_15 := #AlarmA OR #AlarmB OR #AlarmC OR #AlarmD,
                    O_Word => #"H_VDComMasterPNS7-1500".H_Anim[1].H_DWord.%W0);
   END_IF;
END_REGION

NETWORK
TITLE = **** 5.2 - Equations **** MessageType to Local Variable
// Check that the received data is Ok Copy MessageType to local variable
      OPN   #I_VDCommRecvDB;
      L     %DBW0;  // VDVersion must always be same
      L     16#0100;
      <>I;
      =     #AD_VersionError;

      L     16#0100;
      T     %DBW0;

// Check new SeqNbr
      A     #TRECV.Ndr;  // New data is received
      A(;
      O(;
      L     %DBW8;  // Check seq nbr Ok
      L     #OldRecMsgNbr;
      <>I;
      );
      O(;
      L     %DBW8;  // Check seq nbr Ok
      L     0;
      ==I;
      );
      );
      S     #NewMsgNbr;

//-----------------------------------------------------------
// For next cycle OldRecSeqNbr=0 NewSeqNbr will always be Ok
//      L     -1
//      T     #OldRecMsgNbr
//-----------------------------------------------------------

// Check Messagetype
      L     %DBW4;
      L     2;
      >I;
      =     #UserMsgType;  // Messagetype > 2 then Ok message
      AN    #UserMsgType;
      JC    RSEQ;
//Remember messagenumber
      L     %DBW8;
      T     #OldRecMsgNbr;  // Remember last seq nbr
      L     %DBW6;
      T     #OldSubSystem;  // Remember last subsystem
RSEQ: NOP   0;

// Ack recieved Ack recieved
      L     %DBW4;
      L     1;
      ==I;
      =     #AckRcvd;

      L     %DBW8;
      L     #SendMsgNbr;
      ==I;
      =     #SeqNbrOk;  // Sequence number Ok for Ack rcvd

// Message length
      L     %DBW2;  // Message length in DB_RECV
      T     #MessageLengthRecv;

// Sequence number NOK
      A     #TRECV.Ndr;  // New data is received
      A     #UserMsgType;  // Data is of User type
      AN    #NewMsgNbr;  // Sequence number is NOK
      O     #AD_SequenceNumberNok;  // Hold status
      AN    #NewMsgNbr;  // Sequence number is NOK
      =     #AD_SequenceNumberNok;  // Sequence number NOK



REGION Network 53: **** 5.2 - Equations **** Save Temp
   // Temp
   IF "TRUE" THEN #TempInt := #OldSubSystem; END_IF;
END_REGION

REGION Network 54: **** 5.2 - Equations **** Receive Length
   // Receive length only copy if Ndr of read is set to 1
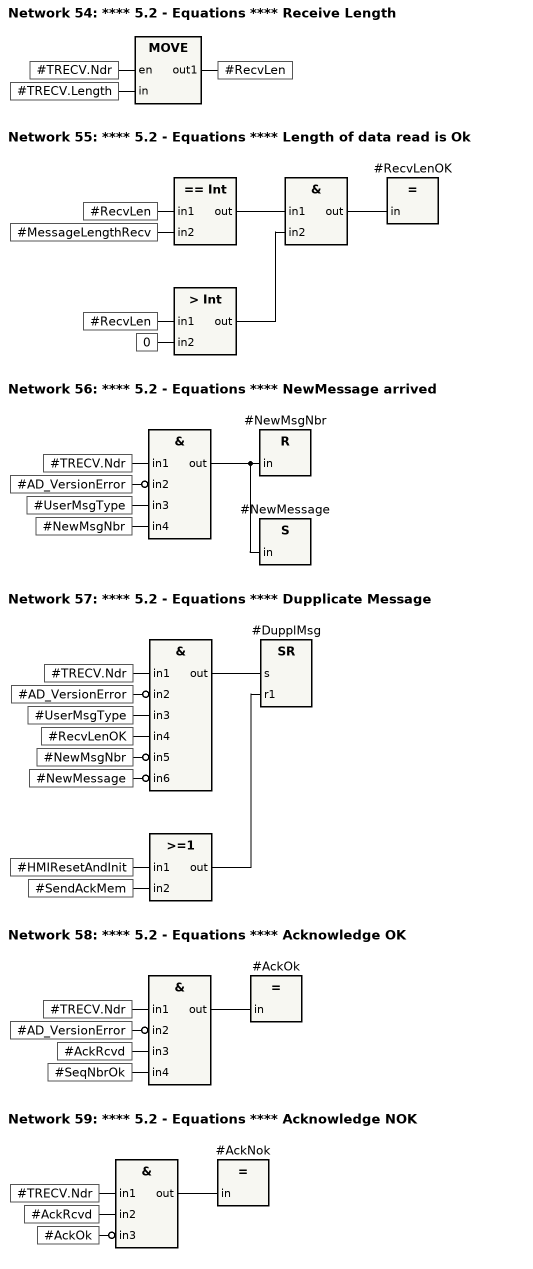
   IF #TRECV.Ndr THEN #RecvLen := #TRECV.Length; END_IF;
END_REGION

REGION Network 55: **** 5.2 - Equations **** Length of data read is Ok
   // Length of data read is Ok
   #RecvLenOK := (#RecvLen = #MessageLengthRecv) AND (#RecvLen > 0);
END_REGION

REGION Network 56: **** 5.2 - Equations **** NewMessage arrived
   // If new data is available and the data is Ok, then set output to subsystems NewMessage arrived.
   #_w1 := #TRECV.Ndr AND NOT #AD_VersionError AND #UserMsgType AND #NewMsgNbr;
   IF #_w1 THEN
       #NewMsgNbr := FALSE;
       #NewMessage := TRUE;
   END_IF;
END_REGION

REGION Network 57: **** 5.2 - Equations **** Dupplicate Message
   // Dupplicate Message
   IF #TRECV.Ndr AND NOT #AD_VersionError AND #UserMsgType AND #RecvLenOK AND NOT #NewMsgNbr AND NOT #NewMessage THEN
       #DupplMsg := TRUE;   // SR flip-flop
   END_IF;
   IF #HMIResetAndInit OR #SendAckMem THEN #DupplMsg := FALSE; END_IF;
END_REGION

REGION Network 58: **** 5.2 - Equations **** Acknowledge OK
   // Acknowledge OK
   #AckOk := #TRECV.Ndr AND NOT #AD_VersionError AND #AckRcvd AND #SeqNbrOk;
END_REGION

REGION Network 59: **** 5.2 - Equations **** Acknowledge NOK
   // Acknowledge not OK
   #AckNok := #TRECV.Ndr AND #AckRcvd AND NOT #AckOk;
END_REGION

REGION Network 60: **** 7.2 - Submodules - Command **** Postpone Send Ack
   // Time to postpone to send Ack upon reception of new message. This to prevent thatmessages are send too fast.
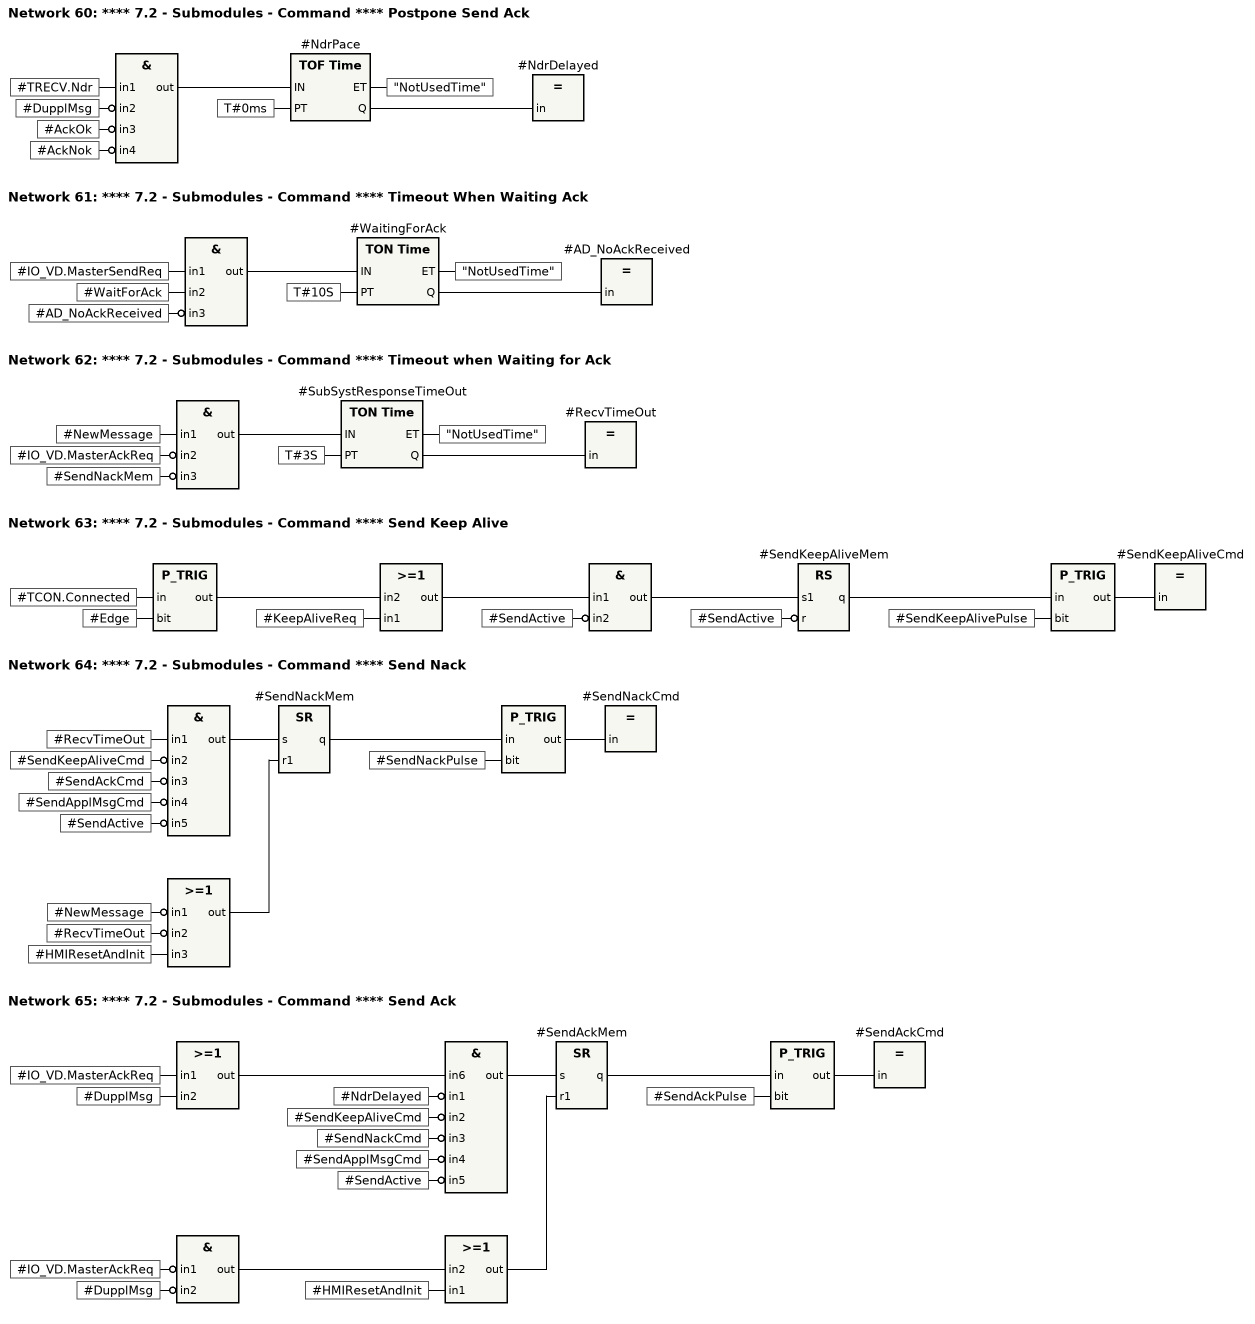
   #NdrPace(IN := #TRECV.Ndr AND NOT #DupplMsg AND NOT #AckOk AND NOT #AckNok, PT := T#0ms, ET => "NotUsedTime");   // TOF
   #NdrDelayed := #NdrPace.Q;
END_REGION

REGION Network 61: **** 7.2 - Submodules - Command **** Timeout When Waiting Ack
   // Timeout when waiting for Ack from superior system
   #WaitingForAck(IN := #IO_VD.MasterSendReq AND #WaitForAck AND NOT #AD_NoAckReceived,   // TON
                  PT := T#10S,
                  ET => "NotUsedTime");
   #AD_NoAckReceived := #WaitingForAck.Q;
END_REGION

REGION Network 62: **** 7.2 - Submodules - Command **** Timeout when Waiting for Ack
   // Timeout when waiting for Acknowlegde Request from Subsystem
   #SubSystResponseTimeOut(IN := #NewMessage AND NOT #IO_VD.MasterAckReq AND NOT #SendNackMem,   // TON
                           PT := T#3S,
                           ET => "NotUsedTime");
   #RecvTimeOut := #SubSystResponseTimeOut.Q;
END_REGION

REGION Network 63: **** 7.2 - Submodules - Command **** Send Keep Alive
   // Send Keep Alive
   #_w1 := #TCON.Connected AND NOT #Edge;   // rising edge
   #Edge := #TCON.Connected;
   IF NOT #SendActive THEN
       #SendKeepAliveMem := FALSE;   // RS flip-flop
   END_IF;
   IF (#_w1 OR #KeepAliveReq) AND NOT #SendActive THEN #SendKeepAliveMem := TRUE; END_IF;
   #_w2 := #SendKeepAliveMem AND NOT #SendKeepAlivePulse;   // rising edge
   #SendKeepAlivePulse := #SendKeepAliveMem;
   #SendKeepAliveCmd := #_w2;
END_REGION

REGION Network 64: **** 7.2 - Submodules - Command **** Send Nack
   // Send Nack when no subsystem is reacting on a new message received. This means 
   // that the new messages was not recognised by one of the subsystems ( subsystem 
   // number wrong or Messagetype wrong). Then the sender should be aware that what 
   // was send has no client.
   IF #RecvTimeOut AND NOT #SendKeepAliveCmd AND NOT #SendAckCmd AND NOT #SendApplMsgCmd AND NOT #SendActive THEN
       #SendNackMem := TRUE;   // SR flip-flop
   END_IF;
   IF NOT #NewMessage OR NOT #RecvTimeOut OR #HMIResetAndInit THEN #SendNackMem := FALSE; END_IF;
   #_w1 := #SendNackMem AND NOT #SendNackPulse;   // rising edge
   #SendNackPulse := #SendNackMem;
   #SendNackCmd := #_w1;
END_REGION

REGION Network 65: **** 7.2 - Submodules - Command **** Send Ack
   // Send Ack
   IF (#IO_VD.MasterAckReq OR #DupplMsg) AND NOT #NdrDelayed AND NOT #SendKeepAliveCmd AND NOT #SendNackCmd AND NOT #SendApplMsgCmd AND NOT #SendActive THEN
       #SendAckMem := TRUE;   // SR flip-flop
   END_IF;
   IF (NOT #IO_VD.MasterAckReq AND NOT #DupplMsg) OR #HMIResetAndInit THEN #SendAckMem := FALSE; END_IF;
   #_w1 := #SendAckMem AND NOT #SendAckPulse;   // rising edge
   #SendAckPulse := #SendAckMem;
   #SendAckCmd := #_w1;
END_REGION

REGION Network 66: **** 7.2 - Submodules - Command **** Ack Nack Sent
   // Ack Nack Sent
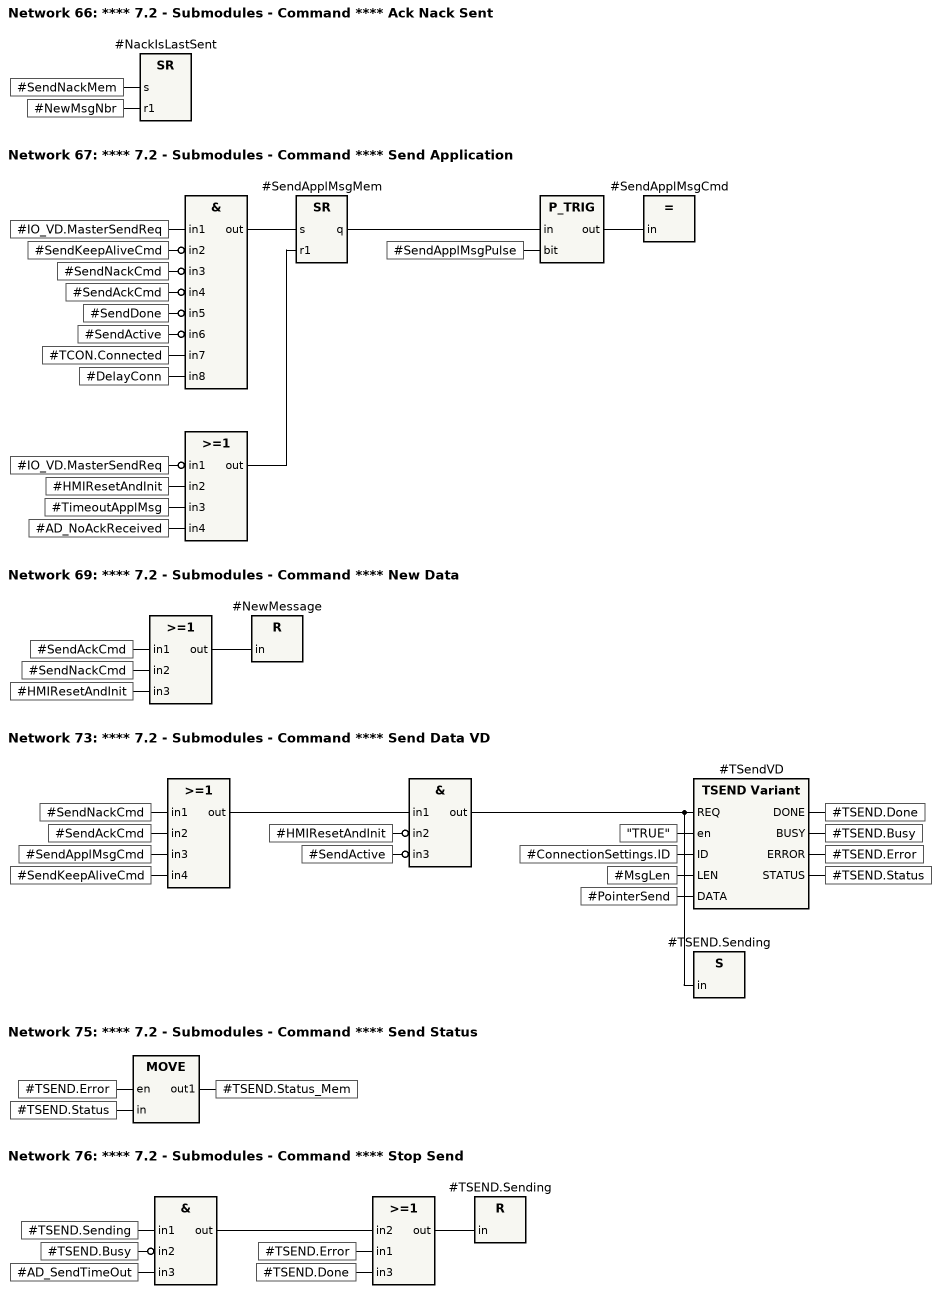
   IF #SendNackMem THEN
       #NackIsLastSent := TRUE;   // SR flip-flop
   END_IF;
   IF #NewMsgNbr THEN #NackIsLastSent := FALSE; END_IF;
END_REGION

REGION Network 67: **** 7.2 - Submodules - Command **** Send Application
   // Send Application
   IF #IO_VD.MasterSendReq AND NOT #SendKeepAliveCmd AND NOT #SendNackCmd AND NOT #SendAckCmd AND NOT #SendDone AND NOT #SendActive AND #TCON.Connected AND #DelayConn THEN
       #SendApplMsgMem := TRUE;   // SR flip-flop
   END_IF;
   IF NOT #IO_VD.MasterSendReq OR #HMIResetAndInit OR #TimeoutApplMsg OR #AD_NoAckReceived THEN
       #SendApplMsgMem := FALSE;
   END_IF;
   #_w1 := #SendApplMsgMem AND NOT #SendApplMsgPulse;   // rising edge
   #SendApplMsgPulse := #SendApplMsgMem;
   #SendApplMsgCmd := #_w1;
END_REGION

NETWORK
TITLE = **** 7.2 - Submodules - Command **** Send Application Sub System
// Send Application Sub System
      A     #SendApplMsgCmd;
      JCN   nOZE;
      OPN   #IO_VD.VDCommSendDB;
      L     %DBW6;
      T     #"H_VDComMasterPNS7-1500".H_Anim[2].H_DWord.%W0;
nOZE: NOP   0;


REGION Network 69: **** 7.2 - Submodules - Command **** New Data
   // If New Data is Available And the data is Ok, then set output to subsystems
   IF #SendAckCmd OR #SendNackCmd OR #HMIResetAndInit THEN #NewMessage := FALSE; END_IF;
END_REGION

NETWORK
TITLE = **** 7.2 - Submodules - Command **** Keep Alive
// Keep Alive command
      A     #SendKeepAliveCmd;
      JCN   SKAC;
      OPN   #I_VDCommSendDB;
      L     10;  //LengthLength
      T     %DBW2;
      L     2;  // MessageTypeMessageType
      T     %DBW4;
      L     0;  // Subsystem
      T     %DBW6;
      L     0;  // MessageNumber (SeqNbr)
      T     %DBW8;
SKAC: NOP   0;


